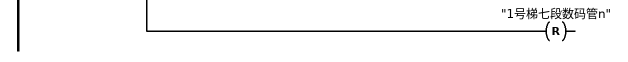
   RUNG wire#powerrail
      { S7_Templates := "SrcType := Int" } EQ_Contact(in1 := "1号梯当前楼层数", in2 := 1)
      wire#w1
      R_Coil( "1号梯七段数码管a" )
   END_RUNG
   RUNG wire#w1
      S_Coil( "1号梯七段数码管b" )
   END_RUNG
   RUNG wire#w1
      S_Coil( "1号梯七段数码管c" )
   END_RUNG
   RUNG wire#w1
      R_Coil( "1号梯七段数码管d" )
   END_RUNG
   RUNG wire#w1
      R_Coil( "1号梯七段数码管e" )
   END_RUNG
   RUNG wire#w1
      R_Coil( "1号梯七段数码管f" )
   END_RUNG
   RUNG wire#w1
      R_Coil( "1号梯七段数码管g" )
   END_RUNG
   RUNG wire#w1
      R_Coil( "1号梯七段数码管h" )
   END_RUNG
   RUNG wire#w1
      R_Coil( "1号梯七段数码管i" )
   END_RUNG
   RUNG wire#w1
      R_Coil( "1号梯七段数码管j" )
   END_RUNG
   RUNG wire#w1
      R_Coil( "1号梯七段数码管k" )
   END_RUNG
   RUNG wire#w1
      R_Coil( "1号梯七段数码管l" )
   END_RUNG
   RUNG wire#w1
      R_Coil( "1号梯七段数码管m" )
   END_RUNG
   RUNG wire#w1
      R_Coil( "1号梯七段数码管n" )
   END_RUNG
   RUNG wire#powerrail
      { S7_Templates := "SrcType := Int" } EQ_Contact(in1 := "1号梯当前楼层数", in2 := 2)
      wire#w2
      S_Coil( "1号梯七段数码管a" )
   END_RUNG
   RUNG wire#w2
      S_Coil( "1号梯七段数码管b" )
   END_RUNG
   RUNG wire#w2
      R_Coil( "1号梯七段数码管c" )
   END_RUNG
   RUNG wire#w2
      S_Coil( "1号梯七段数码管d" )
   END_RUNG
   RUNG wire#w2
      S_Coil( "1号梯七段数码管e" )
   END_RUNG
   RUNG wire#w2
      R_Coil( "1号梯七段数码管f" )
   END_RUNG
   RUNG wire#w2
      S_Coil( "1号梯七段数码管g" )
   END_RUNG
   RUNG wire#w2
      R_Coil( "1号梯七段数码管h" )
   END_RUNG
   RUNG wire#w2
      R_Coil( "1号梯七段数码管i" )
   END_RUNG
   RUNG wire#w2
      R_Coil( "1号梯七段数码管j" )
   END_RUNG
   RUNG wire#w2
      R_Coil( "1号梯七段数码管k" )
   END_RUNG
   RUNG wire#w2
      R_Coil( "1号梯七段数码管l" )
   END_RUNG
   RUNG wire#w2
      R_Coil( "1号梯七段数码管m" )
   END_RUNG
   RUNG wire#w2
      R_Coil( "1号梯七段数码管n" )
   END_RUNG
   RUNG wire#powerrail
      { S7_Templates := "SrcType := Int" } EQ_Contact(in1 := "1号梯当前楼层数", in2 := 3)
      wire#w3
      S_Coil( "1号梯七段数码管a" )
   END_RUNG
   RUNG wire#w3
      S_Coil( "1号梯七段数码管b" )
   END_RUNG
   RUNG wire#w3
      S_Coil( "1号梯七段数码管c" )
   END_RUNG
   RUNG wire#w3
      S_Coil( "1号梯七段数码管d" )
   END_RUNG
   RUNG wire#w3
      R_Coil( "1号梯七段数码管e" )
   END_RUNG
   RUNG wire#w3
      R_Coil( "1号梯七段数码管f" )
   END_RUNG
   RUNG wire#w3
      S_Coil( "1号梯七段数码管g" )
   END_RUNG
   RUNG wire#w3
      R_Coil( "1号梯七段数码管h" )
   END_RUNG
   RUNG wire#w3
      R_Coil( "1号梯七段数码管i" )
   END_RUNG
   RUNG wire#w3
      R_Coil( "1号梯七段数码管j" )
   END_RUNG
   RUNG wire#w3
      R_Coil( "1号梯七段数码管k" )
   END_RUNG
   RUNG wire#w3
      R_Coil( "1号梯七段数码管l" )
   END_RUNG
   RUNG wire#w3
      R_Coil( "1号梯七段数码管m" )
   END_RUNG
   RUNG wire#w3
      R_Coil( "1号梯七段数码管n" )
   END_RUNG
   RUNG wire#powerrail
      { S7_Templates := "SrcType := Int" } EQ_Contact(in1 := "1号梯当前楼层数", in2 := 4)
      wire#w4
      R_Coil( "1号梯七段数码管a" )
   END_RUNG
   RUNG wire#w4
      S_Coil( "1号梯七段数码管b" )
   END_RUNG
   RUNG wire#w4
      S_Coil( "1号梯七段数码管c" )
   END_RUNG
   RUNG wire#w4
      R_Coil( "1号梯七段数码管d" )
   END_RUNG
   RUNG wire#w4
      R_Coil( "1号梯七段数码管e" )
   END_RUNG
   RUNG wire#w4
      S_Coil( "1号梯七段数码管f" )
   END_RUNG
   RUNG wire#w4
      S_Coil( "1号梯七段数码管g" )
   END_RUNG
   RUNG wire#w4
      R_Coil( "1号梯七段数码管h" )
   END_RUNG
   RUNG wire#w4
      R_Coil( "1号梯七段数码管i" )
   END_RUNG
   RUNG wire#w4
      R_Coil( "1号梯七段数码管j" )
   END_RUNG
   RUNG wire#w4
      R_Coil( "1号梯七段数码管k" )
   END_RUNG
   RUNG wire#w4
      R_Coil( "1号梯七段数码管l" )
   END_RUNG
   RUNG wire#w4
      R_Coil( "1号梯七段数码管m" )
   END_RUNG
   RUNG wire#w4
      R_Coil( "1号梯七段数码管n" )
   END_RUNG
   RUNG wire#powerrail
      { S7_Templates := "SrcType := Int" } EQ_Contact(in1 := "1号梯当前楼层数", in2 := 5)
      wire#w5
      S_Coil( "1号梯七段数码管a" )
   END_RUNG
   RUNG wire#w5
      R_Coil( "1号梯七段数码管b" )
   END_RUNG
   RUNG wire#w5
      S_Coil( "1号梯七段数码管c" )
   END_RUNG
   RUNG wire#w5
      S_Coil( "1号梯七段数码管d" )
   END_RUNG
   RUNG wire#w5
      R_Coil( "1号梯七段数码管e" )
   END_RUNG
   RUNG wire#w5
      S_Coil( "1号梯七段数码管f" )
   END_RUNG
   RUNG wire#w5
      S_Coil( "1号梯七段数码管g" )
   END_RUNG
   RUNG wire#w5
      R_Coil( "1号梯七段数码管h" )
   END_RUNG
   RUNG wire#w5
      R_Coil( "1号梯七段数码管i" )
   END_RUNG
   RUNG wire#w5
      R_Coil( "1号梯七段数码管j" )
   END_RUNG
   RUNG wire#w5
      R_Coil( "1号梯七段数码管k" )
   END_RUNG
   RUNG wire#w5
      R_Coil( "1号梯七段数码管l" )
   END_RUNG
   RUNG wire#w5
      R_Coil( "1号梯七段数码管m" )
   END_RUNG
   RUNG wire#w5
      R_Coil( "1号梯七段数码管n" )
   END_RUNG
   RUNG wire#powerrail
      { S7_Templates := "SrcType := Int" } EQ_Contact(in1 := "1号梯当前楼层数", in2 := 6)
      wire#w6
      S_Coil( "1号梯七段数码管a" )
   END_RUNG
   RUNG wire#w6
      R_Coil( "1号梯七段数码管b" )
   END_RUNG
   RUNG wire#w6
      S_Coil( "1号梯七段数码管c" )
   END_RUNG
   RUNG wire#w6
      S_Coil( "1号梯七段数码管d" )
   END_RUNG
   RUNG wire#w6
      S_Coil( "1号梯七段数码管e" )
   END_RUNG
   RUNG wire#w6
      S_Coil( "1号梯七段数码管f" )
   END_RUNG
   RUNG wire#w6
      S_Coil( "1号梯七段数码管g" )
   END_RUNG
   RUNG wire#w6
      R_Coil( "1号梯七段数码管h" )
   END_RUNG
   RUNG wire#w6
      R_Coil( "1号梯七段数码管i" )
   END_RUNG
   RUNG wire#w6
      R_Coil( "1号梯七段数码管j" )
   END_RUNG
   RUNG wire#w6
      R_Coil( "1号梯七段数码管k" )
   END_RUNG
   RUNG wire#w6
      R_Coil( "1号梯七段数码管l" )
   END_RUNG
   RUNG wire#w6
      R_Coil( "1号梯七段数码管m" )
   END_RUNG
   RUNG wire#w6
      R_Coil( "1号梯七段数码管n" )
   END_RUNG
   RUNG wire#powerrail
      { S7_Templates := "SrcType := Int" } EQ_Contact(in1 := "1号梯当前楼层数", in2 := 7)
      wire#w7
      S_Coil( "1号梯七段数码管a" )
   END_RUNG
   RUNG wire#w7
      S_Coil( "1号梯七段数码管b" )
   END_RUNG
   RUNG wire#w7
      S_Coil( "1号梯七段数码管c" )
   END_RUNG
   RUNG wire#w7
      R_Coil( "1号梯七段数码管d" )
   END_RUNG
   RUNG wire#w7
      R_Coil( "1号梯七段数码管e" )
   END_RUNG
   RUNG wire#w7
      R_Coil( "1号梯七段数码管f" )
   END_RUNG
   RUNG wire#w7
      R_Coil( "1号梯七段数码管g" )
   END_RUNG
   RUNG wire#w7
      R_Coil( "1号梯七段数码管h" )
   END_RUNG
   RUNG wire#w7
      R_Coil( "1号梯七段数码管i" )
   END_RUNG
   RUNG wire#w7
      R_Coil( "1号梯七段数码管j" )
   END_RUNG
   RUNG wire#w7
      R_Coil( "1号梯七段数码管k" )
   END_RUNG
   RUNG wire#w7
      R_Coil( "1号梯七段数码管l" )
   END_RUNG
   RUNG wire#w7
      R_Coil( "1号梯七段数码管m" )
   END_RUNG
   RUNG wire#w7
      R_Coil( "1号梯七段数码管n" )
   END_RUNG
   RUNG wire#powerrail
      { S7_Templates := "SrcType := Int" } EQ_Contact(in1 := "1号梯当前楼层数", in2 := 8)
      wire#w8
      S_Coil( "1号梯七段数码管a" )
   END_RUNG
   RUNG wire#w8
      S_Coil( "1号梯七段数码管b" )
   END_RUNG
   RUNG wire#w8
      S_Coil( "1号梯七段数码管c" )
   END_RUNG
   RUNG wire#w8
      S_Coil( "1号梯七段数码管d" )
   END_RUNG
   RUNG wire#w8
      S_Coil( "1号梯七段数码管e" )
   END_RUNG
   RUNG wire#w8
      S_Coil( "1号梯七段数码管f" )
   END_RUNG
   RUNG wire#w8
      S_Coil( "1号梯七段数码管g" )
   END_RUNG
   RUNG wire#w8
      R_Coil( "1号梯七段数码管h" )
   END_RUNG
   RUNG wire#w8
      R_Coil( "1号梯七段数码管i" )
   END_RUNG
   RUNG wire#w8
      R_Coil( "1号梯七段数码管j" )
   END_RUNG
   RUNG wire#w8
      R_Coil( "1号梯七段数码管k" )
   END_RUNG
   RUNG wire#w8
      R_Coil( "1号梯七段数码管l" )
   END_RUNG
   RUNG wire#w8
      R_Coil( "1号梯七段数码管m" )
   END_RUNG
   RUNG wire#w8
      R_Coil( "1号梯七段数码管n" )
   END_RUNG
   RUNG wire#powerrail
      { S7_Templates := "SrcType := Int" } EQ_Contact(in1 := "1号梯当前楼层数", in2 := 9)
      wire#w9
      S_Coil( "1号梯七段数码管a" )
   END_RUNG
   RUNG wire#w9
      S_Coil( "1号梯七段数码管b" )
   END_RUNG
   RUNG wire#w9
      S_Coil( "1号梯七段数码管c" )
   END_RUNG
   RUNG wire#w9
      S_Coil( "1号梯七段数码管d" )
   END_RUNG
   RUNG wire#w9
      R_Coil( "1号梯七段数码管e" )
   END_RUNG
   RUNG wire#w9
      S_Coil( "1号梯七段数码管f" )
   END_RUNG
   RUNG wire#w9
      S_Coil( "1号梯七段数码管g" )
   END_RUNG
   RUNG wire#w9
      R_Coil( "1号梯七段数码管h" )
   END_RUNG
   RUNG wire#w9
      R_Coil( "1号梯七段数码管i" )
   END_RUNG
   RUNG wire#w9
      R_Coil( "1号梯七段数码管j" )
   END_RUNG
   RUNG wire#w9
      R_Coil( "1号梯七段数码管k" )
   END_RUNG
   RUNG wire#w9
      R_Coil( "1号梯七段数码管l" )
   END_RUNG
   RUNG wire#w9
      R_Coil( "1号梯七段数码管m" )
   END_RUNG
   RUNG wire#w9
      R_Coil( "1号梯七段数码管n" )
   END_RUNG
   RUNG wire#powerrail
      { S7_Templates := "SrcType := Int" } EQ_Contact(in1 := "1号梯当前楼层数", in2 := 10)
      wire#w10
      S_Coil( "1号梯七段数码管a" )
   END_RUNG
   RUNG wire#w10
      S_Coil( "1号梯七段数码管b" )
   END_RUNG
   RUNG wire#w10
      S_Coil( "1号梯七段数码管c" )
   END_RUNG
   RUNG wire#w10
      S_Coil( "1号梯七段数码管d" )
   END_RUNG
   RUNG wire#w10
      S_Coil( "1号梯七段数码管e" )
   END_RUNG
   RUNG wire#w10
      S_Coil( "1号梯七段数码管f" )
   END_RUNG
   RUNG wire#w10
      R_Coil( "1号梯七段数码管g" )
   END_RUNG
   RUNG wire#w10
      R_Coil( "1号梯七段数码管h" )
   END_RUNG
   RUNG wire#w10
      S_Coil( "1号梯七段数码管i" )
   END_RUNG
   RUNG wire#w10
      S_Coil( "1号梯七段数码管j" )
   END_RUNG
   RUNG wire#w10
      R_Coil( "1号梯七段数码管k" )
   END_RUNG
   RUNG wire#w10
      R_Coil( "1号梯七段数码管l" )
   END_RUNG
   RUNG wire#w10
      R_Coil( "1号梯七段数码管m" )
   END_RUNG
   RUNG wire#w10
      R_Coil( "1号梯七段数码管n" )
   END_RUNG
   // the same network as SCL:
   IF "1号梯当前楼层数" = 1 THEN
       "1号梯七段数码管a" := FALSE;
       "1号梯七段数码管b" := TRUE;
       "1号梯七段数码管c" := TRUE;
       "1号梯七段数码管d" := FALSE;
       "1号梯七段数码管e" := FALSE;
       "1号梯七段数码管f" := FALSE;
       "1号梯七段数码管g" := FALSE;
       "1号梯七段数码管h" := FALSE;
       "1号梯七段数码管i" := FALSE;
       "1号梯七段数码管j" := FALSE;
       "1号梯七段数码管k" := FALSE;
       "1号梯七段数码管l" := FALSE;
       "1号梯七段数码管m" := FALSE;
       "1号梯七段数码管n" := FALSE;
   END_IF;
   IF "1号梯当前楼层数" = 2 THEN
       "1号梯七段数码管a" := TRUE;
       "1号梯七段数码管b" := TRUE;
       "1号梯七段数码管c" := FALSE;
       "1号梯七段数码管d" := TRUE;
       "1号梯七段数码管e" := TRUE;
       "1号梯七段数码管f" := FALSE;
       "1号梯七段数码管g" := TRUE;
       "1号梯七段数码管h" := FALSE;
       "1号梯七段数码管i" := FALSE;
       "1号梯七段数码管j" := FALSE;
       "1号梯七段数码管k" := FALSE;
       "1号梯七段数码管l" := FALSE;
       "1号梯七段数码管m" := FALSE;
       "1号梯七段数码管n" := FALSE;
   END_IF;
   IF "1号梯当前楼层数" = 3 THEN
       "1号梯七段数码管a" := TRUE;
       "1号梯七段数码管b" := TRUE;
       "1号梯七段数码管c" := TRUE;
       "1号梯七段数码管d" := TRUE;
       "1号梯七段数码管e" := FALSE;
       "1号梯七段数码管f" := FALSE;
       "1号梯七段数码管g" := TRUE;
       "1号梯七段数码管h" := FALSE;
       "1号梯七段数码管i" := FALSE;
       "1号梯七段数码管j" := FALSE;
       "1号梯七段数码管k" := FALSE;
       "1号梯七段数码管l" := FALSE;
       "1号梯七段数码管m" := FALSE;
       "1号梯七段数码管n" := FALSE;
   END_IF;
   IF "1号梯当前楼层数" = 4 THEN
       "1号梯七段数码管a" := FALSE;
       "1号梯七段数码管b" := TRUE;
       "1号梯七段数码管c" := TRUE;
       "1号梯七段数码管d" := FALSE;
       "1号梯七段数码管e" := FALSE;
       "1号梯七段数码管f" := TRUE;
       "1号梯七段数码管g" := TRUE;
       "1号梯七段数码管h" := FALSE;
       "1号梯七段数码管i" := FALSE;
       "1号梯七段数码管j" := FALSE;
       "1号梯七段数码管k" := FALSE;
       "1号梯七段数码管l" := FALSE;
       "1号梯七段数码管m" := FALSE;
       "1号梯七段数码管n" := FALSE;
   END_IF;
   IF "1号梯当前楼层数" = 5 THEN
       "1号梯七段数码管a" := TRUE;
       "1号梯七段数码管b" := FALSE;
       "1号梯七段数码管c" := TRUE;
       "1号梯七段数码管d" := TRUE;
       "1号梯七段数码管e" := FALSE;
       "1号梯七段数码管f" := TRUE;
       "1号梯七段数码管g" := TRUE;
       "1号梯七段数码管h" := FALSE;
       "1号梯七段数码管i" := FALSE;
       "1号梯七段数码管j" := FALSE;
       "1号梯七段数码管k" := FALSE;
       "1号梯七段数码管l" := FALSE;
       "1号梯七段数码管m" := FALSE;
       "1号梯七段数码管n" := FALSE;
   END_IF;
   IF "1号梯当前楼层数" = 6 THEN
       "1号梯七段数码管a" := TRUE;
       "1号梯七段数码管b" := FALSE;
       "1号梯七段数码管c" := TRUE;
       "1号梯七段数码管d" := TRUE;
       "1号梯七段数码管e" := TRUE;
       "1号梯七段数码管f" := TRUE;
       "1号梯七段数码管g" := TRUE;
       "1号梯七段数码管h" := FALSE;
       "1号梯七段数码管i" := FALSE;
       "1号梯七段数码管j" := FALSE;
       "1号梯七段数码管k" := FALSE;
       "1号梯七段数码管l" := FALSE;
       "1号梯七段数码管m" := FALSE;
       "1号梯七段数码管n" := FALSE;
   END_IF;
   IF "1号梯当前楼层数" = 7 THEN
       "1号梯七段数码管a" := TRUE;
       "1号梯七段数码管b" := TRUE;
       "1号梯七段数码管c" := TRUE;
       "1号梯七段数码管d" := FALSE;
       "1号梯七段数码管e" := FALSE;
       "1号梯七段数码管f" := FALSE;
       "1号梯七段数码管g" := FALSE;
       "1号梯七段数码管h" := FALSE;
       "1号梯七段数码管i" := FALSE;
       "1号梯七段数码管j" := FALSE;
       "1号梯七段数码管k" := FALSE;
       "1号梯七段数码管l" := FALSE;
       "1号梯七段数码管m" := FALSE;
       "1号梯七段数码管n" := FALSE;
   END_IF;
   IF "1号梯当前楼层数" = 8 THEN
       "1号梯七段数码管a" := TRUE;
       "1号梯七段数码管b" := TRUE;
       "1号梯七段数码管c" := TRUE;
       "1号梯七段数码管d" := TRUE;
       "1号梯七段数码管e" := TRUE;
       "1号梯七段数码管f" := TRUE;
       "1号梯七段数码管g" := TRUE;
       "1号梯七段数码管h" := FALSE;
       "1号梯七段数码管i" := FALSE;
       "1号梯七段数码管j" := FALSE;
       "1号梯七段数码管k" := FALSE;
       "1号梯七段数码管l" := FALSE;
       "1号梯七段数码管m" := FALSE;
       "1号梯七段数码管n" := FALSE;
   END_IF;
   IF "1号梯当前楼层数" = 9 THEN
       "1号梯七段数码管a" := TRUE;
       "1号梯七段数码管b" := TRUE;
       "1号梯七段数码管c" := TRUE;
       "1号梯七段数码管d" := TRUE;
       "1号梯七段数码管e" := FALSE;
       "1号梯七段数码管f" := TRUE;
       "1号梯七段数码管g" := TRUE;
       "1号梯七段数码管h" := FALSE;
       "1号梯七段数码管i" := FALSE;
       "1号梯七段数码管j" := FALSE;
       "1号梯七段数码管k" := FALSE;
       "1号梯七段数码管l" := FALSE;
       "1号梯七段数码管m" := FALSE;
       "1号梯七段数码管n" := FALSE;
   END_IF;
   IF "1号梯当前楼层数" = 10 THEN
       "1号梯七段数码管a" := TRUE;
       "1号梯七段数码管b" := TRUE;
       "1号梯七段数码管c" := TRUE;
       "1号梯七段数码管d" := TRUE;
       "1号梯七段数码管e" := TRUE;
       "1号梯七段数码管f" := TRUE;
       "1号梯七段数码管g" := FALSE;
       "1号梯七段数码管h" := FALSE;
       "1号梯七段数码管i" := TRUE;
       "1号梯七段数码管j" := TRUE;
       "1号梯七段数码管k" := FALSE;
       "1号梯七段数码管l" := FALSE;
       "1号梯七段数码管m" := FALSE;
       "1号梯七段数码管n" := FALSE;
   END_IF;
END_REGION

REGION Network 2: 上下行指示灯
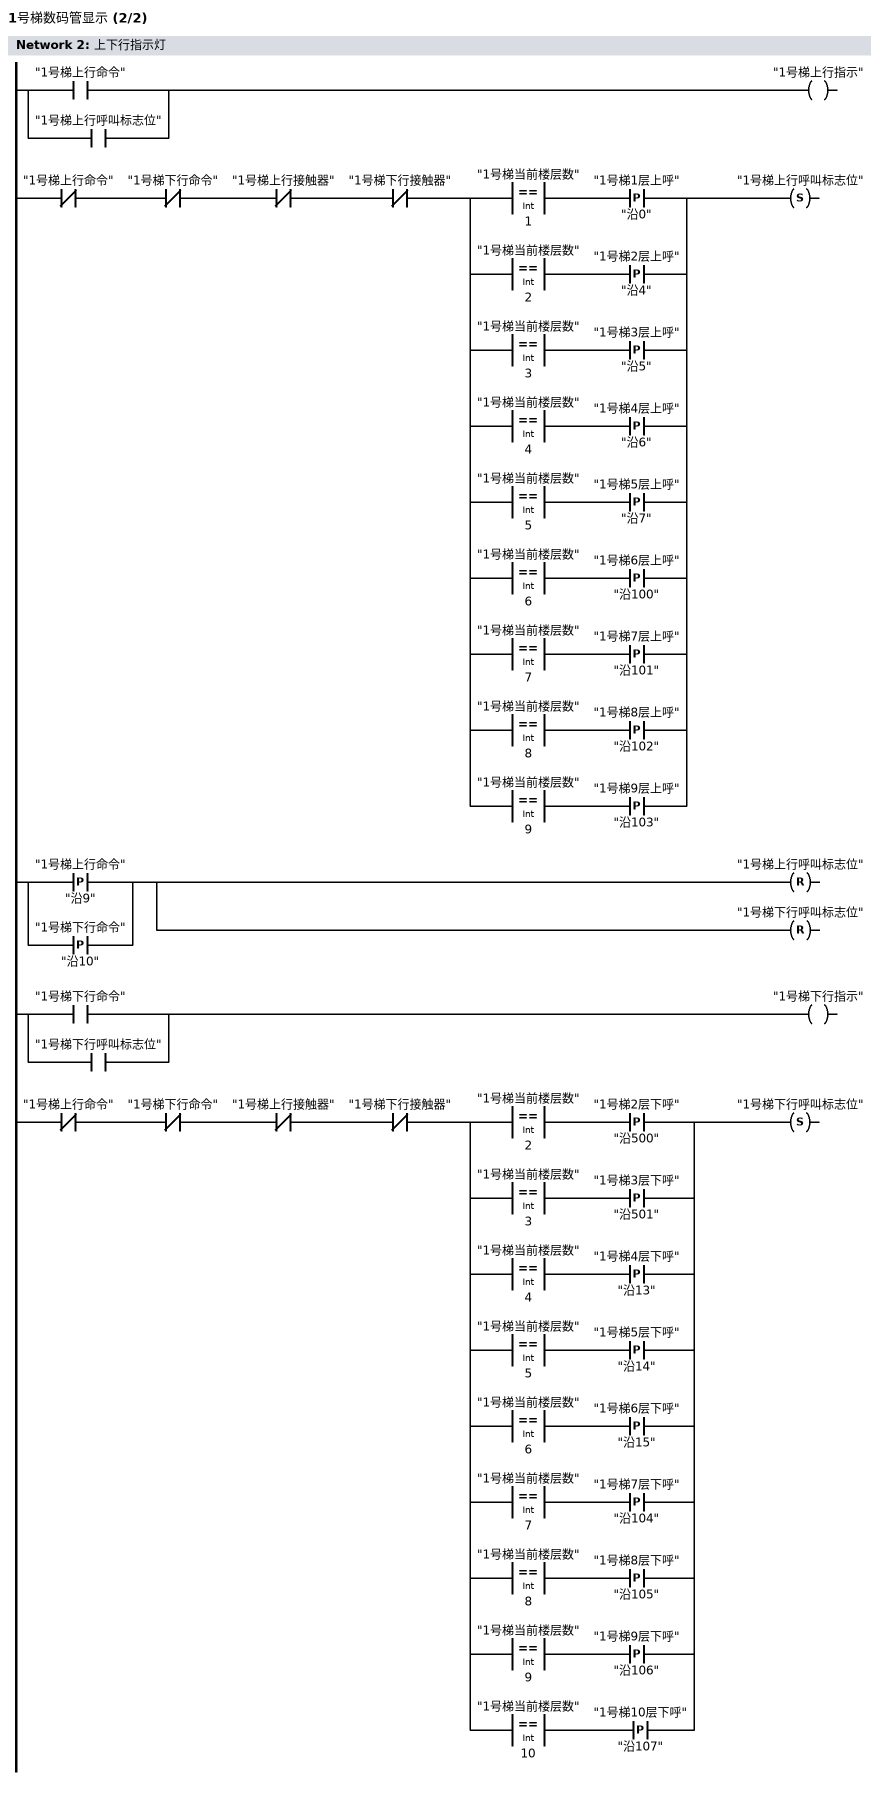
   RUNG wire#powerrail
      Contact( "1号梯上行命令" )
      wire#w1
      Coil( "1号梯上行指示" )
   END_RUNG
   RUNG wire#powerrail
      Contact( "1号梯上行呼叫标志位" )
   END_RUNG wire#w1
   RUNG wire#powerrail
      I_Contact( "1号梯上行命令" )
      I_Contact( "1号梯下行命令" )
      I_Contact( "1号梯上行接触器" )
      I_Contact( "1号梯下行接触器" )
      wire#w2
      { S7_Templates := "SrcType := Int" } EQ_Contact(in1 := "1号梯当前楼层数", in2 := 1)
      P_Contact(operand := "1号梯1层上呼", bit := "沿0")
      wire#w3
      S_Coil( "1号梯上行呼叫标志位" )
   END_RUNG
   RUNG wire#w2
      { S7_Templates := "SrcType := Int" } EQ_Contact(in1 := "1号梯当前楼层数", in2 := 2)
      P_Contact(operand := "1号梯2层上呼", bit := "沿4")
   END_RUNG wire#w3
   RUNG wire#w2
      { S7_Templates := "SrcType := Int" } EQ_Contact(in1 := "1号梯当前楼层数", in2 := 3)
      P_Contact(operand := "1号梯3层上呼", bit := "沿5")
   END_RUNG wire#w3
   RUNG wire#w2
      { S7_Templates := "SrcType := Int" } EQ_Contact(in1 := "1号梯当前楼层数", in2 := 4)
      P_Contact(operand := "1号梯4层上呼", bit := "沿6")
   END_RUNG wire#w3
   RUNG wire#w2
      { S7_Templates := "SrcType := Int" } EQ_Contact(in1 := "1号梯当前楼层数", in2 := 5)
      P_Contact(operand := "1号梯5层上呼", bit := "沿7")
   END_RUNG wire#w3
   RUNG wire#w2
      { S7_Templates := "SrcType := Int" } EQ_Contact(in1 := "1号梯当前楼层数", in2 := 6)
      P_Contact(operand := "1号梯6层上呼", bit := "沿100")
   END_RUNG wire#w3
   RUNG wire#w2
      { S7_Templates := "SrcType := Int" } EQ_Contact(in1 := "1号梯当前楼层数", in2 := 7)
      P_Contact(operand := "1号梯7层上呼", bit := "沿101")
   END_RUNG wire#w3
   RUNG wire#w2
      { S7_Templates := "SrcType := Int" } EQ_Contact(in1 := "1号梯当前楼层数", in2 := 8)
      P_Contact(operand := "1号梯8层上呼", bit := "沿102")
   END_RUNG wire#w3
   RUNG wire#w2
      { S7_Templates := "SrcType := Int" } EQ_Contact(in1 := "1号梯当前楼层数", in2 := 9)
      P_Contact(operand := "1号梯9层上呼", bit := "沿103")
   END_RUNG wire#w3
   RUNG wire#powerrail
      P_Contact(operand := "1号梯上行命令", bit := "沿9")
      wire#w4
      R_Coil( "1号梯上行呼叫标志位" )
   END_RUNG
   RUNG wire#powerrail
      P_Contact(operand := "1号梯下行命令", bit := "沿10")
   END_RUNG wire#w4
   RUNG wire#w4
      R_Coil( "1号梯下行呼叫标志位" )
   END_RUNG
   RUNG wire#powerrail
      Contact( "1号梯下行命令" )
      wire#w5
      Coil( "1号梯下行指示" )
   END_RUNG
   RUNG wire#powerrail
      Contact( "1号梯下行呼叫标志位" )
   END_RUNG wire#w5
   RUNG wire#powerrail
      I_Contact( "1号梯上行命令" )
      I_Contact( "1号梯下行命令" )
      I_Contact( "1号梯上行接触器" )
      I_Contact( "1号梯下行接触器" )
      wire#w6
      { S7_Templates := "SrcType := Int" } EQ_Contact(in1 := "1号梯当前楼层数", in2 := 2)
      P_Contact(operand := "1号梯2层下呼", bit := "沿500")
      wire#w7
      S_Coil( "1号梯下行呼叫标志位" )
   END_RUNG
   RUNG wire#w6
      { S7_Templates := "SrcType := Int" } EQ_Contact(in1 := "1号梯当前楼层数", in2 := 3)
      P_Contact(operand := "1号梯3层下呼", bit := "沿501")
   END_RUNG wire#w7
   RUNG wire#w6
      { S7_Templates := "SrcType := Int" } EQ_Contact(in1 := "1号梯当前楼层数", in2 := 4)
      P_Contact(operand := "1号梯4层下呼", bit := "沿13")
   END_RUNG wire#w7
   RUNG wire#w6
      { S7_Templates := "SrcType := Int" } EQ_Contact(in1 := "1号梯当前楼层数", in2 := 5)
      P_Contact(operand := "1号梯5层下呼", bit := "沿14")
   END_RUNG wire#w7
   RUNG wire#w6
      { S7_Templates := "SrcType := Int" } EQ_Contact(in1 := "1号梯当前楼层数", in2 := 6)
      P_Contact(operand := "1号梯6层下呼", bit := "沿15")
   END_RUNG wire#w7
   RUNG wire#w6
      { S7_Templates := "SrcType := Int" } EQ_Contact(in1 := "1号梯当前楼层数", in2 := 7)
      P_Contact(operand := "1号梯7层下呼", bit := "沿104")
   END_RUNG wire#w7
   RUNG wire#w6
      { S7_Templates := "SrcType := Int" } EQ_Contact(in1 := "1号梯当前楼层数", in2 := 8)
      P_Contact(operand := "1号梯8层下呼", bit := "沿105")
   END_RUNG wire#w7
   RUNG wire#w6
      { S7_Templates := "SrcType := Int" } EQ_Contact(in1 := "1号梯当前楼层数", in2 := 9)
      P_Contact(operand := "1号梯9层下呼", bit := "沿106")
   END_RUNG wire#w7
   RUNG wire#w6
      { S7_Templates := "SrcType := Int" } EQ_Contact(in1 := "1号梯当前楼层数", in2 := 10)
      P_Contact(operand := "1号梯10层下呼", bit := "沿107")
   END_RUNG wire#w7
   // the same network as SCL:
   "1号梯上行指示" := "1号梯上行命令" OR "1号梯上行呼叫标志位";
   #_w1 := NOT "1号梯上行命令" AND NOT "1号梯下行命令" AND NOT "1号梯上行接触器" AND NOT "1号梯下行接触器" AND ("1号梯当前楼层数" = 1) AND "1号梯1层上呼" AND NOT "沿0";   // rising edge of "1号梯1层上呼"
   "沿0" := "1号梯1层上呼";
   #_w2 := NOT "1号梯上行命令" AND NOT "1号梯下行命令" AND NOT "1号梯上行接触器" AND NOT "1号梯下行接触器" AND ("1号梯当前楼层数" = 2) AND "1号梯2层上呼" AND NOT "沿4";   // rising edge of "1号梯2层上呼"
   "沿4" := "1号梯2层上呼";
   #_w3 := NOT "1号梯上行命令" AND NOT "1号梯下行命令" AND NOT "1号梯上行接触器" AND NOT "1号梯下行接触器" AND ("1号梯当前楼层数" = 3) AND "1号梯3层上呼" AND NOT "沿5";   // rising edge of "1号梯3层上呼"
   "沿5" := "1号梯3层上呼";
   #_w4 := NOT "1号梯上行命令" AND NOT "1号梯下行命令" AND NOT "1号梯上行接触器" AND NOT "1号梯下行接触器" AND ("1号梯当前楼层数" = 4) AND "1号梯4层上呼" AND NOT "沿6";   // rising edge of "1号梯4层上呼"
   "沿6" := "1号梯4层上呼";
   #_w5 := NOT "1号梯上行命令" AND NOT "1号梯下行命令" AND NOT "1号梯上行接触器" AND NOT "1号梯下行接触器" AND ("1号梯当前楼层数" = 5) AND "1号梯5层上呼" AND NOT "沿7";   // rising edge of "1号梯5层上呼"
   "沿7" := "1号梯5层上呼";
   #_w6 := NOT "1号梯上行命令" AND NOT "1号梯下行命令" AND NOT "1号梯上行接触器" AND NOT "1号梯下行接触器" AND ("1号梯当前楼层数" = 6) AND "1号梯6层上呼" AND NOT "沿100";   // rising edge of "1号梯6层上呼"
   "沿100" := "1号梯6层上呼";
   #_w7 := NOT "1号梯上行命令" AND NOT "1号梯下行命令" AND NOT "1号梯上行接触器" AND NOT "1号梯下行接触器" AND ("1号梯当前楼层数" = 7) AND "1号梯7层上呼" AND NOT "沿101";   // rising edge of "1号梯7层上呼"
   "沿101" := "1号梯7层上呼";
   #_w8 := NOT "1号梯上行命令" AND NOT "1号梯下行命令" AND NOT "1号梯上行接触器" AND NOT "1号梯下行接触器" AND ("1号梯当前楼层数" = 8) AND "1号梯8层上呼" AND NOT "沿102";   // rising edge of "1号梯8层上呼"
   "沿102" := "1号梯8层上呼";
   #_w9 := NOT "1号梯上行命令" AND NOT "1号梯下行命令" AND NOT "1号梯上行接触器" AND NOT "1号梯下行接触器" AND ("1号梯当前楼层数" = 9) AND "1号梯9层上呼" AND NOT "沿103";   // rising edge of "1号梯9层上呼"
   "沿103" := "1号梯9层上呼";
   IF #_w1 OR #_w2 OR #_w3 OR #_w4 OR #_w5 OR #_w6 OR #_w7 OR #_w8 OR #_w9 THEN "1号梯上行呼叫标志位" := TRUE; END_IF;
   #_w10 := "1号梯上行命令" AND NOT "沿9";   // rising edge of "1号梯上行命令"
   "沿9" := "1号梯上行命令";
   #_w11 := "1号梯下行命令" AND NOT "沿10";   // rising edge of "1号梯下行命令"
   "沿10" := "1号梯下行命令";
   IF #_w10 OR #_w11 THEN
       "1号梯上行呼叫标志位" := FALSE;
       "1号梯下行呼叫标志位" := FALSE;
   END_IF;
   "1号梯下行指示" := "1号梯下行命令" OR "1号梯下行呼叫标志位";
   #_w12 := NOT "1号梯上行命令" AND NOT "1号梯下行命令" AND NOT "1号梯上行接触器" AND NOT "1号梯下行接触器" AND ("1号梯当前楼层数" = 2) AND "1号梯2层下呼" AND NOT "沿500";   // rising edge of "1号梯2层下呼"
   "沿500" := "1号梯2层下呼";
   #_w13 := NOT "1号梯上行命令" AND NOT "1号梯下行命令" AND NOT "1号梯上行接触器" AND NOT "1号梯下行接触器" AND ("1号梯当前楼层数" = 3) AND "1号梯3层下呼" AND NOT "沿501";   // rising edge of "1号梯3层下呼"
   "沿501" := "1号梯3层下呼";
   #_w14 := NOT "1号梯上行命令" AND NOT "1号梯下行命令" AND NOT "1号梯上行接触器" AND NOT "1号梯下行接触器" AND ("1号梯当前楼层数" = 4) AND "1号梯4层下呼" AND NOT "沿13";   // rising edge of "1号梯4层下呼"
   "沿13" := "1号梯4层下呼";
   #_w15 := NOT "1号梯上行命令" AND NOT "1号梯下行命令" AND NOT "1号梯上行接触器" AND NOT "1号梯下行接触器" AND ("1号梯当前楼层数" = 5) AND "1号梯5层下呼" AND NOT "沿14";   // rising edge of "1号梯5层下呼"
   "沿14" := "1号梯5层下呼";
   #_w16 := NOT "1号梯上行命令" AND NOT "1号梯下行命令" AND NOT "1号梯上行接触器" AND NOT "1号梯下行接触器" AND ("1号梯当前楼层数" = 6) AND "1号梯6层下呼" AND NOT "沿15";   // rising edge of "1号梯6层下呼"
   "沿15" := "1号梯6层下呼";
   #_w17 := NOT "1号梯上行命令" AND NOT "1号梯下行命令" AND NOT "1号梯上行接触器" AND NOT "1号梯下行接触器" AND ("1号梯当前楼层数" = 7) AND "1号梯7层下呼" AND NOT "沿104";   // rising edge of "1号梯7层下呼"
   "沿104" := "1号梯7层下呼";
   #_w18 := NOT "1号梯上行命令" AND NOT "1号梯下行命令" AND NOT "1号梯上行接触器" AND NOT "1号梯下行接触器" AND ("1号梯当前楼层数" = 8) AND "1号梯8层下呼" AND NOT "沿105";   // rising edge of "1号梯8层下呼"
   "沿105" := "1号梯8层下呼";
   #_w19 := NOT "1号梯上行命令" AND NOT "1号梯下行命令" AND NOT "1号梯上行接触器" AND NOT "1号梯下行接触器" AND ("1号梯当前楼层数" = 9) AND "1号梯9层下呼" AND NOT "沿106";   // rising edge of "1号梯9层下呼"
   "沿106" := "1号梯9层下呼";
   #_w20 := NOT "1号梯上行命令" AND NOT "1号梯下行命令" AND NOT "1号梯上行接触器" AND NOT "1号梯下行接触器" AND ("1号梯当前楼层数" = 10) AND "1号梯10层下呼" AND NOT "沿107";   // rising edge of "1号梯10层下呼"
   "沿107" := "1号梯10层下呼";
   IF #_w12 OR #_w13 OR #_w14 OR #_w15 OR #_w16 OR #_w17 OR #_w18 OR #_w19 OR #_w20 THEN
       "1号梯下行呼叫标志位" := TRUE;
   END_IF;
END_REGION
END_FUNCTION

FUNCTION "2号梯数码管显示" : Void   // FC10, LAD
{ S7_Optimized_Access := 'TRUE' }
VERSION : 0.1
   VAR_TEMP   // added for the SCL form of the ladder/FBD networks
      _w1 : Bool;
      _w2 : Bool;
      _w3 : Bool;
      _w4 : Bool;
      _w5 : Bool;
      _w6 : Bool;
      _w7 : Bool;
      _w8 : Bool;
      _w9 : Bool;
      _w10 : Bool;
      _w11 : Bool;
      _w12 : Bool;
      _w13 : Bool;
      _w14 : Bool;
      _w15 : Bool;
      _w16 : Bool;
      _w17 : Bool;
      _w18 : Bool;
      _w19 : Bool;
      _w20 : Bool;
   END_VAR
BEGIN

REGION Network 1: 根据楼层显示数码管
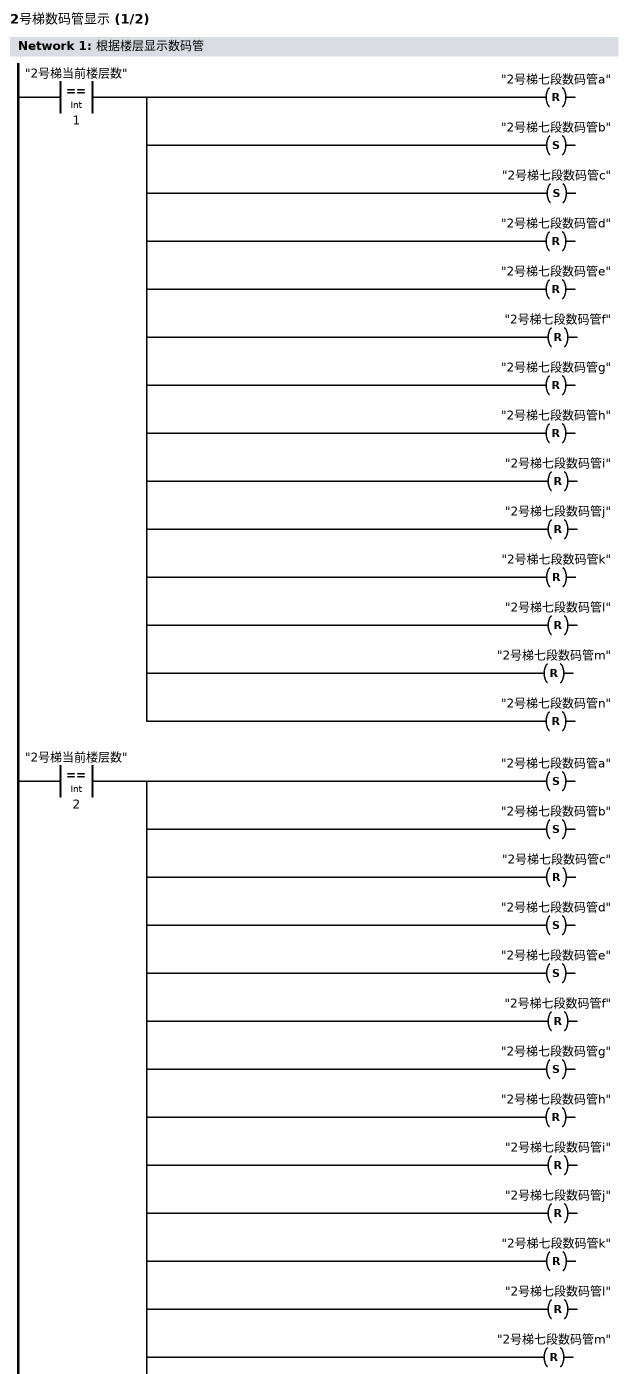
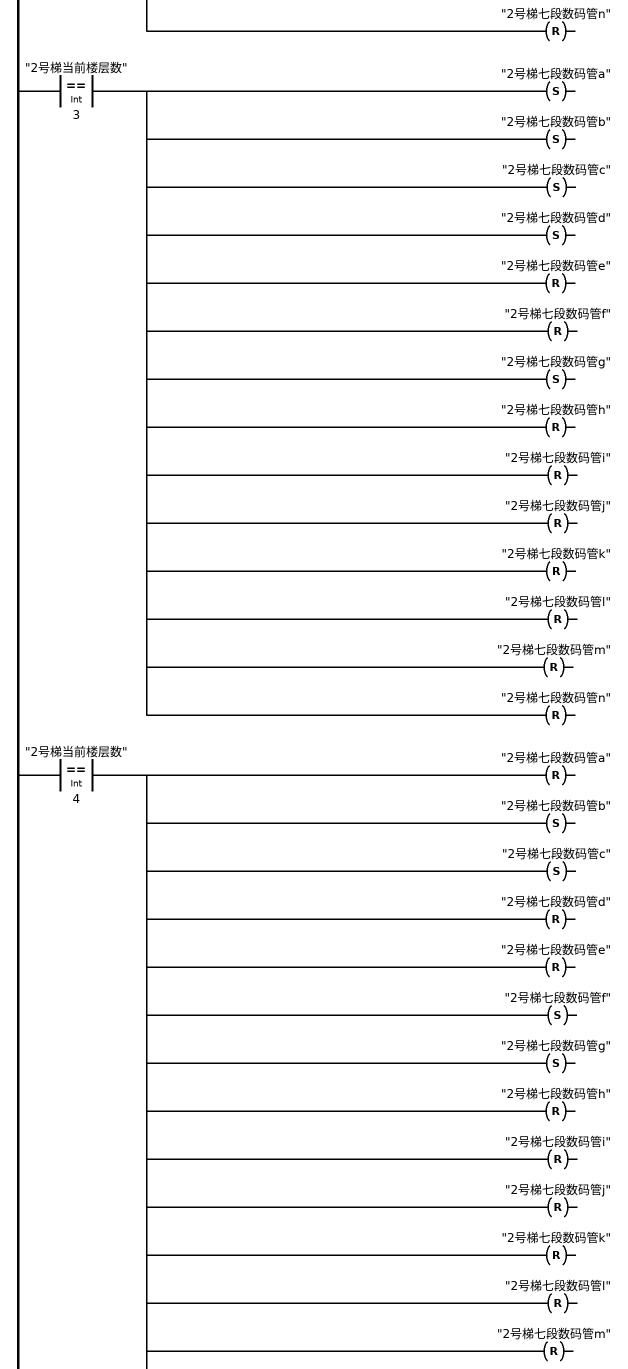
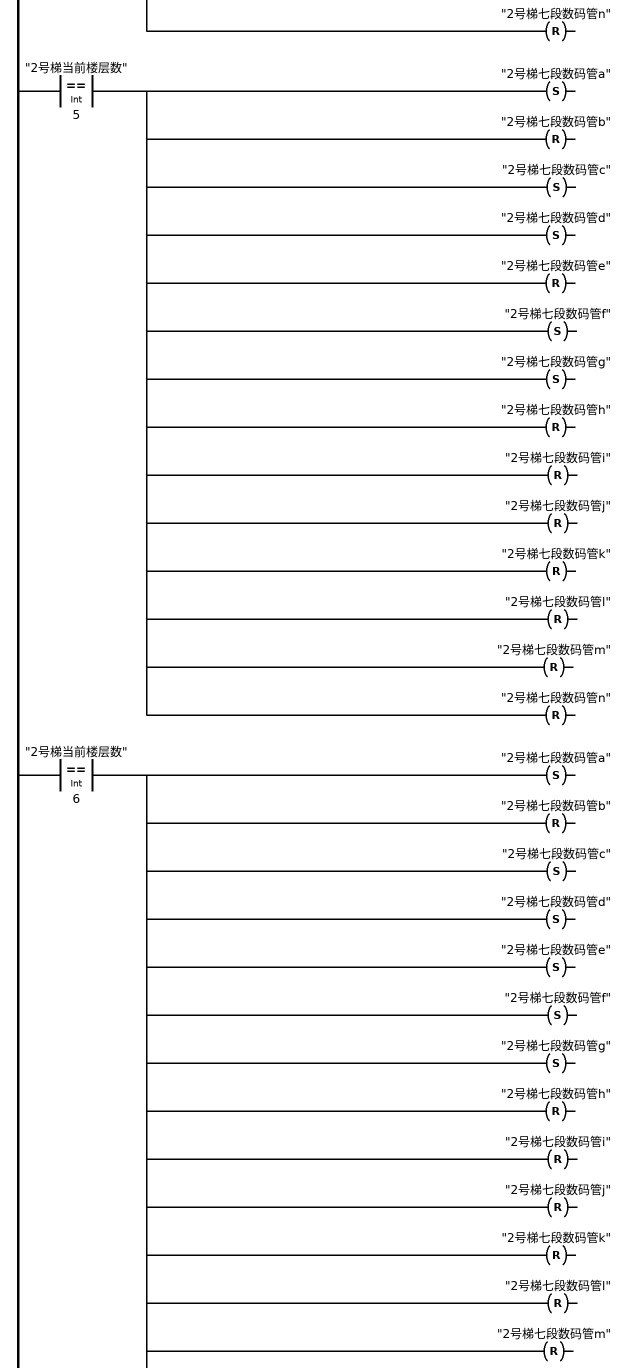
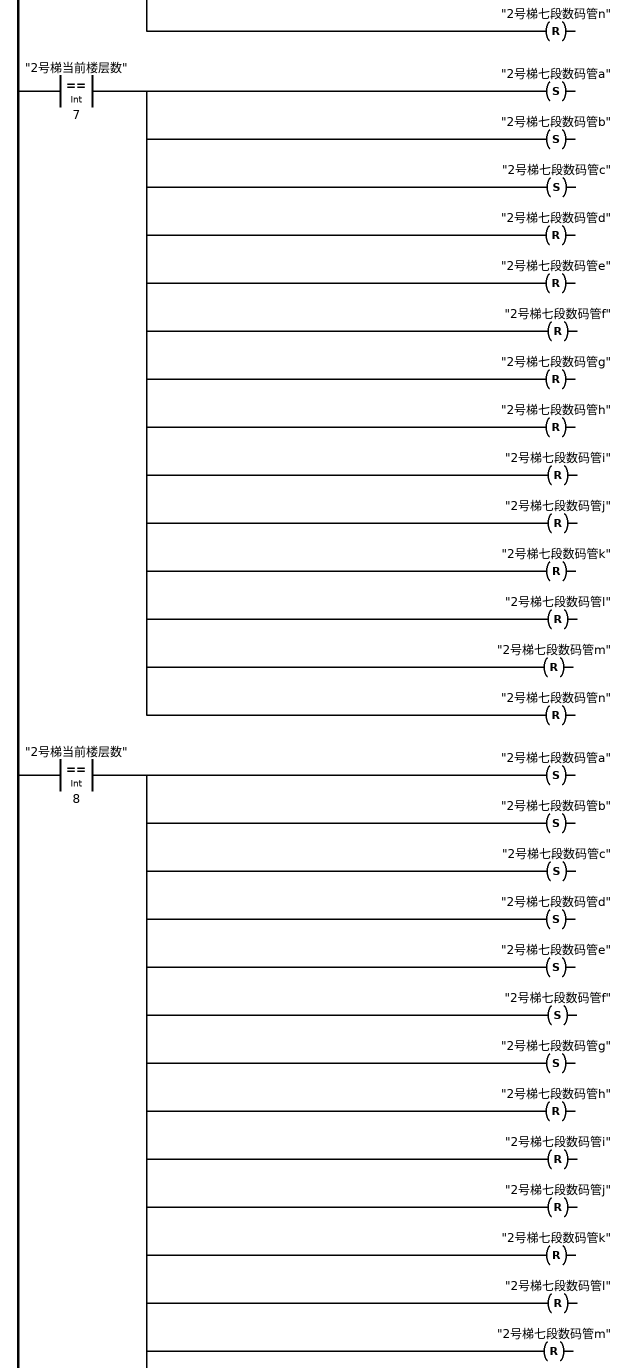
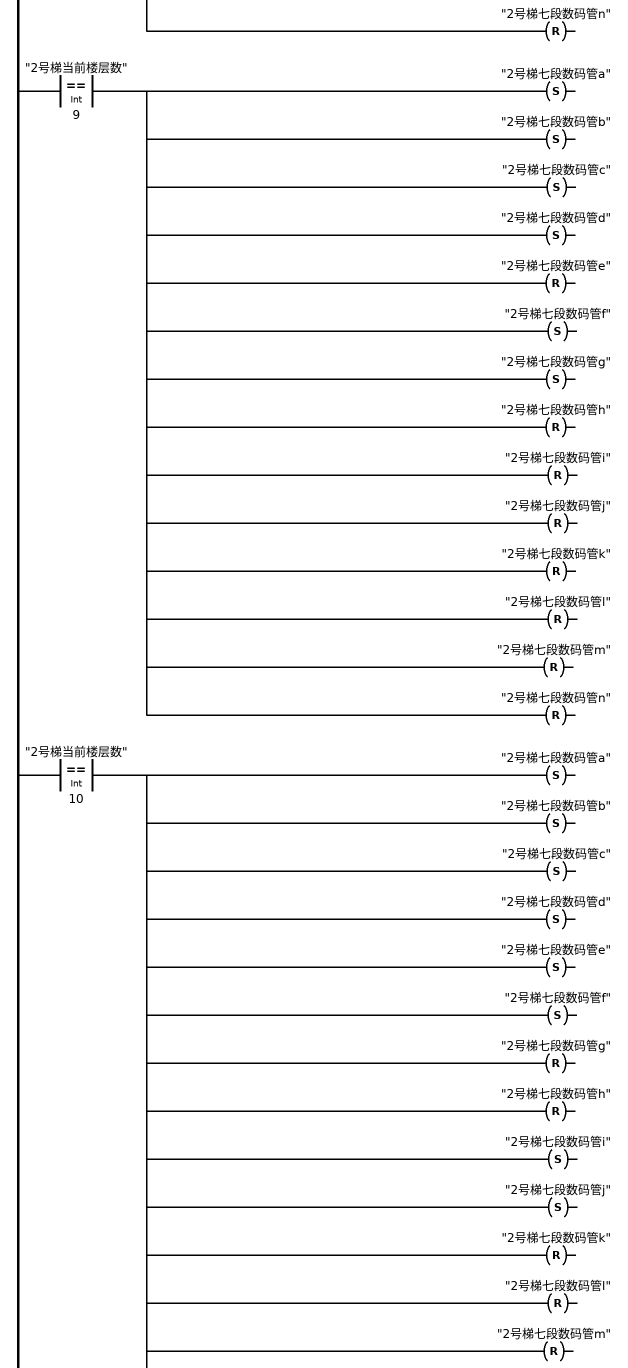
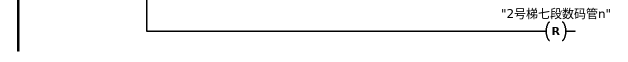
   RUNG wire#powerrail
      { S7_Templates := "SrcType := Int" } EQ_Contact(in1 := "2号梯当前楼层数", in2 := 1)
      wire#w1
      R_Coil( "2号梯七段数码管a" )
   END_RUNG
   RUNG wire#w1
      S_Coil( "2号梯七段数码管b" )
   END_RUNG
   RUNG wire#w1
      S_Coil( "2号梯七段数码管c" )
   END_RUNG
   RUNG wire#w1
      R_Coil( "2号梯七段数码管d" )
   END_RUNG
   RUNG wire#w1
      R_Coil( "2号梯七段数码管e" )
   END_RUNG
   RUNG wire#w1
      R_Coil( "2号梯七段数码管f" )
   END_RUNG
   RUNG wire#w1
      R_Coil( "2号梯七段数码管g" )
   END_RUNG
   RUNG wire#w1
      R_Coil( "2号梯七段数码管h" )
   END_RUNG
   RUNG wire#w1
      R_Coil( "2号梯七段数码管i" )
   END_RUNG
   RUNG wire#w1
      R_Coil( "2号梯七段数码管j" )
   END_RUNG
   RUNG wire#w1
      R_Coil( "2号梯七段数码管k" )
   END_RUNG
   RUNG wire#w1
      R_Coil( "2号梯七段数码管l" )
   END_RUNG
   RUNG wire#w1
      R_Coil( "2号梯七段数码管m" )
   END_RUNG
   RUNG wire#w1
      R_Coil( "2号梯七段数码管n" )
   END_RUNG
   RUNG wire#powerrail
      { S7_Templates := "SrcType := Int" } EQ_Contact(in1 := "2号梯当前楼层数", in2 := 2)
      wire#w2
      S_Coil( "2号梯七段数码管a" )
   END_RUNG
   RUNG wire#w2
      S_Coil( "2号梯七段数码管b" )
   END_RUNG
   RUNG wire#w2
      R_Coil( "2号梯七段数码管c" )
   END_RUNG
   RUNG wire#w2
      S_Coil( "2号梯七段数码管d" )
   END_RUNG
   RUNG wire#w2
      S_Coil( "2号梯七段数码管e" )
   END_RUNG
   RUNG wire#w2
      R_Coil( "2号梯七段数码管f" )
   END_RUNG
   RUNG wire#w2
      S_Coil( "2号梯七段数码管g" )
   END_RUNG
   RUNG wire#w2
      R_Coil( "2号梯七段数码管h" )
   END_RUNG
   RUNG wire#w2
      R_Coil( "2号梯七段数码管i" )
   END_RUNG
   RUNG wire#w2
      R_Coil( "2号梯七段数码管j" )
   END_RUNG
   RUNG wire#w2
      R_Coil( "2号梯七段数码管k" )
   END_RUNG
   RUNG wire#w2
      R_Coil( "2号梯七段数码管l" )
   END_RUNG
   RUNG wire#w2
      R_Coil( "2号梯七段数码管m" )
   END_RUNG
   RUNG wire#w2
      R_Coil( "2号梯七段数码管n" )
   END_RUNG
   RUNG wire#powerrail
      { S7_Templates := "SrcType := Int" } EQ_Contact(in1 := "2号梯当前楼层数", in2 := 3)
      wire#w3
      S_Coil( "2号梯七段数码管a" )
   END_RUNG
   RUNG wire#w3
      S_Coil( "2号梯七段数码管b" )
   END_RUNG
   RUNG wire#w3
      S_Coil( "2号梯七段数码管c" )
   END_RUNG
   RUNG wire#w3
      S_Coil( "2号梯七段数码管d" )
   END_RUNG
   RUNG wire#w3
      R_Coil( "2号梯七段数码管e" )
   END_RUNG
   RUNG wire#w3
      R_Coil( "2号梯七段数码管f" )
   END_RUNG
   RUNG wire#w3
      S_Coil( "2号梯七段数码管g" )
   END_RUNG
   RUNG wire#w3
      R_Coil( "2号梯七段数码管h" )
   END_RUNG
   RUNG wire#w3
      R_Coil( "2号梯七段数码管i" )
   END_RUNG
   RUNG wire#w3
      R_Coil( "2号梯七段数码管j" )
   END_RUNG
   RUNG wire#w3
      R_Coil( "2号梯七段数码管k" )
   END_RUNG
   RUNG wire#w3
      R_Coil( "2号梯七段数码管l" )
   END_RUNG
   RUNG wire#w3
      R_Coil( "2号梯七段数码管m" )
   END_RUNG
   RUNG wire#w3
      R_Coil( "2号梯七段数码管n" )
   END_RUNG
   RUNG wire#powerrail
      { S7_Templates := "SrcType := Int" } EQ_Contact(in1 := "2号梯当前楼层数", in2 := 4)
      wire#w4
      R_Coil( "2号梯七段数码管a" )
   END_RUNG
   RUNG wire#w4
      S_Coil( "2号梯七段数码管b" )
   END_RUNG
   RUNG wire#w4
      S_Coil( "2号梯七段数码管c" )
   END_RUNG
   RUNG wire#w4
      R_Coil( "2号梯七段数码管d" )
   END_RUNG
   RUNG wire#w4
      R_Coil( "2号梯七段数码管e" )
   END_RUNG
   RUNG wire#w4
      S_Coil( "2号梯七段数码管f" )
   END_RUNG
   RUNG wire#w4
      S_Coil( "2号梯七段数码管g" )
   END_RUNG
   RUNG wire#w4
      R_Coil( "2号梯七段数码管h" )
   END_RUNG
   RUNG wire#w4
      R_Coil( "2号梯七段数码管i" )
   END_RUNG
   RUNG wire#w4
      R_Coil( "2号梯七段数码管j" )
   END_RUNG
   RUNG wire#w4
      R_Coil( "2号梯七段数码管k" )
   END_RUNG
   RUNG wire#w4
      R_Coil( "2号梯七段数码管l" )
   END_RUNG
   RUNG wire#w4
      R_Coil( "2号梯七段数码管m" )
   END_RUNG
   RUNG wire#w4
      R_Coil( "2号梯七段数码管n" )
   END_RUNG
   RUNG wire#powerrail
      { S7_Templates := "SrcType := Int" } EQ_Contact(in1 := "2号梯当前楼层数", in2 := 5)
      wire#w5
      S_Coil( "2号梯七段数码管a" )
   END_RUNG
   RUNG wire#w5
      R_Coil( "2号梯七段数码管b" )
   END_RUNG
   RUNG wire#w5
      S_Coil( "2号梯七段数码管c" )
   END_RUNG
   RUNG wire#w5
      S_Coil( "2号梯七段数码管d" )
   END_RUNG
   RUNG wire#w5
      R_Coil( "2号梯七段数码管e" )
   END_RUNG
   RUNG wire#w5
      S_Coil( "2号梯七段数码管f" )
   END_RUNG
   RUNG wire#w5
      S_Coil( "2号梯七段数码管g" )
   END_RUNG
   RUNG wire#w5
      R_Coil( "2号梯七段数码管h" )
   END_RUNG
   RUNG wire#w5
      R_Coil( "2号梯七段数码管i" )
   END_RUNG
   RUNG wire#w5
      R_Coil( "2号梯七段数码管j" )
   END_RUNG
   RUNG wire#w5
      R_Coil( "2号梯七段数码管k" )
   END_RUNG
   RUNG wire#w5
      R_Coil( "2号梯七段数码管l" )
   END_RUNG
   RUNG wire#w5
      R_Coil( "2号梯七段数码管m" )
   END_RUNG
   RUNG wire#w5
      R_Coil( "2号梯七段数码管n" )
   END_RUNG
   RUNG wire#powerrail
      { S7_Templates := "SrcType := Int" } EQ_Contact(in1 := "2号梯当前楼层数", in2 := 6)
      wire#w6
      S_Coil( "2号梯七段数码管a" )
   END_RUNG
   RUNG wire#w6
      R_Coil( "2号梯七段数码管b" )
   END_RUNG
   RUNG wire#w6
      S_Coil( "2号梯七段数码管c" )
   END_RUNG
   RUNG wire#w6
      S_Coil( "2号梯七段数码管d" )
   END_RUNG
   RUNG wire#w6
      S_Coil( "2号梯七段数码管e" )
   END_RUNG
   RUNG wire#w6
      S_Coil( "2号梯七段数码管f" )
   END_RUNG
   RUNG wire#w6
      S_Coil( "2号梯七段数码管g" )
   END_RUNG
   RUNG wire#w6
      R_Coil( "2号梯七段数码管h" )
   END_RUNG
   RUNG wire#w6
      R_Coil( "2号梯七段数码管i" )
   END_RUNG
   RUNG wire#w6
      R_Coil( "2号梯七段数码管j" )
   END_RUNG
   RUNG wire#w6
      R_Coil( "2号梯七段数码管k" )
   END_RUNG
   RUNG wire#w6
      R_Coil( "2号梯七段数码管l" )
   END_RUNG
   RUNG wire#w6
      R_Coil( "2号梯七段数码管m" )
   END_RUNG
   RUNG wire#w6
      R_Coil( "2号梯七段数码管n" )
   END_RUNG
   RUNG wire#powerrail
      { S7_Templates := "SrcType := Int" } EQ_Contact(in1 := "2号梯当前楼层数", in2 := 7)
      wire#w7
      S_Coil( "2号梯七段数码管a" )
   END_RUNG
   RUNG wire#w7
      S_Coil( "2号梯七段数码管b" )
   END_RUNG
   RUNG wire#w7
      S_Coil( "2号梯七段数码管c" )
   END_RUNG
   RUNG wire#w7
      R_Coil( "2号梯七段数码管d" )
   END_RUNG
   RUNG wire#w7
      R_Coil( "2号梯七段数码管e" )
   END_RUNG
   RUNG wire#w7
      R_Coil( "2号梯七段数码管f" )
   END_RUNG
   RUNG wire#w7
      R_Coil( "2号梯七段数码管g" )
   END_RUNG
   RUNG wire#w7
      R_Coil( "2号梯七段数码管h" )
   END_RUNG
   RUNG wire#w7
      R_Coil( "2号梯七段数码管i" )
   END_RUNG
   RUNG wire#w7
      R_Coil( "2号梯七段数码管j" )
   END_RUNG
   RUNG wire#w7
      R_Coil( "2号梯七段数码管k" )
   END_RUNG
   RUNG wire#w7
      R_Coil( "2号梯七段数码管l" )
   END_RUNG
   RUNG wire#w7
      R_Coil( "2号梯七段数码管m" )
   END_RUNG
   RUNG wire#w7
      R_Coil( "2号梯七段数码管n" )
   END_RUNG
   RUNG wire#powerrail
      { S7_Templates := "SrcType := Int" } EQ_Contact(in1 := "2号梯当前楼层数", in2 := 8)
      wire#w8
      S_Coil( "2号梯七段数码管a" )
   END_RUNG
   RUNG wire#w8
      S_Coil( "2号梯七段数码管b" )
   END_RUNG
   RUNG wire#w8
      S_Coil( "2号梯七段数码管c" )
   END_RUNG
   RUNG wire#w8
      S_Coil( "2号梯七段数码管d" )
   END_RUNG
   RUNG wire#w8
      S_Coil( "2号梯七段数码管e" )
   END_RUNG
   RUNG wire#w8
      S_Coil( "2号梯七段数码管f" )
   END_RUNG
   RUNG wire#w8
      S_Coil( "2号梯七段数码管g" )
   END_RUNG
   RUNG wire#w8
      R_Coil( "2号梯七段数码管h" )
   END_RUNG
   RUNG wire#w8
      R_Coil( "2号梯七段数码管i" )
   END_RUNG
   RUNG wire#w8
      R_Coil( "2号梯七段数码管j" )
   END_RUNG
   RUNG wire#w8
      R_Coil( "2号梯七段数码管k" )
   END_RUNG
   RUNG wire#w8
      R_Coil( "2号梯七段数码管l" )
   END_RUNG
   RUNG wire#w8
      R_Coil( "2号梯七段数码管m" )
   END_RUNG
   RUNG wire#w8
      R_Coil( "2号梯七段数码管n" )
   END_RUNG
   RUNG wire#powerrail
      { S7_Templates := "SrcType := Int" } EQ_Contact(in1 := "2号梯当前楼层数", in2 := 9)
      wire#w9
      S_Coil( "2号梯七段数码管a" )
   END_RUNG
   RUNG wire#w9
      S_Coil( "2号梯七段数码管b" )
   END_RUNG
   RUNG wire#w9
      S_Coil( "2号梯七段数码管c" )
   END_RUNG
   RUNG wire#w9
      S_Coil( "2号梯七段数码管d" )
   END_RUNG
   RUNG wire#w9
      R_Coil( "2号梯七段数码管e" )
   END_RUNG
   RUNG wire#w9
      S_Coil( "2号梯七段数码管f" )
   END_RUNG
   RUNG wire#w9
      S_Coil( "2号梯七段数码管g" )
   END_RUNG
   RUNG wire#w9
      R_Coil( "2号梯七段数码管h" )
   END_RUNG
   RUNG wire#w9
      R_Coil( "2号梯七段数码管i" )
   END_RUNG
   RUNG wire#w9
      R_Coil( "2号梯七段数码管j" )
   END_RUNG
   RUNG wire#w9
      R_Coil( "2号梯七段数码管k" )
   END_RUNG
   RUNG wire#w9
      R_Coil( "2号梯七段数码管l" )
   END_RUNG
   RUNG wire#w9
      R_Coil( "2号梯七段数码管m" )
   END_RUNG
   RUNG wire#w9
      R_Coil( "2号梯七段数码管n" )
   END_RUNG
   RUNG wire#powerrail
      { S7_Templates := "SrcType := Int" } EQ_Contact(in1 := "2号梯当前楼层数", in2 := 10)
      wire#w10
      S_Coil( "2号梯七段数码管a" )
   END_RUNG
   RUNG wire#w10
      S_Coil( "2号梯七段数码管b" )
   END_RUNG
   RUNG wire#w10
      S_Coil( "2号梯七段数码管c" )
   END_RUNG
   RUNG wire#w10
      S_Coil( "2号梯七段数码管d" )
   END_RUNG
   RUNG wire#w10
      S_Coil( "2号梯七段数码管e" )
   END_RUNG
   RUNG wire#w10
      S_Coil( "2号梯七段数码管f" )
   END_RUNG
   RUNG wire#w10
      R_Coil( "2号梯七段数码管g" )
   END_RUNG
   RUNG wire#w10
      R_Coil( "2号梯七段数码管h" )
   END_RUNG
   RUNG wire#w10
      S_Coil( "2号梯七段数码管i" )
   END_RUNG
   RUNG wire#w10
      S_Coil( "2号梯七段数码管j" )
   END_RUNG
   RUNG wire#w10
      R_Coil( "2号梯七段数码管k" )
   END_RUNG
   RUNG wire#w10
      R_Coil( "2号梯七段数码管l" )
   END_RUNG
   RUNG wire#w10
      R_Coil( "2号梯七段数码管m" )
   END_RUNG
   RUNG wire#w10
      R_Coil( "2号梯七段数码管n" )
   END_RUNG
   // the same network as SCL:
   IF "2号梯当前楼层数" = 1 THEN
       "2号梯七段数码管a" := FALSE;
       "2号梯七段数码管b" := TRUE;
       "2号梯七段数码管c" := TRUE;
       "2号梯七段数码管d" := FALSE;
       "2号梯七段数码管e" := FALSE;
       "2号梯七段数码管f" := FALSE;
       "2号梯七段数码管g" := FALSE;
       "2号梯七段数码管h" := FALSE;
       "2号梯七段数码管i" := FALSE;
       "2号梯七段数码管j" := FALSE;
       "2号梯七段数码管k" := FALSE;
       "2号梯七段数码管l" := FALSE;
       "2号梯七段数码管m" := FALSE;
       "2号梯七段数码管n" := FALSE;
   END_IF;
   IF "2号梯当前楼层数" = 2 THEN
       "2号梯七段数码管a" := TRUE;
       "2号梯七段数码管b" := TRUE;
       "2号梯七段数码管c" := FALSE;
       "2号梯七段数码管d" := TRUE;
       "2号梯七段数码管e" := TRUE;
       "2号梯七段数码管f" := FALSE;
       "2号梯七段数码管g" := TRUE;
       "2号梯七段数码管h" := FALSE;
       "2号梯七段数码管i" := FALSE;
       "2号梯七段数码管j" := FALSE;
       "2号梯七段数码管k" := FALSE;
       "2号梯七段数码管l" := FALSE;
       "2号梯七段数码管m" := FALSE;
       "2号梯七段数码管n" := FALSE;
   END_IF;
   IF "2号梯当前楼层数" = 3 THEN
       "2号梯七段数码管a" := TRUE;
       "2号梯七段数码管b" := TRUE;
       "2号梯七段数码管c" := TRUE;
       "2号梯七段数码管d" := TRUE;
       "2号梯七段数码管e" := FALSE;
       "2号梯七段数码管f" := FALSE;
       "2号梯七段数码管g" := TRUE;
       "2号梯七段数码管h" := FALSE;
       "2号梯七段数码管i" := FALSE;
       "2号梯七段数码管j" := FALSE;
       "2号梯七段数码管k" := FALSE;
       "2号梯七段数码管l" := FALSE;
       "2号梯七段数码管m" := FALSE;
       "2号梯七段数码管n" := FALSE;
   END_IF;
   IF "2号梯当前楼层数" = 4 THEN
       "2号梯七段数码管a" := FALSE;
       "2号梯七段数码管b" := TRUE;
       "2号梯七段数码管c" := TRUE;
       "2号梯七段数码管d" := FALSE;
       "2号梯七段数码管e" := FALSE;
       "2号梯七段数码管f" := TRUE;
       "2号梯七段数码管g" := TRUE;
       "2号梯七段数码管h" := FALSE;
       "2号梯七段数码管i" := FALSE;
       "2号梯七段数码管j" := FALSE;
       "2号梯七段数码管k" := FALSE;
       "2号梯七段数码管l" := FALSE;
       "2号梯七段数码管m" := FALSE;
       "2号梯七段数码管n" := FALSE;
   END_IF;
   IF "2号梯当前楼层数" = 5 THEN
       "2号梯七段数码管a" := TRUE;
       "2号梯七段数码管b" := FALSE;
       "2号梯七段数码管c" := TRUE;
       "2号梯七段数码管d" := TRUE;
       "2号梯七段数码管e" := FALSE;
       "2号梯七段数码管f" := TRUE;
       "2号梯七段数码管g" := TRUE;
       "2号梯七段数码管h" := FALSE;
       "2号梯七段数码管i" := FALSE;
       "2号梯七段数码管j" := FALSE;
       "2号梯七段数码管k" := FALSE;
       "2号梯七段数码管l" := FALSE;
       "2号梯七段数码管m" := FALSE;
       "2号梯七段数码管n" := FALSE;
   END_IF;
   IF "2号梯当前楼层数" = 6 THEN
       "2号梯七段数码管a" := TRUE;
       "2号梯七段数码管b" := FALSE;
       "2号梯七段数码管c" := TRUE;
       "2号梯七段数码管d" := TRUE;
       "2号梯七段数码管e" := TRUE;
       "2号梯七段数码管f" := TRUE;
       "2号梯七段数码管g" := TRUE;
       "2号梯七段数码管h" := FALSE;
       "2号梯七段数码管i" := FALSE;
       "2号梯七段数码管j" := FALSE;
       "2号梯七段数码管k" := FALSE;
       "2号梯七段数码管l" := FALSE;
       "2号梯七段数码管m" := FALSE;
       "2号梯七段数码管n" := FALSE;
   END_IF;
   IF "2号梯当前楼层数" = 7 THEN
       "2号梯七段数码管a" := TRUE;
       "2号梯七段数码管b" := TRUE;
       "2号梯七段数码管c" := TRUE;
       "2号梯七段数码管d" := FALSE;
       "2号梯七段数码管e" := FALSE;
       "2号梯七段数码管f" := FALSE;
       "2号梯七段数码管g" := FALSE;
       "2号梯七段数码管h" := FALSE;
       "2号梯七段数码管i" := FALSE;
       "2号梯七段数码管j" := FALSE;
       "2号梯七段数码管k" := FALSE;
       "2号梯七段数码管l" := FALSE;
       "2号梯七段数码管m" := FALSE;
       "2号梯七段数码管n" := FALSE;
   END_IF;
   IF "2号梯当前楼层数" = 8 THEN
       "2号梯七段数码管a" := TRUE;
       "2号梯七段数码管b" := TRUE;
       "2号梯七段数码管c" := TRUE;
       "2号梯七段数码管d" := TRUE;
       "2号梯七段数码管e" := TRUE;
       "2号梯七段数码管f" := TRUE;
       "2号梯七段数码管g" := TRUE;
       "2号梯七段数码管h" := FALSE;
       "2号梯七段数码管i" := FALSE;
       "2号梯七段数码管j" := FALSE;
       "2号梯七段数码管k" := FALSE;
       "2号梯七段数码管l" := FALSE;
       "2号梯七段数码管m" := FALSE;
       "2号梯七段数码管n" := FALSE;
   END_IF;
   IF "2号梯当前楼层数" = 9 THEN
       "2号梯七段数码管a" := TRUE;
       "2号梯七段数码管b" := TRUE;
       "2号梯七段数码管c" := TRUE;
       "2号梯七段数码管d" := TRUE;
       "2号梯七段数码管e" := FALSE;
       "2号梯七段数码管f" := TRUE;
       "2号梯七段数码管g" := TRUE;
       "2号梯七段数码管h" := FALSE;
       "2号梯七段数码管i" := FALSE;
       "2号梯七段数码管j" := FALSE;
       "2号梯七段数码管k" := FALSE;
       "2号梯七段数码管l" := FALSE;
       "2号梯七段数码管m" := FALSE;
       "2号梯七段数码管n" := FALSE;
   END_IF;
   IF "2号梯当前楼层数" = 10 THEN
       "2号梯七段数码管a" := TRUE;
       "2号梯七段数码管b" := TRUE;
       "2号梯七段数码管c" := TRUE;
       "2号梯七段数码管d" := TRUE;
       "2号梯七段数码管e" := TRUE;
       "2号梯七段数码管f" := TRUE;
       "2号梯七段数码管g" := FALSE;
       "2号梯七段数码管h" := FALSE;
       "2号梯七段数码管i" := TRUE;
       "2号梯七段数码管j" := TRUE;
       "2号梯七段数码管k" := FALSE;
       "2号梯七段数码管l" := FALSE;
       "2号梯七段数码管m" := FALSE;
       "2号梯七段数码管n" := FALSE;
   END_IF;
END_REGION

REGION Network 2: 上下行指示灯
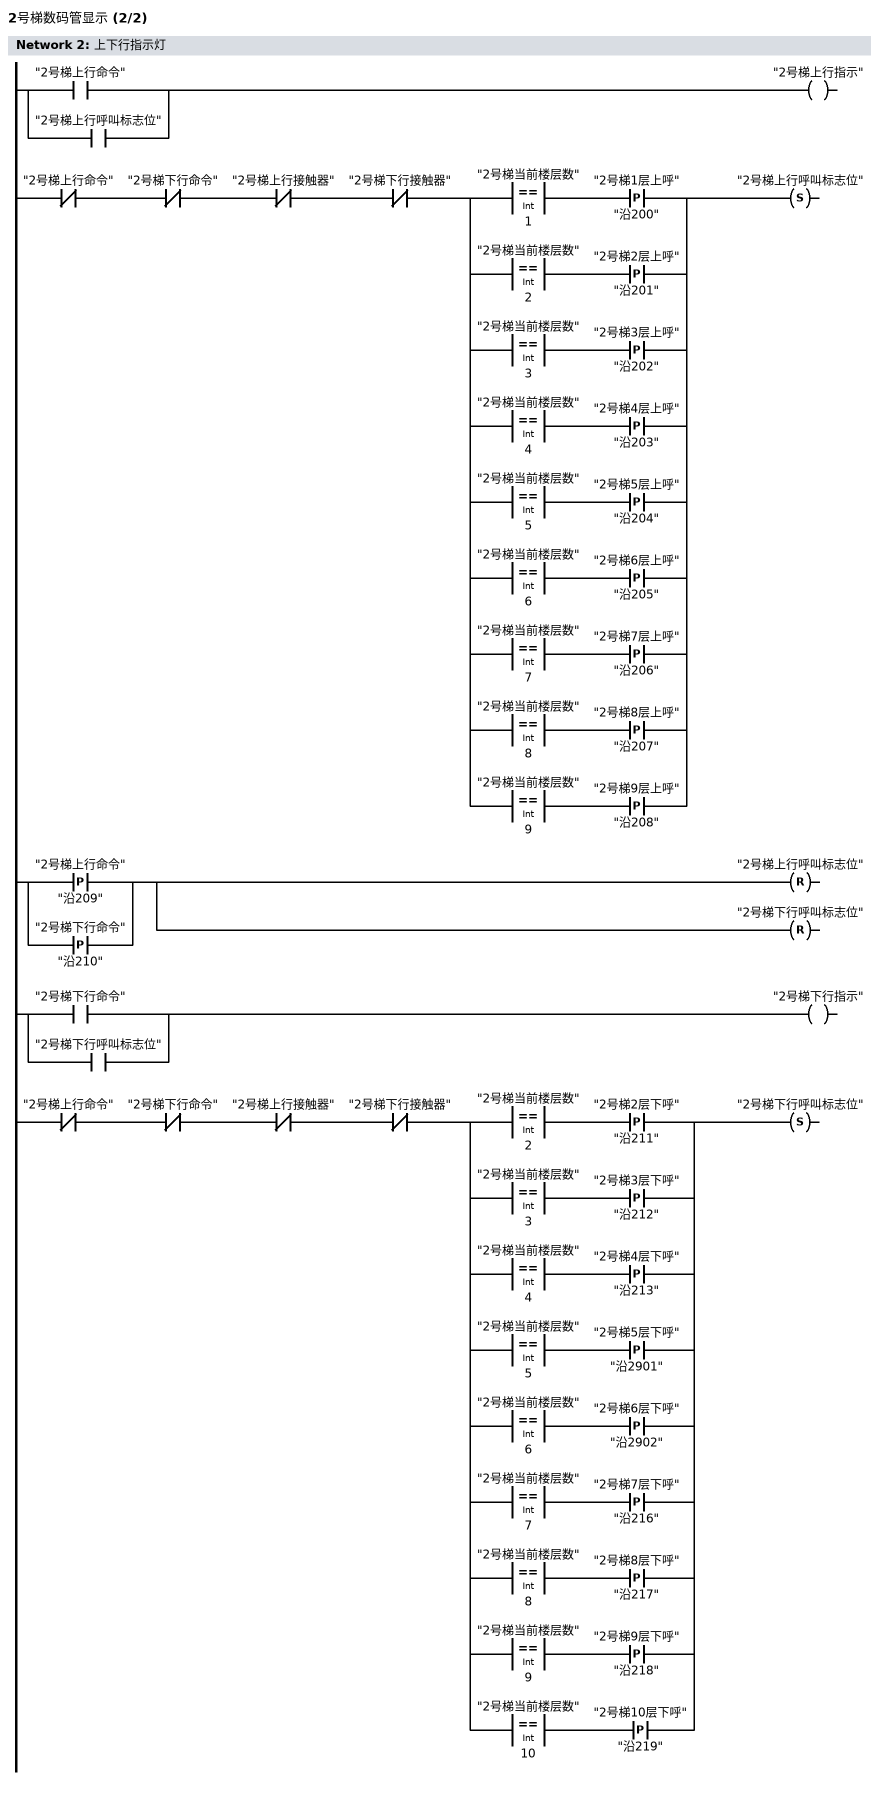
   RUNG wire#powerrail
      Contact( "2号梯上行命令" )
      wire#w1
      Coil( "2号梯上行指示" )
   END_RUNG
   RUNG wire#powerrail
      Contact( "2号梯上行呼叫标志位" )
   END_RUNG wire#w1
   RUNG wire#powerrail
      I_Contact( "2号梯上行命令" )
      I_Contact( "2号梯下行命令" )
      I_Contact( "2号梯上行接触器" )
      I_Contact( "2号梯下行接触器" )
      wire#w2
      { S7_Templates := "SrcType := Int" } EQ_Contact(in1 := "2号梯当前楼层数", in2 := 1)
      P_Contact(operand := "2号梯1层上呼", bit := "沿200")
      wire#w3
      S_Coil( "2号梯上行呼叫标志位" )
   END_RUNG
   RUNG wire#w2
      { S7_Templates := "SrcType := Int" } EQ_Contact(in1 := "2号梯当前楼层数", in2 := 2)
      P_Contact(operand := "2号梯2层上呼", bit := "沿201")
   END_RUNG wire#w3
   RUNG wire#w2
      { S7_Templates := "SrcType := Int" } EQ_Contact(in1 := "2号梯当前楼层数", in2 := 3)
      P_Contact(operand := "2号梯3层上呼", bit := "沿202")
   END_RUNG wire#w3
   RUNG wire#w2
      { S7_Templates := "SrcType := Int" } EQ_Contact(in1 := "2号梯当前楼层数", in2 := 4)
      P_Contact(operand := "2号梯4层上呼", bit := "沿203")
   END_RUNG wire#w3
   RUNG wire#w2
      { S7_Templates := "SrcType := Int" } EQ_Contact(in1 := "2号梯当前楼层数", in2 := 5)
      P_Contact(operand := "2号梯5层上呼", bit := "沿204")
   END_RUNG wire#w3
   RUNG wire#w2
      { S7_Templates := "SrcType := Int" } EQ_Contact(in1 := "2号梯当前楼层数", in2 := 6)
      P_Contact(operand := "2号梯6层上呼", bit := "沿205")
   END_RUNG wire#w3
   RUNG wire#w2
      { S7_Templates := "SrcType := Int" } EQ_Contact(in1 := "2号梯当前楼层数", in2 := 7)
      P_Contact(operand := "2号梯7层上呼", bit := "沿206")
   END_RUNG wire#w3
   RUNG wire#w2
      { S7_Templates := "SrcType := Int" } EQ_Contact(in1 := "2号梯当前楼层数", in2 := 8)
      P_Contact(operand := "2号梯8层上呼", bit := "沿207")
   END_RUNG wire#w3
   RUNG wire#w2
      { S7_Templates := "SrcType := Int" } EQ_Contact(in1 := "2号梯当前楼层数", in2 := 9)
      P_Contact(operand := "2号梯9层上呼", bit := "沿208")
   END_RUNG wire#w3
   RUNG wire#powerrail
      P_Contact(operand := "2号梯上行命令", bit := "沿209")
      wire#w4
      R_Coil( "2号梯上行呼叫标志位" )
   END_RUNG
   RUNG wire#powerrail
      P_Contact(operand := "2号梯下行命令", bit := "沿210")
   END_RUNG wire#w4
   RUNG wire#w4
      R_Coil( "2号梯下行呼叫标志位" )
   END_RUNG
   RUNG wire#powerrail
      Contact( "2号梯下行命令" )
      wire#w5
      Coil( "2号梯下行指示" )
   END_RUNG
   RUNG wire#powerrail
      Contact( "2号梯下行呼叫标志位" )
   END_RUNG wire#w5
   RUNG wire#powerrail
      I_Contact( "2号梯上行命令" )
      I_Contact( "2号梯下行命令" )
      I_Contact( "2号梯上行接触器" )
      I_Contact( "2号梯下行接触器" )
      wire#w6
      { S7_Templates := "SrcType := Int" } EQ_Contact(in1 := "2号梯当前楼层数", in2 := 2)
      P_Contact(operand := "2号梯2层下呼", bit := "沿211")
      wire#w7
      S_Coil( "2号梯下行呼叫标志位" )
   END_RUNG
   RUNG wire#w6
      { S7_Templates := "SrcType := Int" } EQ_Contact(in1 := "2号梯当前楼层数", in2 := 3)
      P_Contact(operand := "2号梯3层下呼", bit := "沿212")
   END_RUNG wire#w7
   RUNG wire#w6
      { S7_Templates := "SrcType := Int" } EQ_Contact(in1 := "2号梯当前楼层数", in2 := 4)
      P_Contact(operand := "2号梯4层下呼", bit := "沿213")
   END_RUNG wire#w7
   RUNG wire#w6
      { S7_Templates := "SrcType := Int" } EQ_Contact(in1 := "2号梯当前楼层数", in2 := 5)
      P_Contact(operand := "2号梯5层下呼", bit := "沿2901")
   END_RUNG wire#w7
   RUNG wire#w6
      { S7_Templates := "SrcType := Int" } EQ_Contact(in1 := "2号梯当前楼层数", in2 := 6)
      P_Contact(operand := "2号梯6层下呼", bit := "沿2902")
   END_RUNG wire#w7
   RUNG wire#w6
      { S7_Templates := "SrcType := Int" } EQ_Contact(in1 := "2号梯当前楼层数", in2 := 7)
      P_Contact(operand := "2号梯7层下呼", bit := "沿216")
   END_RUNG wire#w7
   RUNG wire#w6
      { S7_Templates := "SrcType := Int" } EQ_Contact(in1 := "2号梯当前楼层数", in2 := 8)
      P_Contact(operand := "2号梯8层下呼", bit := "沿217")
   END_RUNG wire#w7
   RUNG wire#w6
      { S7_Templates := "SrcType := Int" } EQ_Contact(in1 := "2号梯当前楼层数", in2 := 9)
      P_Contact(operand := "2号梯9层下呼", bit := "沿218")
   END_RUNG wire#w7
   RUNG wire#w6
      { S7_Templates := "SrcType := Int" } EQ_Contact(in1 := "2号梯当前楼层数", in2 := 10)
      P_Contact(operand := "2号梯10层下呼", bit := "沿219")
   END_RUNG wire#w7
   // the same network as SCL:
   "2号梯上行指示" := "2号梯上行命令" OR "2号梯上行呼叫标志位";
   #_w1 := NOT "2号梯上行命令" AND NOT "2号梯下行命令" AND NOT "2号梯上行接触器" AND NOT "2号梯下行接触器" AND ("2号梯当前楼层数" = 1) AND "2号梯1层上呼" AND NOT "沿200";   // rising edge of "2号梯1层上呼"
   "沿200" := "2号梯1层上呼";
   #_w2 := NOT "2号梯上行命令" AND NOT "2号梯下行命令" AND NOT "2号梯上行接触器" AND NOT "2号梯下行接触器" AND ("2号梯当前楼层数" = 2) AND "2号梯2层上呼" AND NOT "沿201";   // rising edge of "2号梯2层上呼"
   "沿201" := "2号梯2层上呼";
   #_w3 := NOT "2号梯上行命令" AND NOT "2号梯下行命令" AND NOT "2号梯上行接触器" AND NOT "2号梯下行接触器" AND ("2号梯当前楼层数" = 3) AND "2号梯3层上呼" AND NOT "沿202";   // rising edge of "2号梯3层上呼"
   "沿202" := "2号梯3层上呼";
   #_w4 := NOT "2号梯上行命令" AND NOT "2号梯下行命令" AND NOT "2号梯上行接触器" AND NOT "2号梯下行接触器" AND ("2号梯当前楼层数" = 4) AND "2号梯4层上呼" AND NOT "沿203";   // rising edge of "2号梯4层上呼"
   "沿203" := "2号梯4层上呼";
   #_w5 := NOT "2号梯上行命令" AND NOT "2号梯下行命令" AND NOT "2号梯上行接触器" AND NOT "2号梯下行接触器" AND ("2号梯当前楼层数" = 5) AND "2号梯5层上呼" AND NOT "沿204";   // rising edge of "2号梯5层上呼"
   "沿204" := "2号梯5层上呼";
   #_w6 := NOT "2号梯上行命令" AND NOT "2号梯下行命令" AND NOT "2号梯上行接触器" AND NOT "2号梯下行接触器" AND ("2号梯当前楼层数" = 6) AND "2号梯6层上呼" AND NOT "沿205";   // rising edge of "2号梯6层上呼"
   "沿205" := "2号梯6层上呼";
   #_w7 := NOT "2号梯上行命令" AND NOT "2号梯下行命令" AND NOT "2号梯上行接触器" AND NOT "2号梯下行接触器" AND ("2号梯当前楼层数" = 7) AND "2号梯7层上呼" AND NOT "沿206";   // rising edge of "2号梯7层上呼"
   "沿206" := "2号梯7层上呼";
   #_w8 := NOT "2号梯上行命令" AND NOT "2号梯下行命令" AND NOT "2号梯上行接触器" AND NOT "2号梯下行接触器" AND ("2号梯当前楼层数" = 8) AND "2号梯8层上呼" AND NOT "沿207";   // rising edge of "2号梯8层上呼"
   "沿207" := "2号梯8层上呼";
   #_w9 := NOT "2号梯上行命令" AND NOT "2号梯下行命令" AND NOT "2号梯上行接触器" AND NOT "2号梯下行接触器" AND ("2号梯当前楼层数" = 9) AND "2号梯9层上呼" AND NOT "沿208";   // rising edge of "2号梯9层上呼"
   "沿208" := "2号梯9层上呼";
   IF #_w1 OR #_w2 OR #_w3 OR #_w4 OR #_w5 OR #_w6 OR #_w7 OR #_w8 OR #_w9 THEN "2号梯上行呼叫标志位" := TRUE; END_IF;
   #_w10 := "2号梯上行命令" AND NOT "沿209";   // rising edge of "2号梯上行命令"
   "沿209" := "2号梯上行命令";
   #_w11 := "2号梯下行命令" AND NOT "沿210";   // rising edge of "2号梯下行命令"
   "沿210" := "2号梯下行命令";
   IF #_w10 OR #_w11 THEN
       "2号梯上行呼叫标志位" := FALSE;
       "2号梯下行呼叫标志位" := FALSE;
   END_IF;
   "2号梯下行指示" := "2号梯下行命令" OR "2号梯下行呼叫标志位";
   #_w12 := NOT "2号梯上行命令" AND NOT "2号梯下行命令" AND NOT "2号梯上行接触器" AND NOT "2号梯下行接触器" AND ("2号梯当前楼层数" = 2) AND "2号梯2层下呼" AND NOT "沿211";   // rising edge of "2号梯2层下呼"
   "沿211" := "2号梯2层下呼";
   #_w13 := NOT "2号梯上行命令" AND NOT "2号梯下行命令" AND NOT "2号梯上行接触器" AND NOT "2号梯下行接触器" AND ("2号梯当前楼层数" = 3) AND "2号梯3层下呼" AND NOT "沿212";   // rising edge of "2号梯3层下呼"
   "沿212" := "2号梯3层下呼";
   #_w14 := NOT "2号梯上行命令" AND NOT "2号梯下行命令" AND NOT "2号梯上行接触器" AND NOT "2号梯下行接触器" AND ("2号梯当前楼层数" = 4) AND "2号梯4层下呼" AND NOT "沿213";   // rising edge of "2号梯4层下呼"
   "沿213" := "2号梯4层下呼";
   #_w15 := NOT "2号梯上行命令" AND NOT "2号梯下行命令" AND NOT "2号梯上行接触器" AND NOT "2号梯下行接触器" AND ("2号梯当前楼层数" = 5) AND "2号梯5层下呼" AND NOT "沿2901";   // rising edge of "2号梯5层下呼"
   "沿2901" := "2号梯5层下呼";
   #_w16 := NOT "2号梯上行命令" AND NOT "2号梯下行命令" AND NOT "2号梯上行接触器" AND NOT "2号梯下行接触器" AND ("2号梯当前楼层数" = 6) AND "2号梯6层下呼" AND NOT "沿2902";   // rising edge of "2号梯6层下呼"
   "沿2902" := "2号梯6层下呼";
   #_w17 := NOT "2号梯上行命令" AND NOT "2号梯下行命令" AND NOT "2号梯上行接触器" AND NOT "2号梯下行接触器" AND ("2号梯当前楼层数" = 7) AND "2号梯7层下呼" AND NOT "沿216";   // rising edge of "2号梯7层下呼"
   "沿216" := "2号梯7层下呼";
   #_w18 := NOT "2号梯上行命令" AND NOT "2号梯下行命令" AND NOT "2号梯上行接触器" AND NOT "2号梯下行接触器" AND ("2号梯当前楼层数" = 8) AND "2号梯8层下呼" AND NOT "沿217";   // rising edge of "2号梯8层下呼"
   "沿217" := "2号梯8层下呼";
   #_w19 := NOT "2号梯上行命令" AND NOT "2号梯下行命令" AND NOT "2号梯上行接触器" AND NOT "2号梯下行接触器" AND ("2号梯当前楼层数" = 9) AND "2号梯9层下呼" AND NOT "沿218";   // rising edge of "2号梯9层下呼"
   "沿218" := "2号梯9层下呼";
   #_w20 := NOT "2号梯上行命令" AND NOT "2号梯下行命令" AND NOT "2号梯上行接触器" AND NOT "2号梯下行接触器" AND ("2号梯当前楼层数" = 10) AND "2号梯10层下呼" AND NOT "沿219";   // rising edge of "2号梯10层下呼"
   "沿219" := "2号梯10层下呼";
   IF #_w12 OR #_w13 OR #_w14 OR #_w15 OR #_w16 OR #_w17 OR #_w18 OR #_w19 OR #_w20 THEN
       "2号梯下行呼叫标志位" := TRUE;
   END_IF;
END_REGION
END_FUNCTION

FUNCTION "1号梯开门信号" : Void   // FC11, LAD
{ S7_Optimized_Access := 'TRUE' }
VERSION : 0.1
BEGIN

REGION Network 1: 本层开门
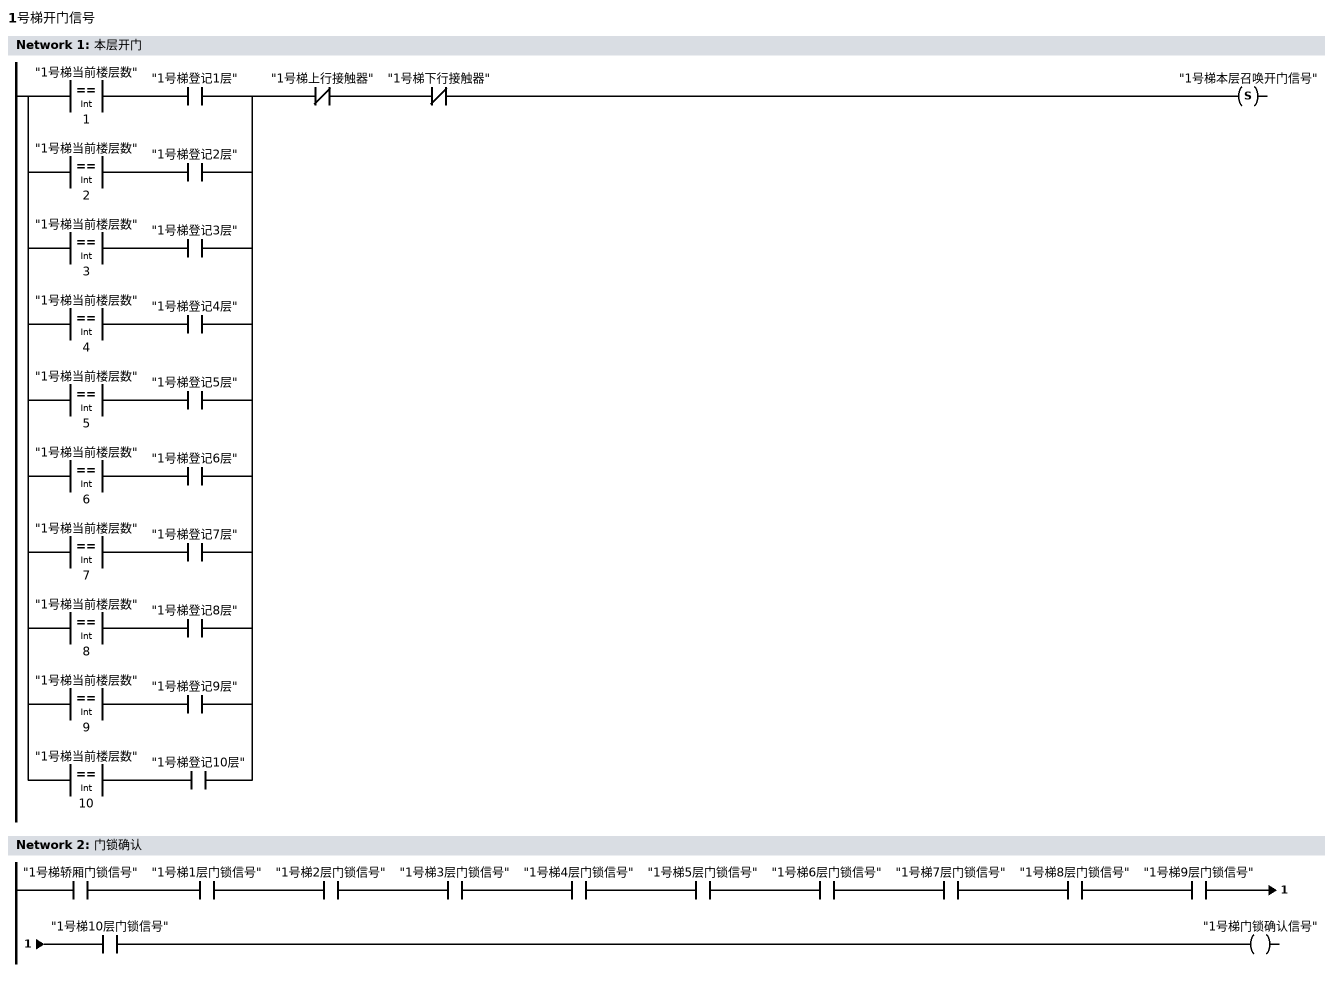
   RUNG wire#powerrail
      { S7_Templates := "SrcType := Int" } EQ_Contact(in1 := "1号梯当前楼层数", in2 := 1)
      Contact( "1号梯登记1层" )
      wire#w1
      I_Contact( "1号梯上行接触器" )
      I_Contact( "1号梯下行接触器" )
      S_Coil( "1号梯本层召唤开门信号" )
   END_RUNG
   RUNG wire#powerrail
      { S7_Templates := "SrcType := Int" } EQ_Contact(in1 := "1号梯当前楼层数", in2 := 2)
      Contact( "1号梯登记2层" )
   END_RUNG wire#w1
   RUNG wire#powerrail
      { S7_Templates := "SrcType := Int" } EQ_Contact(in1 := "1号梯当前楼层数", in2 := 3)
      Contact( "1号梯登记3层" )
   END_RUNG wire#w1
   RUNG wire#powerrail
      { S7_Templates := "SrcType := Int" } EQ_Contact(in1 := "1号梯当前楼层数", in2 := 4)
      Contact( "1号梯登记4层" )
   END_RUNG wire#w1
   RUNG wire#powerrail
      { S7_Templates := "SrcType := Int" } EQ_Contact(in1 := "1号梯当前楼层数", in2 := 5)
      Contact( "1号梯登记5层" )
   END_RUNG wire#w1
   RUNG wire#powerrail
      { S7_Templates := "SrcType := Int" } EQ_Contact(in1 := "1号梯当前楼层数", in2 := 6)
      Contact( "1号梯登记6层" )
   END_RUNG wire#w1
   RUNG wire#powerrail
      { S7_Templates := "SrcType := Int" } EQ_Contact(in1 := "1号梯当前楼层数", in2 := 7)
      Contact( "1号梯登记7层" )
   END_RUNG wire#w1
   RUNG wire#powerrail
      { S7_Templates := "SrcType := Int" } EQ_Contact(in1 := "1号梯当前楼层数", in2 := 8)
      Contact( "1号梯登记8层" )
   END_RUNG wire#w1
   RUNG wire#powerrail
      { S7_Templates := "SrcType := Int" } EQ_Contact(in1 := "1号梯当前楼层数", in2 := 9)
      Contact( "1号梯登记9层" )
   END_RUNG wire#w1
   RUNG wire#powerrail
      { S7_Templates := "SrcType := Int" } EQ_Contact(in1 := "1号梯当前楼层数", in2 := 10)
      Contact( "1号梯登记10层" )
   END_RUNG wire#w1
   // the same network as SCL:
   IF ((("1号梯当前楼层数" = 1) AND "1号梯登记1层") OR (("1号梯当前楼层数" = 2) AND "1号梯登记2层") OR (("1号梯当前楼层数" = 3) AND "1号梯登记3层") OR (("1号梯当前楼层数" = 4) AND "1号梯登记4层") OR (("1号梯当前楼层数" = 5) AND "1号梯登记5层") OR (("1号梯当前楼层数" = 6) AND "1号梯登记6层") OR (("1号梯当前楼层数" = 7) AND "1号梯登记7层") OR (("1号梯当前楼层数" = 8) AND "1号梯登记8层") OR (("1号梯当前楼层数" = 9) AND "1号梯登记9层") OR (("1号梯当前楼层数" = 10) AND "1号梯登记10层")) AND NOT "1号梯上行接触器" AND NOT "1号梯下行接触器" THEN
       "1号梯本层召唤开门信号" := TRUE;
   END_IF;
END_REGION

REGION Network 2: 门锁确认
   RUNG wire#powerrail
      Contact( "1号梯轿厢门锁信号" )
      Contact( "1号梯1层门锁信号" )
      Contact( "1号梯2层门锁信号" )
      Contact( "1号梯3层门锁信号" )
      Contact( "1号梯4层门锁信号" )
      Contact( "1号梯5层门锁信号" )
      Contact( "1号梯6层门锁信号" )
      Contact( "1号梯7层门锁信号" )
      Contact( "1号梯8层门锁信号" )
      Contact( "1号梯9层门锁信号" )
      Contact( "1号梯10层门锁信号" )
      Coil( "1号梯门锁确认信号" )
   END_RUNG
   // the same network as SCL:
   "1号梯门锁确认信号" := "1号梯轿厢门锁信号" AND "1号梯1层门锁信号" AND "1号梯2层门锁信号" AND "1号梯3层门锁信号" AND "1号梯4层门锁信号" AND "1号梯5层门锁信号" AND "1号梯6层门锁信号" AND "1号梯7层门锁信号" AND "1号梯8层门锁信号" AND "1号梯9层门锁信号" AND "1号梯10层门锁信号";
END_REGION
END_FUNCTION

FUNCTION "楼层计数" : Void   // FC12, LAD
{ S7_Optimized_Access := 'TRUE' }
VERSION : 0.1
   VAR_TEMP   // added for the SCL form of the ladder/FBD networks
      _w1 : Bool;
      _w2 : Bool;
      _w3 : Bool;
   END_VAR
BEGIN

REGION Network 1: 上行楼层计数
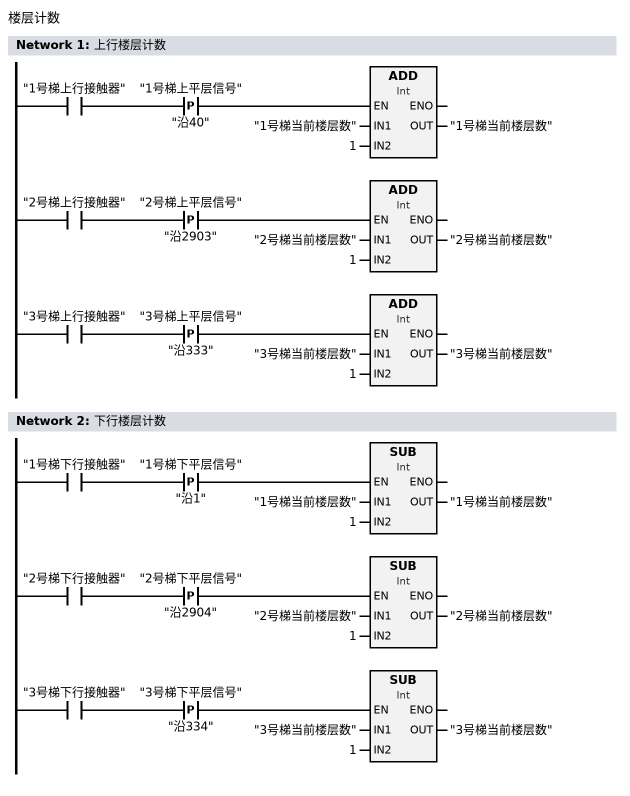
   RUNG wire#powerrail
      Contact( "1号梯上行接触器" )
      P_Contact(operand := "1号梯上平层信号", bit := "沿40")
      { S7_Templates := "SrcType := Int" } Add(in1 := "1号梯当前楼层数", in2 := 1, out => "1号梯当前楼层数")
   END_RUNG
   RUNG wire#powerrail
      Contact( "2号梯上行接触器" )
      P_Contact(operand := "2号梯上平层信号", bit := "沿2903")
      { S7_Templates := "SrcType := Int" } Add(in1 := "2号梯当前楼层数", in2 := 1, out => "2号梯当前楼层数")
   END_RUNG
   RUNG wire#powerrail
      Contact( "3号梯上行接触器" )
      P_Contact(operand := "3号梯上平层信号", bit := "沿333")
      { S7_Templates := "SrcType := Int" } Add(in1 := "3号梯当前楼层数", in2 := 1, out => "3号梯当前楼层数")
   END_RUNG
   // the same network as SCL:
   #_w1 := "1号梯上行接触器" AND "1号梯上平层信号" AND NOT "沿40";   // rising edge of "1号梯上平层信号"
   "沿40" := "1号梯上平层信号";
   IF #_w1 THEN "1号梯当前楼层数" := "1号梯当前楼层数" + 1; END_IF;
   #_w2 := "2号梯上行接触器" AND "2号梯上平层信号" AND NOT "沿2903";   // rising edge of "2号梯上平层信号"
   "沿2903" := "2号梯上平层信号";
   IF #_w2 THEN "2号梯当前楼层数" := "2号梯当前楼层数" + 1; END_IF;
   #_w3 := "3号梯上行接触器" AND "3号梯上平层信号" AND NOT "沿333";   // rising edge of "3号梯上平层信号"
   "沿333" := "3号梯上平层信号";
   IF #_w3 THEN "3号梯当前楼层数" := "3号梯当前楼层数" + 1; END_IF;
END_REGION

REGION Network 2: 下行楼层计数
   RUNG wire#powerrail
      Contact( "1号梯下行接触器" )
      P_Contact(operand := "1号梯下平层信号", bit := "沿1")
      { S7_Templates := "SrcType := Int" } Sub(in1 := "1号梯当前楼层数", in2 := 1, out => "1号梯当前楼层数")
   END_RUNG
   RUNG wire#powerrail
      Contact( "2号梯下行接触器" )
      P_Contact(operand := "2号梯下平层信号", bit := "沿2904")
      { S7_Templates := "SrcType := Int" } Sub(in1 := "2号梯当前楼层数", in2 := 1, out => "2号梯当前楼层数")
   END_RUNG
   RUNG wire#powerrail
      Contact( "3号梯下行接触器" )
      P_Contact(operand := "3号梯下平层信号", bit := "沿334")
      { S7_Templates := "SrcType := Int" } Sub(in1 := "3号梯当前楼层数", in2 := 1, out => "3号梯当前楼层数")
   END_RUNG
   // the same network as SCL:
   #_w1 := "1号梯下行接触器" AND "1号梯下平层信号" AND NOT "沿1";   // rising edge of "1号梯下平层信号"
   "沿1" := "1号梯下平层信号";
   IF #_w1 THEN "1号梯当前楼层数" := "1号梯当前楼层数" - 1; END_IF;
   #_w2 := "2号梯下行接触器" AND "2号梯下平层信号" AND NOT "沿2904";   // rising edge of "2号梯下平层信号"
   "沿2904" := "2号梯下平层信号";
   IF #_w2 THEN "2号梯当前楼层数" := "2号梯当前楼层数" - 1; END_IF;
   #_w3 := "3号梯下行接触器" AND "3号梯下平层信号" AND NOT "沿334";   // rising edge of "3号梯下平层信号"
   "沿334" := "3号梯下平层信号";
   IF #_w3 THEN "3号梯当前楼层数" := "3号梯当前楼层数" - 1; END_IF;
END_REGION
END_FUNCTION

FUNCTION "1号梯指示灯控制" : Void   // FC13, LAD
{ S7_Optimized_Access := 'TRUE' }
VERSION : 0.1
   VAR_TEMP   // added for the SCL form of the ladder/FBD networks
      _w1 : Bool;
      _w2 : Bool;
      _w3 : Bool;
      _w4 : Bool;
      _w5 : Bool;
      _w6 : Bool;
      _w7 : Bool;
      _w8 : Bool;
      _w9 : Bool;
   END_VAR
BEGIN

REGION Network 1: 1号梯终止下呼
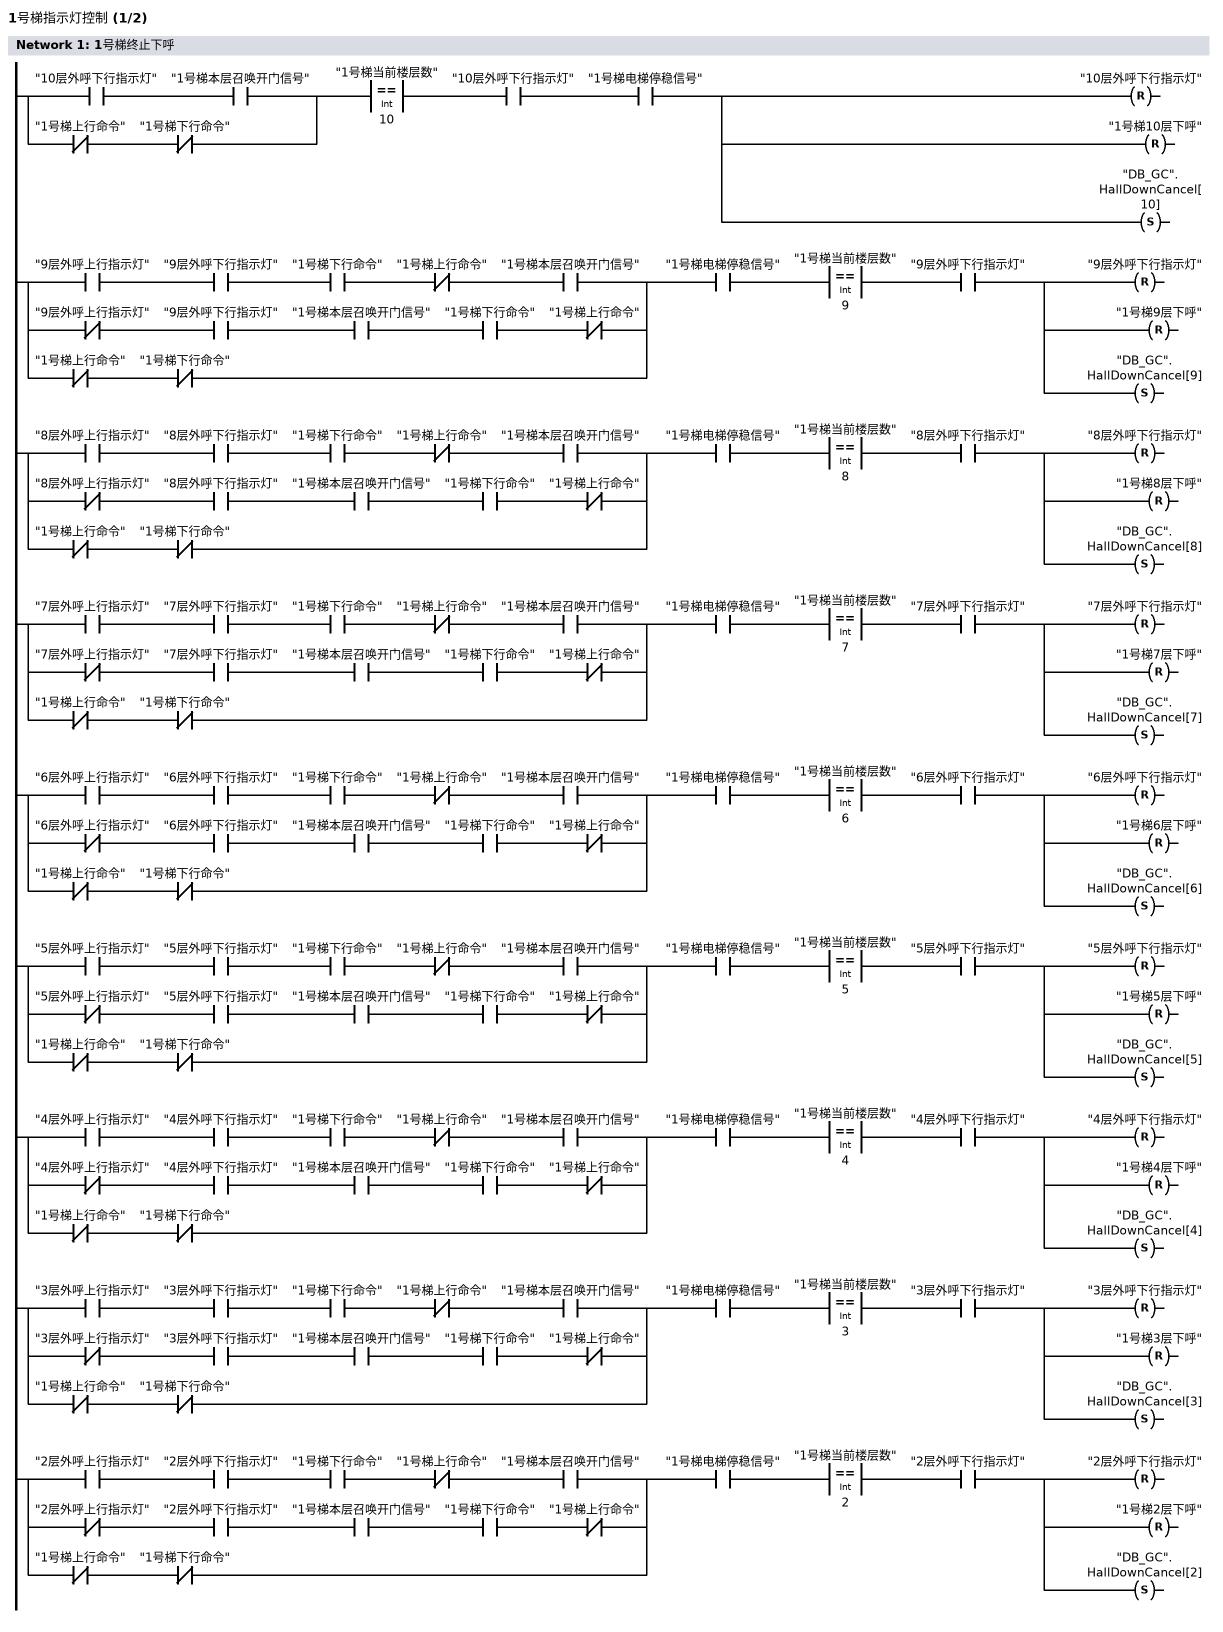
   RUNG wire#powerrail
      Contact( "10层外呼下行指示灯" )
      Contact( "1号梯本层召唤开门信号" )
      wire#w1
      { S7_Templates := "SrcType := Int" } EQ_Contact(in1 := "1号梯当前楼层数", in2 := 10)
      Contact( "10层外呼下行指示灯" )
      Contact( "1号梯电梯停稳信号" )
      wire#w2
      R_Coil( "10层外呼下行指示灯" )
   END_RUNG
   RUNG wire#powerrail
      I_Contact( "1号梯上行命令" )
      I_Contact( "1号梯下行命令" )
   END_RUNG wire#w1
   RUNG wire#w2
      R_Coil( "1号梯10层下呼" )
   END_RUNG
   RUNG wire#w2
      S_Coil( "DB_GC".HallDownCancel[10] )
   END_RUNG
   RUNG wire#powerrail
      Contact( "9层外呼上行指示灯" )
      Contact( "9层外呼下行指示灯" )
      Contact( "1号梯下行命令" )
      I_Contact( "1号梯上行命令" )
      Contact( "1号梯本层召唤开门信号" )
      wire#w3
      Contact( "1号梯电梯停稳信号" )
      { S7_Templates := "SrcType := Int" } EQ_Contact(in1 := "1号梯当前楼层数", in2 := 9)
      Contact( "9层外呼下行指示灯" )
      wire#w4
      R_Coil( "9层外呼下行指示灯" )
   END_RUNG
   RUNG wire#powerrail
      I_Contact( "9层外呼上行指示灯" )
      Contact( "9层外呼下行指示灯" )
      Contact( "1号梯本层召唤开门信号" )
      Contact( "1号梯下行命令" )
      I_Contact( "1号梯上行命令" )
   END_RUNG wire#w3
   RUNG wire#powerrail
      I_Contact( "1号梯上行命令" )
      I_Contact( "1号梯下行命令" )
   END_RUNG wire#w3
   RUNG wire#w4
      R_Coil( "1号梯9层下呼" )
   END_RUNG
   RUNG wire#w4
      S_Coil( "DB_GC".HallDownCancel[9] )
   END_RUNG
   RUNG wire#powerrail
      Contact( "8层外呼上行指示灯" )
      Contact( "8层外呼下行指示灯" )
      Contact( "1号梯下行命令" )
      I_Contact( "1号梯上行命令" )
      Contact( "1号梯本层召唤开门信号" )
      wire#w5
      Contact( "1号梯电梯停稳信号" )
      { S7_Templates := "SrcType := Int" } EQ_Contact(in1 := "1号梯当前楼层数", in2 := 8)
      Contact( "8层外呼下行指示灯" )
      wire#w6
      R_Coil( "8层外呼下行指示灯" )
   END_RUNG
   RUNG wire#powerrail
      I_Contact( "8层外呼上行指示灯" )
      Contact( "8层外呼下行指示灯" )
      Contact( "1号梯本层召唤开门信号" )
      Contact( "1号梯下行命令" )
      I_Contact( "1号梯上行命令" )
   END_RUNG wire#w5
   RUNG wire#powerrail
      I_Contact( "1号梯上行命令" )
      I_Contact( "1号梯下行命令" )
   END_RUNG wire#w5
   RUNG wire#w6
      R_Coil( "1号梯8层下呼" )
   END_RUNG
   RUNG wire#w6
      S_Coil( "DB_GC".HallDownCancel[8] )
   END_RUNG
   RUNG wire#powerrail
      Contact( "7层外呼上行指示灯" )
      Contact( "7层外呼下行指示灯" )
      Contact( "1号梯下行命令" )
      I_Contact( "1号梯上行命令" )
      Contact( "1号梯本层召唤开门信号" )
      wire#w7
      Contact( "1号梯电梯停稳信号" )
      { S7_Templates := "SrcType := Int" } EQ_Contact(in1 := "1号梯当前楼层数", in2 := 7)
      Contact( "7层外呼下行指示灯" )
      wire#w8
      R_Coil( "7层外呼下行指示灯" )
   END_RUNG
   RUNG wire#powerrail
      I_Contact( "7层外呼上行指示灯" )
      Contact( "7层外呼下行指示灯" )
      Contact( "1号梯本层召唤开门信号" )
      Contact( "1号梯下行命令" )
      I_Contact( "1号梯上行命令" )
   END_RUNG wire#w7
   RUNG wire#powerrail
      I_Contact( "1号梯上行命令" )
      I_Contact( "1号梯下行命令" )
   END_RUNG wire#w7
   RUNG wire#w8
      R_Coil( "1号梯7层下呼" )
   END_RUNG
   RUNG wire#w8
      S_Coil( "DB_GC".HallDownCancel[7] )
   END_RUNG
   RUNG wire#powerrail
      Contact( "6层外呼上行指示灯" )
      Contact( "6层外呼下行指示灯" )
      Contact( "1号梯下行命令" )
      I_Contact( "1号梯上行命令" )
      Contact( "1号梯本层召唤开门信号" )
      wire#w9
      Contact( "1号梯电梯停稳信号" )
      { S7_Templates := "SrcType := Int" } EQ_Contact(in1 := "1号梯当前楼层数", in2 := 6)
      Contact( "6层外呼下行指示灯" )
      wire#w10
      R_Coil( "6层外呼下行指示灯" )
   END_RUNG
   RUNG wire#powerrail
      I_Contact( "6层外呼上行指示灯" )
      Contact( "6层外呼下行指示灯" )
      Contact( "1号梯本层召唤开门信号" )
      Contact( "1号梯下行命令" )
      I_Contact( "1号梯上行命令" )
   END_RUNG wire#w9
   RUNG wire#powerrail
      I_Contact( "1号梯上行命令" )
      I_Contact( "1号梯下行命令" )
   END_RUNG wire#w9
   RUNG wire#w10
      R_Coil( "1号梯6层下呼" )
   END_RUNG
   RUNG wire#w10
      S_Coil( "DB_GC".HallDownCancel[6] )
   END_RUNG
   RUNG wire#powerrail
      Contact( "5层外呼上行指示灯" )
      Contact( "5层外呼下行指示灯" )
      Contact( "1号梯下行命令" )
      I_Contact( "1号梯上行命令" )
      Contact( "1号梯本层召唤开门信号" )
      wire#w11
      Contact( "1号梯电梯停稳信号" )
      { S7_Templates := "SrcType := Int" } EQ_Contact(in1 := "1号梯当前楼层数", in2 := 5)
      Contact( "5层外呼下行指示灯" )
      wire#w12
      R_Coil( "5层外呼下行指示灯" )
   END_RUNG
   RUNG wire#powerrail
      I_Contact( "5层外呼上行指示灯" )
      Contact( "5层外呼下行指示灯" )
      Contact( "1号梯本层召唤开门信号" )
      Contact( "1号梯下行命令" )
      I_Contact( "1号梯上行命令" )
   END_RUNG wire#w11
   RUNG wire#powerrail
      I_Contact( "1号梯上行命令" )
      I_Contact( "1号梯下行命令" )
   END_RUNG wire#w11
   RUNG wire#w12
      R_Coil( "1号梯5层下呼" )
   END_RUNG
   RUNG wire#w12
      S_Coil( "DB_GC".HallDownCancel[5] )
   END_RUNG
   RUNG wire#powerrail
      Contact( "4层外呼上行指示灯" )
      Contact( "4层外呼下行指示灯" )
      Contact( "1号梯下行命令" )
      I_Contact( "1号梯上行命令" )
      Contact( "1号梯本层召唤开门信号" )
      wire#w13
      Contact( "1号梯电梯停稳信号" )
      { S7_Templates := "SrcType := Int" } EQ_Contact(in1 := "1号梯当前楼层数", in2 := 4)
      Contact( "4层外呼下行指示灯" )
      wire#w14
      R_Coil( "4层外呼下行指示灯" )
   END_RUNG
   RUNG wire#powerrail
      I_Contact( "4层外呼上行指示灯" )
      Contact( "4层外呼下行指示灯" )
      Contact( "1号梯本层召唤开门信号" )
      Contact( "1号梯下行命令" )
      I_Contact( "1号梯上行命令" )
   END_RUNG wire#w13
   RUNG wire#powerrail
      I_Contact( "1号梯上行命令" )
      I_Contact( "1号梯下行命令" )
   END_RUNG wire#w13
   RUNG wire#w14
      R_Coil( "1号梯4层下呼" )
   END_RUNG
   RUNG wire#w14
      S_Coil( "DB_GC".HallDownCancel[4] )
   END_RUNG
   RUNG wire#powerrail
      Contact( "3层外呼上行指示灯" )
      Contact( "3层外呼下行指示灯" )
      Contact( "1号梯下行命令" )
      I_Contact( "1号梯上行命令" )
      Contact( "1号梯本层召唤开门信号" )
      wire#w15
      Contact( "1号梯电梯停稳信号" )
      { S7_Templates := "SrcType := Int" } EQ_Contact(in1 := "1号梯当前楼层数", in2 := 3)
      Contact( "3层外呼下行指示灯" )
      wire#w16
      R_Coil( "3层外呼下行指示灯" )
   END_RUNG
   RUNG wire#powerrail
      I_Contact( "3层外呼上行指示灯" )
      Contact( "3层外呼下行指示灯" )
      Contact( "1号梯本层召唤开门信号" )
      Contact( "1号梯下行命令" )
      I_Contact( "1号梯上行命令" )
   END_RUNG wire#w15
   RUNG wire#powerrail
      I_Contact( "1号梯上行命令" )
      I_Contact( "1号梯下行命令" )
   END_RUNG wire#w15
   RUNG wire#w16
      R_Coil( "1号梯3层下呼" )
   END_RUNG
   RUNG wire#w16
      S_Coil( "DB_GC".HallDownCancel[3] )
   END_RUNG
   RUNG wire#powerrail
      Contact( "2层外呼上行指示灯" )
      Contact( "2层外呼下行指示灯" )
      Contact( "1号梯下行命令" )
      I_Contact( "1号梯上行命令" )
      Contact( "1号梯本层召唤开门信号" )
      wire#w17
      Contact( "1号梯电梯停稳信号" )
      { S7_Templates := "SrcType := Int" } EQ_Contact(in1 := "1号梯当前楼层数", in2 := 2)
      Contact( "2层外呼下行指示灯" )
      wire#w18
      R_Coil( "2层外呼下行指示灯" )
   END_RUNG
   RUNG wire#powerrail
      I_Contact( "2层外呼上行指示灯" )
      Contact( "2层外呼下行指示灯" )
      Contact( "1号梯本层召唤开门信号" )
      Contact( "1号梯下行命令" )
      I_Contact( "1号梯上行命令" )
   END_RUNG wire#w17
   RUNG wire#powerrail
      I_Contact( "1号梯上行命令" )
      I_Contact( "1号梯下行命令" )
   END_RUNG wire#w17
   RUNG wire#w18
      R_Coil( "1号梯2层下呼" )
   END_RUNG
   RUNG wire#w18
      S_Coil( "DB_GC".HallDownCancel[2] )
   END_RUNG
   // the same network as SCL:
   #_w1 := (("10层外呼下行指示灯" AND "1号梯本层召唤开门信号") OR (NOT "1号梯上行命令" AND NOT "1号梯下行命令")) AND ("1号梯当前楼层数" = 10) AND "10层外呼下行指示灯" AND "1号梯电梯停稳信号";
   IF #_w1 THEN
       "10层外呼下行指示灯" := FALSE;
       "1号梯10层下呼" := FALSE;
       "DB_GC".HallDownCancel[10] := TRUE;
   END_IF;
   #_w2 := (("9层外呼上行指示灯" AND "9层外呼下行指示灯" AND "1号梯下行命令" AND NOT "1号梯上行命令" AND "1号梯本层召唤开门信号") OR (NOT "9层外呼上行指示灯" AND "9层外呼下行指示灯" AND "1号梯本层召唤开门信号" AND "1号梯下行命令" AND NOT "1号梯上行命令") OR (NOT "1号梯上行命令" AND NOT "1号梯下行命令")) AND "1号梯电梯停稳信号" AND ("1号梯当前楼层数" = 9) AND "9层外呼下行指示灯";
   IF #_w2 THEN
       "9层外呼下行指示灯" := FALSE;
       "1号梯9层下呼" := FALSE;
       "DB_GC".HallDownCancel[9] := TRUE;
   END_IF;
   #_w3 := (("8层外呼上行指示灯" AND "8层外呼下行指示灯" AND "1号梯下行命令" AND NOT "1号梯上行命令" AND "1号梯本层召唤开门信号") OR (NOT "8层外呼上行指示灯" AND "8层外呼下行指示灯" AND "1号梯本层召唤开门信号" AND "1号梯下行命令" AND NOT "1号梯上行命令") OR (NOT "1号梯上行命令" AND NOT "1号梯下行命令")) AND "1号梯电梯停稳信号" AND ("1号梯当前楼层数" = 8) AND "8层外呼下行指示灯";
   IF #_w3 THEN
       "8层外呼下行指示灯" := FALSE;
       "1号梯8层下呼" := FALSE;
       "DB_GC".HallDownCancel[8] := TRUE;
   END_IF;
   #_w4 := (("7层外呼上行指示灯" AND "7层外呼下行指示灯" AND "1号梯下行命令" AND NOT "1号梯上行命令" AND "1号梯本层召唤开门信号") OR (NOT "7层外呼上行指示灯" AND "7层外呼下行指示灯" AND "1号梯本层召唤开门信号" AND "1号梯下行命令" AND NOT "1号梯上行命令") OR (NOT "1号梯上行命令" AND NOT "1号梯下行命令")) AND "1号梯电梯停稳信号" AND ("1号梯当前楼层数" = 7) AND "7层外呼下行指示灯";
   IF #_w4 THEN
       "7层外呼下行指示灯" := FALSE;
       "1号梯7层下呼" := FALSE;
       "DB_GC".HallDownCancel[7] := TRUE;
   END_IF;
   #_w5 := (("6层外呼上行指示灯" AND "6层外呼下行指示灯" AND "1号梯下行命令" AND NOT "1号梯上行命令" AND "1号梯本层召唤开门信号") OR (NOT "6层外呼上行指示灯" AND "6层外呼下行指示灯" AND "1号梯本层召唤开门信号" AND "1号梯下行命令" AND NOT "1号梯上行命令") OR (NOT "1号梯上行命令" AND NOT "1号梯下行命令")) AND "1号梯电梯停稳信号" AND ("1号梯当前楼层数" = 6) AND "6层外呼下行指示灯";
   IF #_w5 THEN
       "6层外呼下行指示灯" := FALSE;
       "1号梯6层下呼" := FALSE;
       "DB_GC".HallDownCancel[6] := TRUE;
   END_IF;
   #_w6 := (("5层外呼上行指示灯" AND "5层外呼下行指示灯" AND "1号梯下行命令" AND NOT "1号梯上行命令" AND "1号梯本层召唤开门信号") OR (NOT "5层外呼上行指示灯" AND "5层外呼下行指示灯" AND "1号梯本层召唤开门信号" AND "1号梯下行命令" AND NOT "1号梯上行命令") OR (NOT "1号梯上行命令" AND NOT "1号梯下行命令")) AND "1号梯电梯停稳信号" AND ("1号梯当前楼层数" = 5) AND "5层外呼下行指示灯";
   IF #_w6 THEN
       "5层外呼下行指示灯" := FALSE;
       "1号梯5层下呼" := FALSE;
       "DB_GC".HallDownCancel[5] := TRUE;
   END_IF;
   #_w7 := (("4层外呼上行指示灯" AND "4层外呼下行指示灯" AND "1号梯下行命令" AND NOT "1号梯上行命令" AND "1号梯本层召唤开门信号") OR (NOT "4层外呼上行指示灯" AND "4层外呼下行指示灯" AND "1号梯本层召唤开门信号" AND "1号梯下行命令" AND NOT "1号梯上行命令") OR (NOT "1号梯上行命令" AND NOT "1号梯下行命令")) AND "1号梯电梯停稳信号" AND ("1号梯当前楼层数" = 4) AND "4层外呼下行指示灯";
   IF #_w7 THEN
       "4层外呼下行指示灯" := FALSE;
       "1号梯4层下呼" := FALSE;
       "DB_GC".HallDownCancel[4] := TRUE;
   END_IF;
   #_w8 := (("3层外呼上行指示灯" AND "3层外呼下行指示灯" AND "1号梯下行命令" AND NOT "1号梯上行命令" AND "1号梯本层召唤开门信号") OR (NOT "3层外呼上行指示灯" AND "3层外呼下行指示灯" AND "1号梯本层召唤开门信号" AND "1号梯下行命令" AND NOT "1号梯上行命令") OR (NOT "1号梯上行命令" AND NOT "1号梯下行命令")) AND "1号梯电梯停稳信号" AND ("1号梯当前楼层数" = 3) AND "3层外呼下行指示灯";
   IF #_w8 THEN
       "3层外呼下行指示灯" := FALSE;
       "1号梯3层下呼" := FALSE;
       "DB_GC".HallDownCancel[3] := TRUE;
   END_IF;
   #_w9 := (("2层外呼上行指示灯" AND "2层外呼下行指示灯" AND "1号梯下行命令" AND NOT "1号梯上行命令" AND "1号梯本层召唤开门信号") OR (NOT "2层外呼上行指示灯" AND "2层外呼下行指示灯" AND "1号梯本层召唤开门信号" AND "1号梯下行命令" AND NOT "1号梯上行命令") OR (NOT "1号梯上行命令" AND NOT "1号梯下行命令")) AND "1号梯电梯停稳信号" AND ("1号梯当前楼层数" = 2) AND "2层外呼下行指示灯";
   IF #_w9 THEN
       "2层外呼下行指示灯" := FALSE;
       "1号梯2层下呼" := FALSE;
       "DB_GC".HallDownCancel[2] := TRUE;
   END_IF;
END_REGION

REGION Network 2: 1号梯终止上呼
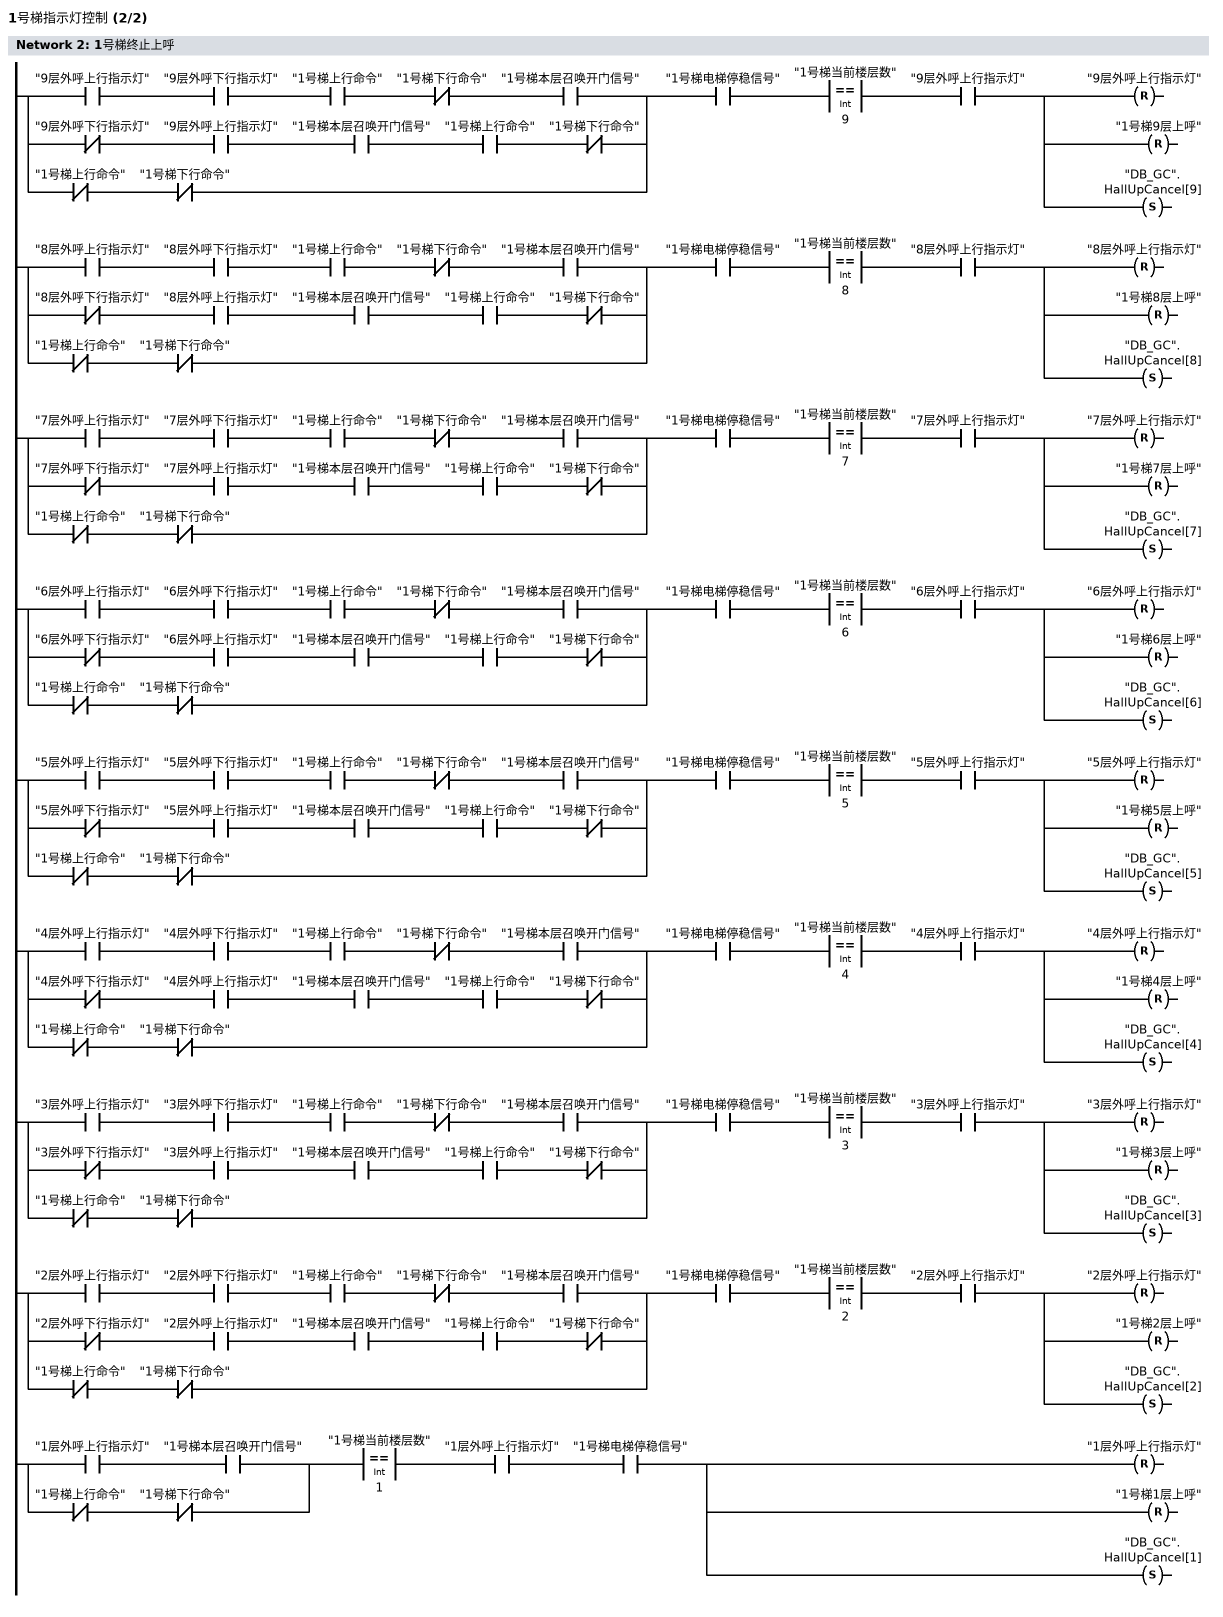
   RUNG wire#powerrail
      Contact( "9层外呼上行指示灯" )
      Contact( "9层外呼下行指示灯" )
      Contact( "1号梯上行命令" )
      I_Contact( "1号梯下行命令" )
      Contact( "1号梯本层召唤开门信号" )
      wire#w1
      Contact( "1号梯电梯停稳信号" )
      { S7_Templates := "SrcType := Int" } EQ_Contact(in1 := "1号梯当前楼层数", in2 := 9)
      Contact( "9层外呼上行指示灯" )
      wire#w2
      R_Coil( "9层外呼上行指示灯" )
   END_RUNG
   RUNG wire#powerrail
      I_Contact( "9层外呼下行指示灯" )
      Contact( "9层外呼上行指示灯" )
      Contact( "1号梯本层召唤开门信号" )
      Contact( "1号梯上行命令" )
      I_Contact( "1号梯下行命令" )
   END_RUNG wire#w1
   RUNG wire#powerrail
      I_Contact( "1号梯上行命令" )
      I_Contact( "1号梯下行命令" )
   END_RUNG wire#w1
   RUNG wire#w2
      R_Coil( "1号梯9层上呼" )
   END_RUNG
   RUNG wire#w2
      S_Coil( "DB_GC".HallUpCancel[9] )
   END_RUNG
   RUNG wire#powerrail
      Contact( "8层外呼上行指示灯" )
      Contact( "8层外呼下行指示灯" )
      Contact( "1号梯上行命令" )
      I_Contact( "1号梯下行命令" )
      Contact( "1号梯本层召唤开门信号" )
      wire#w3
      Contact( "1号梯电梯停稳信号" )
      { S7_Templates := "SrcType := Int" } EQ_Contact(in1 := "1号梯当前楼层数", in2 := 8)
      Contact( "8层外呼上行指示灯" )
      wire#w4
      R_Coil( "8层外呼上行指示灯" )
   END_RUNG
   RUNG wire#powerrail
      I_Contact( "8层外呼下行指示灯" )
      Contact( "8层外呼上行指示灯" )
      Contact( "1号梯本层召唤开门信号" )
      Contact( "1号梯上行命令" )
      I_Contact( "1号梯下行命令" )
   END_RUNG wire#w3
   RUNG wire#powerrail
      I_Contact( "1号梯上行命令" )
      I_Contact( "1号梯下行命令" )
   END_RUNG wire#w3
   RUNG wire#w4
      R_Coil( "1号梯8层上呼" )
   END_RUNG
   RUNG wire#w4
      S_Coil( "DB_GC".HallUpCancel[8] )
   END_RUNG
   RUNG wire#powerrail
      Contact( "7层外呼上行指示灯" )
      Contact( "7层外呼下行指示灯" )
      Contact( "1号梯上行命令" )
      I_Contact( "1号梯下行命令" )
      Contact( "1号梯本层召唤开门信号" )
      wire#w5
      Contact( "1号梯电梯停稳信号" )
      { S7_Templates := "SrcType := Int" } EQ_Contact(in1 := "1号梯当前楼层数", in2 := 7)
      Contact( "7层外呼上行指示灯" )
      wire#w6
      R_Coil( "7层外呼上行指示灯" )
   END_RUNG
   RUNG wire#powerrail
      I_Contact( "7层外呼下行指示灯" )
      Contact( "7层外呼上行指示灯" )
      Contact( "1号梯本层召唤开门信号" )
      Contact( "1号梯上行命令" )
      I_Contact( "1号梯下行命令" )
   END_RUNG wire#w5
   RUNG wire#powerrail
      I_Contact( "1号梯上行命令" )
      I_Contact( "1号梯下行命令" )
   END_RUNG wire#w5
   RUNG wire#w6
      R_Coil( "1号梯7层上呼" )
   END_RUNG
   RUNG wire#w6
      S_Coil( "DB_GC".HallUpCancel[7] )
   END_RUNG
   RUNG wire#powerrail
      Contact( "6层外呼上行指示灯" )
      Contact( "6层外呼下行指示灯" )
      Contact( "1号梯上行命令" )
      I_Contact( "1号梯下行命令" )
      Contact( "1号梯本层召唤开门信号" )
      wire#w7
      Contact( "1号梯电梯停稳信号" )
      { S7_Templates := "SrcType := Int" } EQ_Contact(in1 := "1号梯当前楼层数", in2 := 6)
      Contact( "6层外呼上行指示灯" )
      wire#w8
      R_Coil( "6层外呼上行指示灯" )
   END_RUNG
   RUNG wire#powerrail
      I_Contact( "6层外呼下行指示灯" )
      Contact( "6层外呼上行指示灯" )
      Contact( "1号梯本层召唤开门信号" )
      Contact( "1号梯上行命令" )
      I_Contact( "1号梯下行命令" )
   END_RUNG wire#w7
   RUNG wire#powerrail
      I_Contact( "1号梯上行命令" )
      I_Contact( "1号梯下行命令" )
   END_RUNG wire#w7
   RUNG wire#w8
      R_Coil( "1号梯6层上呼" )
   END_RUNG
   RUNG wire#w8
      S_Coil( "DB_GC".HallUpCancel[6] )
   END_RUNG
   RUNG wire#powerrail
      Contact( "5层外呼上行指示灯" )
      Contact( "5层外呼下行指示灯" )
      Contact( "1号梯上行命令" )
      I_Contact( "1号梯下行命令" )
      Contact( "1号梯本层召唤开门信号" )
      wire#w9
      Contact( "1号梯电梯停稳信号" )
      { S7_Templates := "SrcType := Int" } EQ_Contact(in1 := "1号梯当前楼层数", in2 := 5)
      Contact( "5层外呼上行指示灯" )
      wire#w10
      R_Coil( "5层外呼上行指示灯" )
   END_RUNG
   RUNG wire#powerrail
      I_Contact( "5层外呼下行指示灯" )
      Contact( "5层外呼上行指示灯" )
      Contact( "1号梯本层召唤开门信号" )
      Contact( "1号梯上行命令" )
      I_Contact( "1号梯下行命令" )
   END_RUNG wire#w9
   RUNG wire#powerrail
      I_Contact( "1号梯上行命令" )
      I_Contact( "1号梯下行命令" )
   END_RUNG wire#w9
   RUNG wire#w10
      R_Coil( "1号梯5层上呼" )
   END_RUNG
   RUNG wire#w10
      S_Coil( "DB_GC".HallUpCancel[5] )
   END_RUNG
   RUNG wire#powerrail
      Contact( "4层外呼上行指示灯" )
      Contact( "4层外呼下行指示灯" )
      Contact( "1号梯上行命令" )
      I_Contact( "1号梯下行命令" )
      Contact( "1号梯本层召唤开门信号" )
      wire#w11
      Contact( "1号梯电梯停稳信号" )
      { S7_Templates := "SrcType := Int" } EQ_Contact(in1 := "1号梯当前楼层数", in2 := 4)
      Contact( "4层外呼上行指示灯" )
      wire#w12
      R_Coil( "4层外呼上行指示灯" )
   END_RUNG
   RUNG wire#powerrail
      I_Contact( "4层外呼下行指示灯" )
      Contact( "4层外呼上行指示灯" )
      Contact( "1号梯本层召唤开门信号" )
      Contact( "1号梯上行命令" )
      I_Contact( "1号梯下行命令" )
   END_RUNG wire#w11
   RUNG wire#powerrail
      I_Contact( "1号梯上行命令" )
      I_Contact( "1号梯下行命令" )
   END_RUNG wire#w11
   RUNG wire#w12
      R_Coil( "1号梯4层上呼" )
   END_RUNG
   RUNG wire#w12
      S_Coil( "DB_GC".HallUpCancel[4] )
   END_RUNG
   RUNG wire#powerrail
      Contact( "3层外呼上行指示灯" )
      Contact( "3层外呼下行指示灯" )
      Contact( "1号梯上行命令" )
      I_Contact( "1号梯下行命令" )
      Contact( "1号梯本层召唤开门信号" )
      wire#w13
      Contact( "1号梯电梯停稳信号" )
      { S7_Templates := "SrcType := Int" } EQ_Contact(in1 := "1号梯当前楼层数", in2 := 3)
      Contact( "3层外呼上行指示灯" )
      wire#w14
      R_Coil( "3层外呼上行指示灯" )
   END_RUNG
   RUNG wire#powerrail
      I_Contact( "3层外呼下行指示灯" )
      Contact( "3层外呼上行指示灯" )
      Contact( "1号梯本层召唤开门信号" )
      Contact( "1号梯上行命令" )
      I_Contact( "1号梯下行命令" )
   END_RUNG wire#w13
   RUNG wire#powerrail
      I_Contact( "1号梯上行命令" )
      I_Contact( "1号梯下行命令" )
   END_RUNG wire#w13
   RUNG wire#w14
      R_Coil( "1号梯3层上呼" )
   END_RUNG
   RUNG wire#w14
      S_Coil( "DB_GC".HallUpCancel[3] )
   END_RUNG
   RUNG wire#powerrail
      Contact( "2层外呼上行指示灯" )
      Contact( "2层外呼下行指示灯" )
      Contact( "1号梯上行命令" )
      I_Contact( "1号梯下行命令" )
      Contact( "1号梯本层召唤开门信号" )
      wire#w15
      Contact( "1号梯电梯停稳信号" )
      { S7_Templates := "SrcType := Int" } EQ_Contact(in1 := "1号梯当前楼层数", in2 := 2)
      Contact( "2层外呼上行指示灯" )
      wire#w16
      R_Coil( "2层外呼上行指示灯" )
   END_RUNG
   RUNG wire#powerrail
      I_Contact( "2层外呼下行指示灯" )
      Contact( "2层外呼上行指示灯" )
      Contact( "1号梯本层召唤开门信号" )
      Contact( "1号梯上行命令" )
      I_Contact( "1号梯下行命令" )
   END_RUNG wire#w15
   RUNG wire#powerrail
      I_Contact( "1号梯上行命令" )
      I_Contact( "1号梯下行命令" )
   END_RUNG wire#w15
   RUNG wire#w16
      R_Coil( "1号梯2层上呼" )
   END_RUNG
   RUNG wire#w16
      S_Coil( "DB_GC".HallUpCancel[2] )
   END_RUNG
   RUNG wire#powerrail
      Contact( "1层外呼上行指示灯" )
      Contact( "1号梯本层召唤开门信号" )
      wire#w17
      { S7_Templates := "SrcType := Int" } EQ_Contact(in1 := "1号梯当前楼层数", in2 := 1)
      Contact( "1层外呼上行指示灯" )
      Contact( "1号梯电梯停稳信号" )
      wire#w18
      R_Coil( "1层外呼上行指示灯" )
   END_RUNG
   RUNG wire#powerrail
      I_Contact( "1号梯上行命令" )
      I_Contact( "1号梯下行命令" )
   END_RUNG wire#w17
   RUNG wire#w18
      R_Coil( "1号梯1层上呼" )
   END_RUNG
   RUNG wire#w18
      S_Coil( "DB_GC".HallUpCancel[1] )
   END_RUNG
   // the same network as SCL:
   #_w1 := (("9层外呼上行指示灯" AND "9层外呼下行指示灯" AND "1号梯上行命令" AND NOT "1号梯下行命令" AND "1号梯本层召唤开门信号") OR (NOT "9层外呼下行指示灯" AND "9层外呼上行指示灯" AND "1号梯本层召唤开门信号" AND "1号梯上行命令" AND NOT "1号梯下行命令") OR (NOT "1号梯上行命令" AND NOT "1号梯下行命令")) AND "1号梯电梯停稳信号" AND ("1号梯当前楼层数" = 9) AND "9层外呼上行指示灯";
   IF #_w1 THEN
       "9层外呼上行指示灯" := FALSE;
       "1号梯9层上呼" := FALSE;
       "DB_GC".HallUpCancel[9] := TRUE;
   END_IF;
   #_w2 := (("8层外呼上行指示灯" AND "8层外呼下行指示灯" AND "1号梯上行命令" AND NOT "1号梯下行命令" AND "1号梯本层召唤开门信号") OR (NOT "8层外呼下行指示灯" AND "8层外呼上行指示灯" AND "1号梯本层召唤开门信号" AND "1号梯上行命令" AND NOT "1号梯下行命令") OR (NOT "1号梯上行命令" AND NOT "1号梯下行命令")) AND "1号梯电梯停稳信号" AND ("1号梯当前楼层数" = 8) AND "8层外呼上行指示灯";
   IF #_w2 THEN
       "8层外呼上行指示灯" := FALSE;
       "1号梯8层上呼" := FALSE;
       "DB_GC".HallUpCancel[8] := TRUE;
   END_IF;
   #_w3 := (("7层外呼上行指示灯" AND "7层外呼下行指示灯" AND "1号梯上行命令" AND NOT "1号梯下行命令" AND "1号梯本层召唤开门信号") OR (NOT "7层外呼下行指示灯" AND "7层外呼上行指示灯" AND "1号梯本层召唤开门信号" AND "1号梯上行命令" AND NOT "1号梯下行命令") OR (NOT "1号梯上行命令" AND NOT "1号梯下行命令")) AND "1号梯电梯停稳信号" AND ("1号梯当前楼层数" = 7) AND "7层外呼上行指示灯";
   IF #_w3 THEN
       "7层外呼上行指示灯" := FALSE;
       "1号梯7层上呼" := FALSE;
       "DB_GC".HallUpCancel[7] := TRUE;
   END_IF;
   #_w4 := (("6层外呼上行指示灯" AND "6层外呼下行指示灯" AND "1号梯上行命令" AND NOT "1号梯下行命令" AND "1号梯本层召唤开门信号") OR (NOT "6层外呼下行指示灯" AND "6层外呼上行指示灯" AND "1号梯本层召唤开门信号" AND "1号梯上行命令" AND NOT "1号梯下行命令") OR (NOT "1号梯上行命令" AND NOT "1号梯下行命令")) AND "1号梯电梯停稳信号" AND ("1号梯当前楼层数" = 6) AND "6层外呼上行指示灯";
   IF #_w4 THEN
       "6层外呼上行指示灯" := FALSE;
       "1号梯6层上呼" := FALSE;
       "DB_GC".HallUpCancel[6] := TRUE;
   END_IF;
   #_w5 := (("5层外呼上行指示灯" AND "5层外呼下行指示灯" AND "1号梯上行命令" AND NOT "1号梯下行命令" AND "1号梯本层召唤开门信号") OR (NOT "5层外呼下行指示灯" AND "5层外呼上行指示灯" AND "1号梯本层召唤开门信号" AND "1号梯上行命令" AND NOT "1号梯下行命令") OR (NOT "1号梯上行命令" AND NOT "1号梯下行命令")) AND "1号梯电梯停稳信号" AND ("1号梯当前楼层数" = 5) AND "5层外呼上行指示灯";
   IF #_w5 THEN
       "5层外呼上行指示灯" := FALSE;
       "1号梯5层上呼" := FALSE;
       "DB_GC".HallUpCancel[5] := TRUE;
   END_IF;
   #_w6 := (("4层外呼上行指示灯" AND "4层外呼下行指示灯" AND "1号梯上行命令" AND NOT "1号梯下行命令" AND "1号梯本层召唤开门信号") OR (NOT "4层外呼下行指示灯" AND "4层外呼上行指示灯" AND "1号梯本层召唤开门信号" AND "1号梯上行命令" AND NOT "1号梯下行命令") OR (NOT "1号梯上行命令" AND NOT "1号梯下行命令")) AND "1号梯电梯停稳信号" AND ("1号梯当前楼层数" = 4) AND "4层外呼上行指示灯";
   IF #_w6 THEN
       "4层外呼上行指示灯" := FALSE;
       "1号梯4层上呼" := FALSE;
       "DB_GC".HallUpCancel[4] := TRUE;
   END_IF;
   #_w7 := (("3层外呼上行指示灯" AND "3层外呼下行指示灯" AND "1号梯上行命令" AND NOT "1号梯下行命令" AND "1号梯本层召唤开门信号") OR (NOT "3层外呼下行指示灯" AND "3层外呼上行指示灯" AND "1号梯本层召唤开门信号" AND "1号梯上行命令" AND NOT "1号梯下行命令") OR (NOT "1号梯上行命令" AND NOT "1号梯下行命令")) AND "1号梯电梯停稳信号" AND ("1号梯当前楼层数" = 3) AND "3层外呼上行指示灯";
   IF #_w7 THEN
       "3层外呼上行指示灯" := FALSE;
       "1号梯3层上呼" := FALSE;
       "DB_GC".HallUpCancel[3] := TRUE;
   END_IF;
   #_w8 := (("2层外呼上行指示灯" AND "2层外呼下行指示灯" AND "1号梯上行命令" AND NOT "1号梯下行命令" AND "1号梯本层召唤开门信号") OR (NOT "2层外呼下行指示灯" AND "2层外呼上行指示灯" AND "1号梯本层召唤开门信号" AND "1号梯上行命令" AND NOT "1号梯下行命令") OR (NOT "1号梯上行命令" AND NOT "1号梯下行命令")) AND "1号梯电梯停稳信号" AND ("1号梯当前楼层数" = 2) AND "2层外呼上行指示灯";
   IF #_w8 THEN
       "2层外呼上行指示灯" := FALSE;
       "1号梯2层上呼" := FALSE;
       "DB_GC".HallUpCancel[2] := TRUE;
   END_IF;
   #_w9 := (("1层外呼上行指示灯" AND "1号梯本层召唤开门信号") OR (NOT "1号梯上行命令" AND NOT "1号梯下行命令")) AND ("1号梯当前楼层数" = 1) AND "1层外呼上行指示灯" AND "1号梯电梯停稳信号";
   IF #_w9 THEN
       "1层外呼上行指示灯" := FALSE;
       "1号梯1层上呼" := FALSE;
       "DB_GC".HallUpCancel[1] := TRUE;
   END_IF;
END_REGION
END_FUNCTION

FUNCTION "3号梯指示灯控制" : Void   // FC14, LAD
{ S7_Optimized_Access := 'TRUE' }
VERSION : 0.1
   VAR_TEMP   // added for the SCL form of the ladder/FBD networks
      _w1 : Bool;
      _w2 : Bool;
      _w3 : Bool;
      _w4 : Bool;
      _w5 : Bool;
      _w6 : Bool;
      _w7 : Bool;
      _w8 : Bool;
      _w9 : Bool;
   END_VAR
BEGIN

REGION Network 1: 3号梯终止下呼
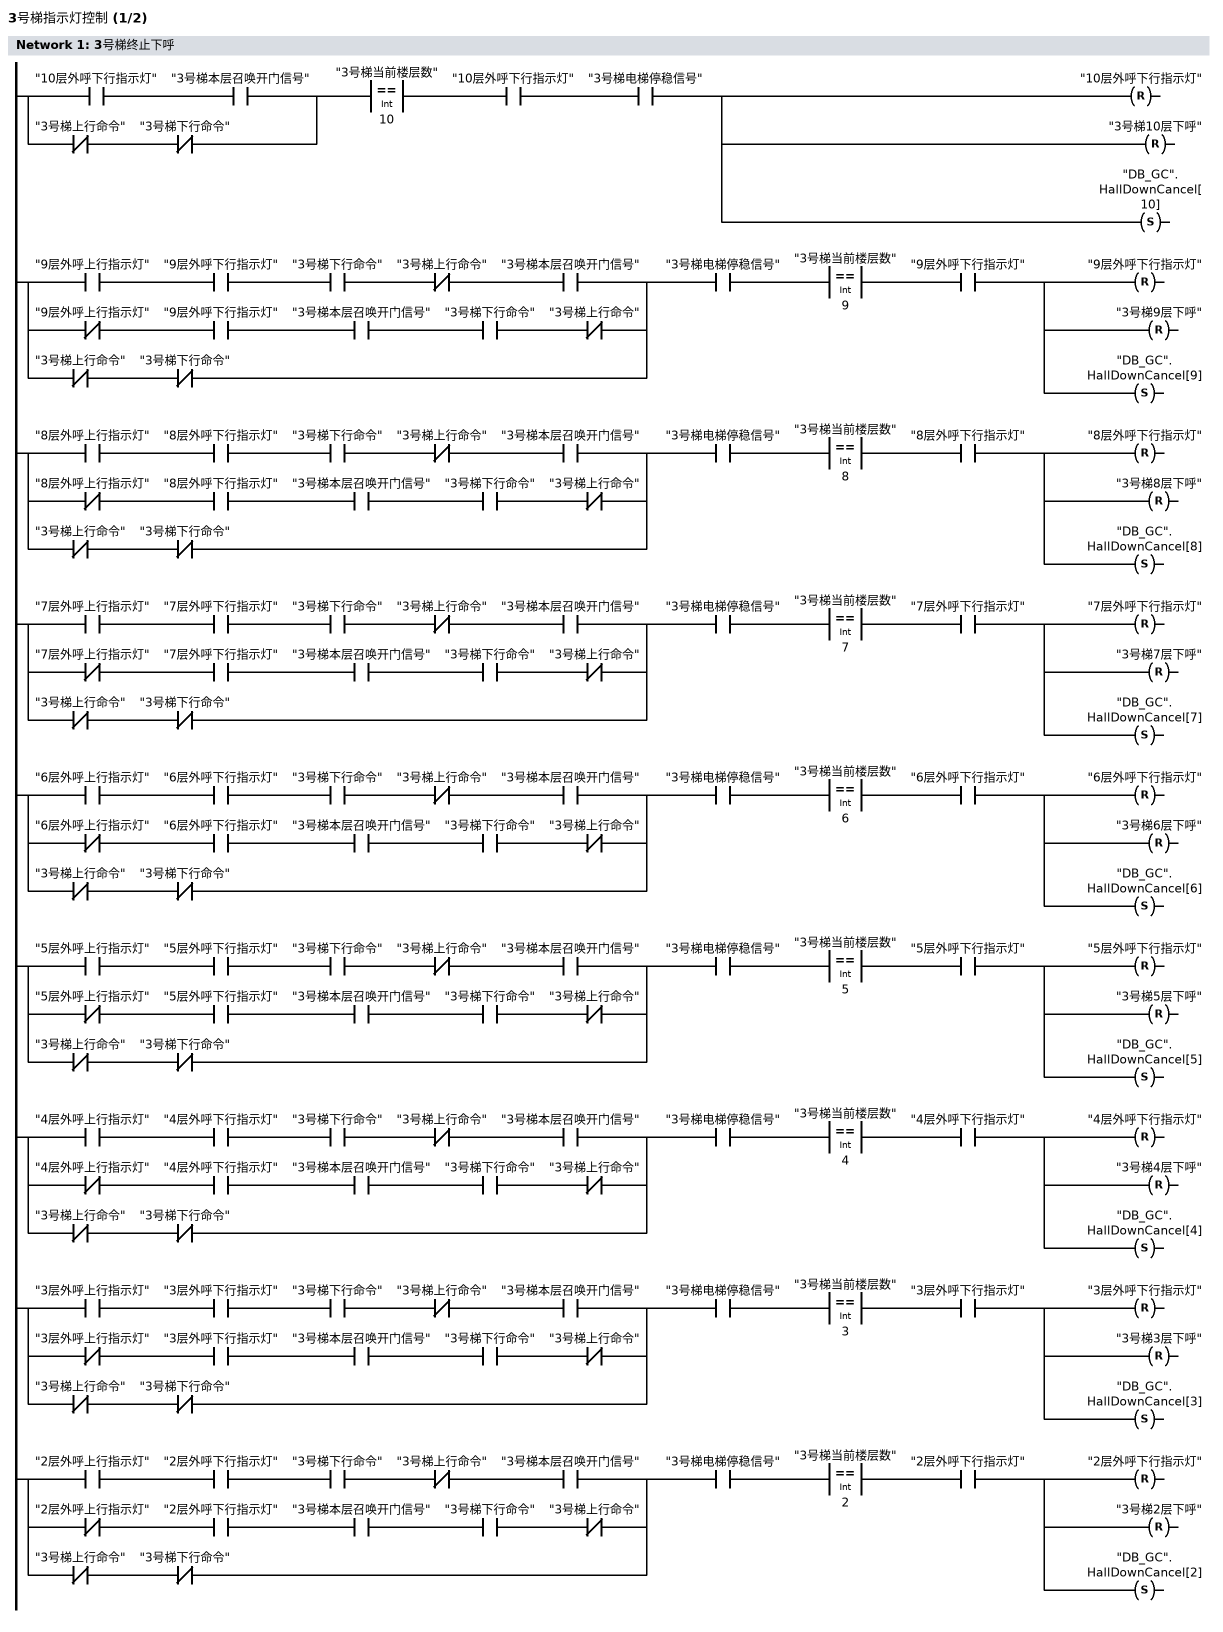
   RUNG wire#powerrail
      Contact( "10层外呼下行指示灯" )
      Contact( "3号梯本层召唤开门信号" )
      wire#w1
      { S7_Templates := "SrcType := Int" } EQ_Contact(in1 := "3号梯当前楼层数", in2 := 10)
      Contact( "10层外呼下行指示灯" )
      Contact( "3号梯电梯停稳信号" )
      wire#w2
      R_Coil( "10层外呼下行指示灯" )
   END_RUNG
   RUNG wire#powerrail
      I_Contact( "3号梯上行命令" )
      I_Contact( "3号梯下行命令" )
   END_RUNG wire#w1
   RUNG wire#w2
      R_Coil( "3号梯10层下呼" )
   END_RUNG
   RUNG wire#w2
      S_Coil( "DB_GC".HallDownCancel[10] )
   END_RUNG
   RUNG wire#powerrail
      Contact( "9层外呼上行指示灯" )
      Contact( "9层外呼下行指示灯" )
      Contact( "3号梯下行命令" )
      I_Contact( "3号梯上行命令" )
      Contact( "3号梯本层召唤开门信号" )
      wire#w3
      Contact( "3号梯电梯停稳信号" )
      { S7_Templates := "SrcType := Int" } EQ_Contact(in1 := "3号梯当前楼层数", in2 := 9)
      Contact( "9层外呼下行指示灯" )
      wire#w4
      R_Coil( "9层外呼下行指示灯" )
   END_RUNG
   RUNG wire#powerrail
      I_Contact( "9层外呼上行指示灯" )
      Contact( "9层外呼下行指示灯" )
      Contact( "3号梯本层召唤开门信号" )
      Contact( "3号梯下行命令" )
      I_Contact( "3号梯上行命令" )
   END_RUNG wire#w3
   RUNG wire#powerrail
      I_Contact( "3号梯上行命令" )
      I_Contact( "3号梯下行命令" )
   END_RUNG wire#w3
   RUNG wire#w4
      R_Coil( "3号梯9层下呼" )
   END_RUNG
   RUNG wire#w4
      S_Coil( "DB_GC".HallDownCancel[9] )
   END_RUNG
   RUNG wire#powerrail
      Contact( "8层外呼上行指示灯" )
      Contact( "8层外呼下行指示灯" )
      Contact( "3号梯下行命令" )
      I_Contact( "3号梯上行命令" )
      Contact( "3号梯本层召唤开门信号" )
      wire#w5
      Contact( "3号梯电梯停稳信号" )
      { S7_Templates := "SrcType := Int" } EQ_Contact(in1 := "3号梯当前楼层数", in2 := 8)
      Contact( "8层外呼下行指示灯" )
      wire#w6
      R_Coil( "8层外呼下行指示灯" )
   END_RUNG
   RUNG wire#powerrail
      I_Contact( "8层外呼上行指示灯" )
      Contact( "8层外呼下行指示灯" )
      Contact( "3号梯本层召唤开门信号" )
      Contact( "3号梯下行命令" )
      I_Contact( "3号梯上行命令" )
   END_RUNG wire#w5
   RUNG wire#powerrail
      I_Contact( "3号梯上行命令" )
      I_Contact( "3号梯下行命令" )
   END_RUNG wire#w5
   RUNG wire#w6
      R_Coil( "3号梯8层下呼" )
   END_RUNG
   RUNG wire#w6
      S_Coil( "DB_GC".HallDownCancel[8] )
   END_RUNG
   RUNG wire#powerrail
      Contact( "7层外呼上行指示灯" )
      Contact( "7层外呼下行指示灯" )
      Contact( "3号梯下行命令" )
      I_Contact( "3号梯上行命令" )
      Contact( "3号梯本层召唤开门信号" )
      wire#w7
      Contact( "3号梯电梯停稳信号" )
      { S7_Templates := "SrcType := Int" } EQ_Contact(in1 := "3号梯当前楼层数", in2 := 7)
      Contact( "7层外呼下行指示灯" )
      wire#w8
      R_Coil( "7层外呼下行指示灯" )
   END_RUNG
   RUNG wire#powerrail
      I_Contact( "7层外呼上行指示灯" )
      Contact( "7层外呼下行指示灯" )
      Contact( "3号梯本层召唤开门信号" )
      Contact( "3号梯下行命令" )
      I_Contact( "3号梯上行命令" )
   END_RUNG wire#w7
   RUNG wire#powerrail
      I_Contact( "3号梯上行命令" )
      I_Contact( "3号梯下行命令" )
   END_RUNG wire#w7
   RUNG wire#w8
      R_Coil( "3号梯7层下呼" )
   END_RUNG
   RUNG wire#w8
      S_Coil( "DB_GC".HallDownCancel[7] )
   END_RUNG
   RUNG wire#powerrail
      Contact( "6层外呼上行指示灯" )
      Contact( "6层外呼下行指示灯" )
      Contact( "3号梯下行命令" )
      I_Contact( "3号梯上行命令" )
      Contact( "3号梯本层召唤开门信号" )
      wire#w9
      Contact( "3号梯电梯停稳信号" )
      { S7_Templates := "SrcType := Int" } EQ_Contact(in1 := "3号梯当前楼层数", in2 := 6)
      Contact( "6层外呼下行指示灯" )
      wire#w10
      R_Coil( "6层外呼下行指示灯" )
   END_RUNG
   RUNG wire#powerrail
      I_Contact( "6层外呼上行指示灯" )
      Contact( "6层外呼下行指示灯" )
      Contact( "3号梯本层召唤开门信号" )
      Contact( "3号梯下行命令" )
      I_Contact( "3号梯上行命令" )
   END_RUNG wire#w9
   RUNG wire#powerrail
      I_Contact( "3号梯上行命令" )
      I_Contact( "3号梯下行命令" )
   END_RUNG wire#w9
   RUNG wire#w10
      R_Coil( "3号梯6层下呼" )
   END_RUNG
   RUNG wire#w10
      S_Coil( "DB_GC".HallDownCancel[6] )
   END_RUNG
   RUNG wire#powerrail
      Contact( "5层外呼上行指示灯" )
      Contact( "5层外呼下行指示灯" )
      Contact( "3号梯下行命令" )
      I_Contact( "3号梯上行命令" )
      Contact( "3号梯本层召唤开门信号" )
      wire#w11
      Contact( "3号梯电梯停稳信号" )
      { S7_Templates := "SrcType := Int" } EQ_Contact(in1 := "3号梯当前楼层数", in2 := 5)
      Contact( "5层外呼下行指示灯" )
      wire#w12
      R_Coil( "5层外呼下行指示灯" )
   END_RUNG
   RUNG wire#powerrail
      I_Contact( "5层外呼上行指示灯" )
      Contact( "5层外呼下行指示灯" )
      Contact( "3号梯本层召唤开门信号" )
      Contact( "3号梯下行命令" )
      I_Contact( "3号梯上行命令" )
   END_RUNG wire#w11
   RUNG wire#powerrail
      I_Contact( "3号梯上行命令" )
      I_Contact( "3号梯下行命令" )
   END_RUNG wire#w11
   RUNG wire#w12
      R_Coil( "3号梯5层下呼" )
   END_RUNG
   RUNG wire#w12
      S_Coil( "DB_GC".HallDownCancel[5] )
   END_RUNG
   RUNG wire#powerrail
      Contact( "4层外呼上行指示灯" )
      Contact( "4层外呼下行指示灯" )
      Contact( "3号梯下行命令" )
      I_Contact( "3号梯上行命令" )
      Contact( "3号梯本层召唤开门信号" )
      wire#w13
      Contact( "3号梯电梯停稳信号" )
      { S7_Templates := "SrcType := Int" } EQ_Contact(in1 := "3号梯当前楼层数", in2 := 4)
      Contact( "4层外呼下行指示灯" )
      wire#w14
      R_Coil( "4层外呼下行指示灯" )
   END_RUNG
   RUNG wire#powerrail
      I_Contact( "4层外呼上行指示灯" )
      Contact( "4层外呼下行指示灯" )
      Contact( "3号梯本层召唤开门信号" )
      Contact( "3号梯下行命令" )
      I_Contact( "3号梯上行命令" )
   END_RUNG wire#w13
   RUNG wire#powerrail
      I_Contact( "3号梯上行命令" )
      I_Contact( "3号梯下行命令" )
   END_RUNG wire#w13
   RUNG wire#w14
      R_Coil( "3号梯4层下呼" )
   END_RUNG
   RUNG wire#w14
      S_Coil( "DB_GC".HallDownCancel[4] )
   END_RUNG
   RUNG wire#powerrail
      Contact( "3层外呼上行指示灯" )
      Contact( "3层外呼下行指示灯" )
      Contact( "3号梯下行命令" )
      I_Contact( "3号梯上行命令" )
      Contact( "3号梯本层召唤开门信号" )
      wire#w15
      Contact( "3号梯电梯停稳信号" )
      { S7_Templates := "SrcType := Int" } EQ_Contact(in1 := "3号梯当前楼层数", in2 := 3)
      Contact( "3层外呼下行指示灯" )
      wire#w16
      R_Coil( "3层外呼下行指示灯" )
   END_RUNG
   RUNG wire#powerrail
      I_Contact( "3层外呼上行指示灯" )
      Contact( "3层外呼下行指示灯" )
      Contact( "3号梯本层召唤开门信号" )
      Contact( "3号梯下行命令" )
      I_Contact( "3号梯上行命令" )
   END_RUNG wire#w15
   RUNG wire#powerrail
      I_Contact( "3号梯上行命令" )
      I_Contact( "3号梯下行命令" )
   END_RUNG wire#w15
   RUNG wire#w16
      R_Coil( "3号梯3层下呼" )
   END_RUNG
   RUNG wire#w16
      S_Coil( "DB_GC".HallDownCancel[3] )
   END_RUNG
   RUNG wire#powerrail
      Contact( "2层外呼上行指示灯" )
      Contact( "2层外呼下行指示灯" )
      Contact( "3号梯下行命令" )
      I_Contact( "3号梯上行命令" )
      Contact( "3号梯本层召唤开门信号" )
      wire#w17
      Contact( "3号梯电梯停稳信号" )
      { S7_Templates := "SrcType := Int" } EQ_Contact(in1 := "3号梯当前楼层数", in2 := 2)
      Contact( "2层外呼下行指示灯" )
      wire#w18
      R_Coil( "2层外呼下行指示灯" )
   END_RUNG
   RUNG wire#powerrail
      I_Contact( "2层外呼上行指示灯" )
      Contact( "2层外呼下行指示灯" )
      Contact( "3号梯本层召唤开门信号" )
      Contact( "3号梯下行命令" )
      I_Contact( "3号梯上行命令" )
   END_RUNG wire#w17
   RUNG wire#powerrail
      I_Contact( "3号梯上行命令" )
      I_Contact( "3号梯下行命令" )
   END_RUNG wire#w17
   RUNG wire#w18
      R_Coil( "3号梯2层下呼" )
   END_RUNG
   RUNG wire#w18
      S_Coil( "DB_GC".HallDownCancel[2] )
   END_RUNG
   // the same network as SCL:
   #_w1 := (("10层外呼下行指示灯" AND "3号梯本层召唤开门信号") OR (NOT "3号梯上行命令" AND NOT "3号梯下行命令")) AND ("3号梯当前楼层数" = 10) AND "10层外呼下行指示灯" AND "3号梯电梯停稳信号";
   IF #_w1 THEN
       "10层外呼下行指示灯" := FALSE;
       "3号梯10层下呼" := FALSE;
       "DB_GC".HallDownCancel[10] := TRUE;
   END_IF;
   #_w2 := (("9层外呼上行指示灯" AND "9层外呼下行指示灯" AND "3号梯下行命令" AND NOT "3号梯上行命令" AND "3号梯本层召唤开门信号") OR (NOT "9层外呼上行指示灯" AND "9层外呼下行指示灯" AND "3号梯本层召唤开门信号" AND "3号梯下行命令" AND NOT "3号梯上行命令") OR (NOT "3号梯上行命令" AND NOT "3号梯下行命令")) AND "3号梯电梯停稳信号" AND ("3号梯当前楼层数" = 9) AND "9层外呼下行指示灯";
   IF #_w2 THEN
       "9层外呼下行指示灯" := FALSE;
       "3号梯9层下呼" := FALSE;
       "DB_GC".HallDownCancel[9] := TRUE;
   END_IF;
   #_w3 := (("8层外呼上行指示灯" AND "8层外呼下行指示灯" AND "3号梯下行命令" AND NOT "3号梯上行命令" AND "3号梯本层召唤开门信号") OR (NOT "8层外呼上行指示灯" AND "8层外呼下行指示灯" AND "3号梯本层召唤开门信号" AND "3号梯下行命令" AND NOT "3号梯上行命令") OR (NOT "3号梯上行命令" AND NOT "3号梯下行命令")) AND "3号梯电梯停稳信号" AND ("3号梯当前楼层数" = 8) AND "8层外呼下行指示灯";
   IF #_w3 THEN
       "8层外呼下行指示灯" := FALSE;
       "3号梯8层下呼" := FALSE;
       "DB_GC".HallDownCancel[8] := TRUE;
   END_IF;
   #_w4 := (("7层外呼上行指示灯" AND "7层外呼下行指示灯" AND "3号梯下行命令" AND NOT "3号梯上行命令" AND "3号梯本层召唤开门信号") OR (NOT "7层外呼上行指示灯" AND "7层外呼下行指示灯" AND "3号梯本层召唤开门信号" AND "3号梯下行命令" AND NOT "3号梯上行命令") OR (NOT "3号梯上行命令" AND NOT "3号梯下行命令")) AND "3号梯电梯停稳信号" AND ("3号梯当前楼层数" = 7) AND "7层外呼下行指示灯";
   IF #_w4 THEN
       "7层外呼下行指示灯" := FALSE;
       "3号梯7层下呼" := FALSE;
       "DB_GC".HallDownCancel[7] := TRUE;
   END_IF;
   #_w5 := (("6层外呼上行指示灯" AND "6层外呼下行指示灯" AND "3号梯下行命令" AND NOT "3号梯上行命令" AND "3号梯本层召唤开门信号") OR (NOT "6层外呼上行指示灯" AND "6层外呼下行指示灯" AND "3号梯本层召唤开门信号" AND "3号梯下行命令" AND NOT "3号梯上行命令") OR (NOT "3号梯上行命令" AND NOT "3号梯下行命令")) AND "3号梯电梯停稳信号" AND ("3号梯当前楼层数" = 6) AND "6层外呼下行指示灯";
   IF #_w5 THEN
       "6层外呼下行指示灯" := FALSE;
       "3号梯6层下呼" := FALSE;
       "DB_GC".HallDownCancel[6] := TRUE;
   END_IF;
   #_w6 := (("5层外呼上行指示灯" AND "5层外呼下行指示灯" AND "3号梯下行命令" AND NOT "3号梯上行命令" AND "3号梯本层召唤开门信号") OR (NOT "5层外呼上行指示灯" AND "5层外呼下行指示灯" AND "3号梯本层召唤开门信号" AND "3号梯下行命令" AND NOT "3号梯上行命令") OR (NOT "3号梯上行命令" AND NOT "3号梯下行命令")) AND "3号梯电梯停稳信号" AND ("3号梯当前楼层数" = 5) AND "5层外呼下行指示灯";
   IF #_w6 THEN
       "5层外呼下行指示灯" := FALSE;
       "3号梯5层下呼" := FALSE;
       "DB_GC".HallDownCancel[5] := TRUE;
   END_IF;
   #_w7 := (("4层外呼上行指示灯" AND "4层外呼下行指示灯" AND "3号梯下行命令" AND NOT "3号梯上行命令" AND "3号梯本层召唤开门信号") OR (NOT "4层外呼上行指示灯" AND "4层外呼下行指示灯" AND "3号梯本层召唤开门信号" AND "3号梯下行命令" AND NOT "3号梯上行命令") OR (NOT "3号梯上行命令" AND NOT "3号梯下行命令")) AND "3号梯电梯停稳信号" AND ("3号梯当前楼层数" = 4) AND "4层外呼下行指示灯";
   IF #_w7 THEN
       "4层外呼下行指示灯" := FALSE;
       "3号梯4层下呼" := FALSE;
       "DB_GC".HallDownCancel[4] := TRUE;
   END_IF;
   #_w8 := (("3层外呼上行指示灯" AND "3层外呼下行指示灯" AND "3号梯下行命令" AND NOT "3号梯上行命令" AND "3号梯本层召唤开门信号") OR (NOT "3层外呼上行指示灯" AND "3层外呼下行指示灯" AND "3号梯本层召唤开门信号" AND "3号梯下行命令" AND NOT "3号梯上行命令") OR (NOT "3号梯上行命令" AND NOT "3号梯下行命令")) AND "3号梯电梯停稳信号" AND ("3号梯当前楼层数" = 3) AND "3层外呼下行指示灯";
   IF #_w8 THEN
       "3层外呼下行指示灯" := FALSE;
       "3号梯3层下呼" := FALSE;
       "DB_GC".HallDownCancel[3] := TRUE;
   END_IF;
   #_w9 := (("2层外呼上行指示灯" AND "2层外呼下行指示灯" AND "3号梯下行命令" AND NOT "3号梯上行命令" AND "3号梯本层召唤开门信号") OR (NOT "2层外呼上行指示灯" AND "2层外呼下行指示灯" AND "3号梯本层召唤开门信号" AND "3号梯下行命令" AND NOT "3号梯上行命令") OR (NOT "3号梯上行命令" AND NOT "3号梯下行命令")) AND "3号梯电梯停稳信号" AND ("3号梯当前楼层数" = 2) AND "2层外呼下行指示灯";
   IF #_w9 THEN
       "2层外呼下行指示灯" := FALSE;
       "3号梯2层下呼" := FALSE;
       "DB_GC".HallDownCancel[2] := TRUE;
   END_IF;
END_REGION

REGION Network 2: 3号梯终止上呼
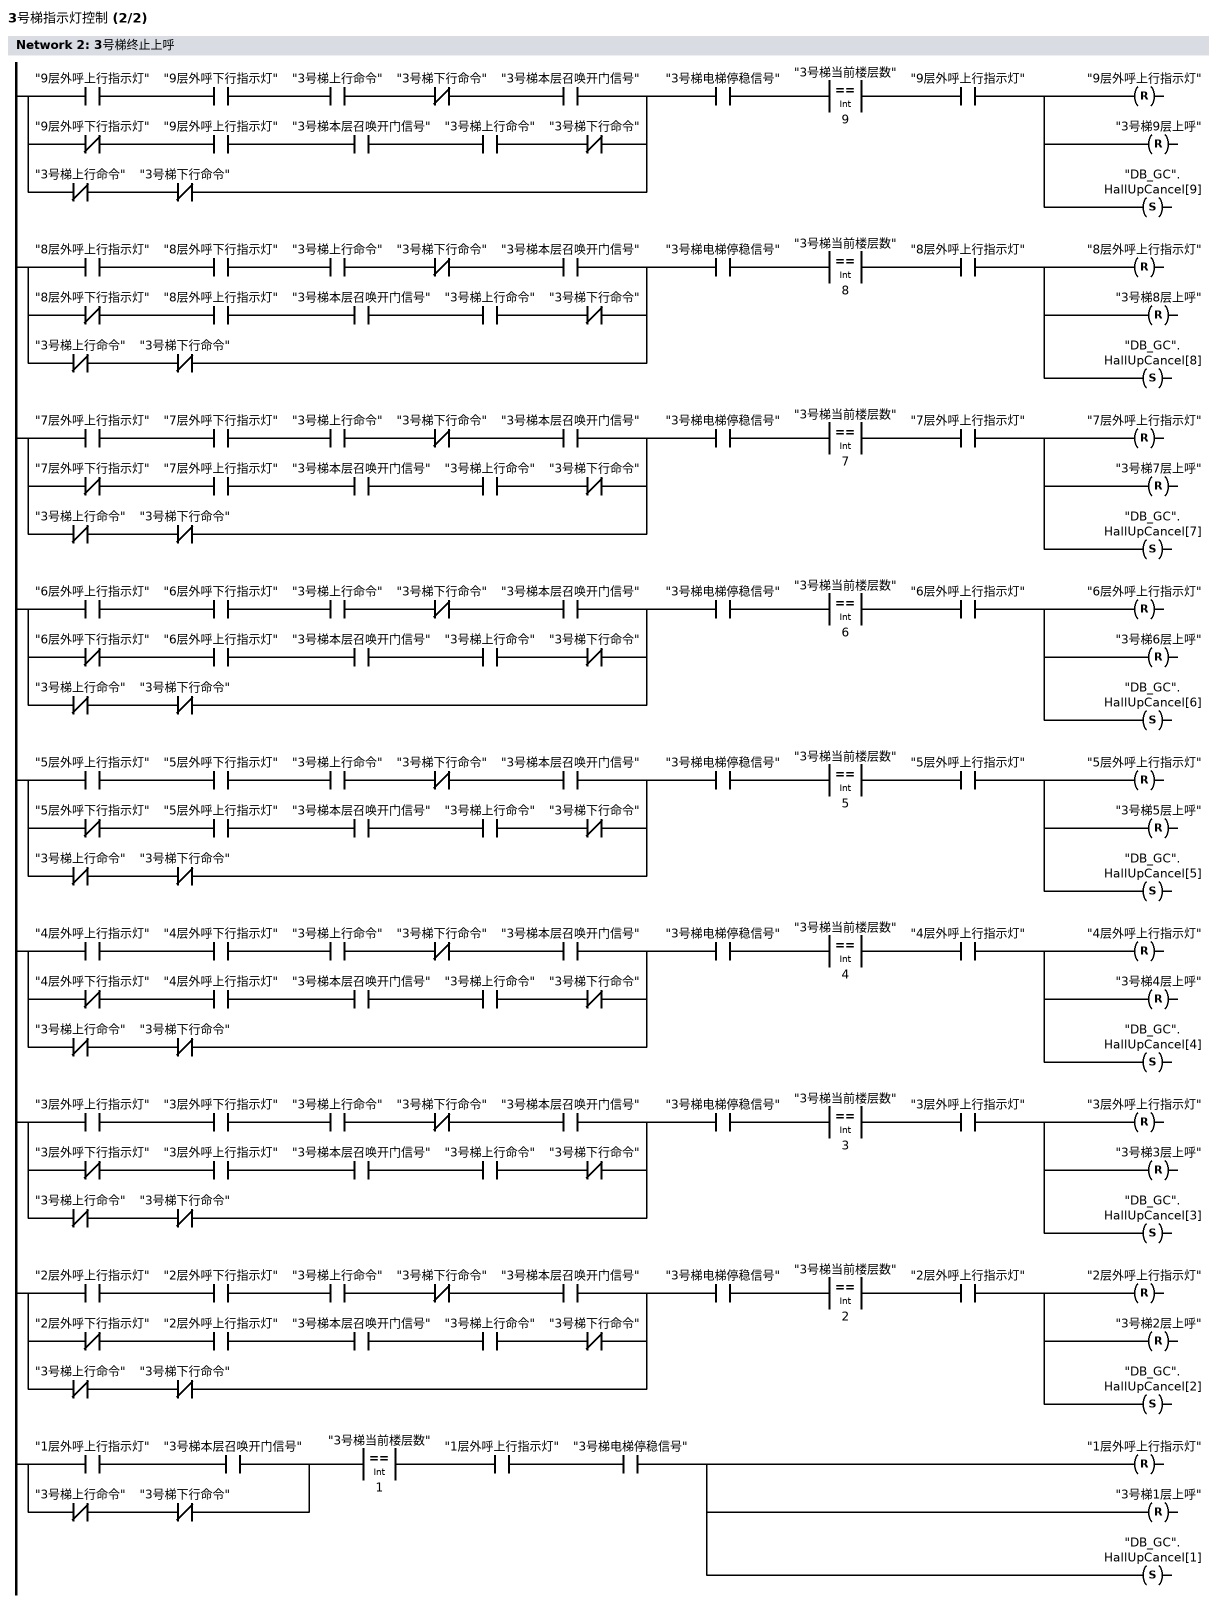
   RUNG wire#powerrail
      Contact( "9层外呼上行指示灯" )
      Contact( "9层外呼下行指示灯" )
      Contact( "3号梯上行命令" )
      I_Contact( "3号梯下行命令" )
      Contact( "3号梯本层召唤开门信号" )
      wire#w1
      Contact( "3号梯电梯停稳信号" )
      { S7_Templates := "SrcType := Int" } EQ_Contact(in1 := "3号梯当前楼层数", in2 := 9)
      Contact( "9层外呼上行指示灯" )
      wire#w2
      R_Coil( "9层外呼上行指示灯" )
   END_RUNG
   RUNG wire#powerrail
      I_Contact( "9层外呼下行指示灯" )
      Contact( "9层外呼上行指示灯" )
      Contact( "3号梯本层召唤开门信号" )
      Contact( "3号梯上行命令" )
      I_Contact( "3号梯下行命令" )
   END_RUNG wire#w1
   RUNG wire#powerrail
      I_Contact( "3号梯上行命令" )
      I_Contact( "3号梯下行命令" )
   END_RUNG wire#w1
   RUNG wire#w2
      R_Coil( "3号梯9层上呼" )
   END_RUNG
   RUNG wire#w2
      S_Coil( "DB_GC".HallUpCancel[9] )
   END_RUNG
   RUNG wire#powerrail
      Contact( "8层外呼上行指示灯" )
      Contact( "8层外呼下行指示灯" )
      Contact( "3号梯上行命令" )
      I_Contact( "3号梯下行命令" )
      Contact( "3号梯本层召唤开门信号" )
      wire#w3
      Contact( "3号梯电梯停稳信号" )
      { S7_Templates := "SrcType := Int" } EQ_Contact(in1 := "3号梯当前楼层数", in2 := 8)
      Contact( "8层外呼上行指示灯" )
      wire#w4
      R_Coil( "8层外呼上行指示灯" )
   END_RUNG
   RUNG wire#powerrail
      I_Contact( "8层外呼下行指示灯" )
      Contact( "8层外呼上行指示灯" )
      Contact( "3号梯本层召唤开门信号" )
      Contact( "3号梯上行命令" )
      I_Contact( "3号梯下行命令" )
   END_RUNG wire#w3
   RUNG wire#powerrail
      I_Contact( "3号梯上行命令" )
      I_Contact( "3号梯下行命令" )
   END_RUNG wire#w3
   RUNG wire#w4
      R_Coil( "3号梯8层上呼" )
   END_RUNG
   RUNG wire#w4
      S_Coil( "DB_GC".HallUpCancel[8] )
   END_RUNG
   RUNG wire#powerrail
      Contact( "7层外呼上行指示灯" )
      Contact( "7层外呼下行指示灯" )
      Contact( "3号梯上行命令" )
      I_Contact( "3号梯下行命令" )
      Contact( "3号梯本层召唤开门信号" )
      wire#w5
      Contact( "3号梯电梯停稳信号" )
      { S7_Templates := "SrcType := Int" } EQ_Contact(in1 := "3号梯当前楼层数", in2 := 7)
      Contact( "7层外呼上行指示灯" )
      wire#w6
      R_Coil( "7层外呼上行指示灯" )
   END_RUNG
   RUNG wire#powerrail
      I_Contact( "7层外呼下行指示灯" )
      Contact( "7层外呼上行指示灯" )
      Contact( "3号梯本层召唤开门信号" )
      Contact( "3号梯上行命令" )
      I_Contact( "3号梯下行命令" )
   END_RUNG wire#w5
   RUNG wire#powerrail
      I_Contact( "3号梯上行命令" )
      I_Contact( "3号梯下行命令" )
   END_RUNG wire#w5
   RUNG wire#w6
      R_Coil( "3号梯7层上呼" )
   END_RUNG
   RUNG wire#w6
      S_Coil( "DB_GC".HallUpCancel[7] )
   END_RUNG
   RUNG wire#powerrail
      Contact( "6层外呼上行指示灯" )
      Contact( "6层外呼下行指示灯" )
      Contact( "3号梯上行命令" )
      I_Contact( "3号梯下行命令" )
      Contact( "3号梯本层召唤开门信号" )
      wire#w7
      Contact( "3号梯电梯停稳信号" )
      { S7_Templates := "SrcType := Int" } EQ_Contact(in1 := "3号梯当前楼层数", in2 := 6)
      Contact( "6层外呼上行指示灯" )
      wire#w8
      R_Coil( "6层外呼上行指示灯" )
   END_RUNG
   RUNG wire#powerrail
      I_Contact( "6层外呼下行指示灯" )
      Contact( "6层外呼上行指示灯" )
      Contact( "3号梯本层召唤开门信号" )
      Contact( "3号梯上行命令" )
      I_Contact( "3号梯下行命令" )
   END_RUNG wire#w7
   RUNG wire#powerrail
      I_Contact( "3号梯上行命令" )
      I_Contact( "3号梯下行命令" )
   END_RUNG wire#w7
   RUNG wire#w8
      R_Coil( "3号梯6层上呼" )
   END_RUNG
   RUNG wire#w8
      S_Coil( "DB_GC".HallUpCancel[6] )
   END_RUNG
   RUNG wire#powerrail
      Contact( "5层外呼上行指示灯" )
      Contact( "5层外呼下行指示灯" )
      Contact( "3号梯上行命令" )
      I_Contact( "3号梯下行命令" )
      Contact( "3号梯本层召唤开门信号" )
      wire#w9
      Contact( "3号梯电梯停稳信号" )
      { S7_Templates := "SrcType := Int" } EQ_Contact(in1 := "3号梯当前楼层数", in2 := 5)
      Contact( "5层外呼上行指示灯" )
      wire#w10
      R_Coil( "5层外呼上行指示灯" )
   END_RUNG
   RUNG wire#powerrail
      I_Contact( "5层外呼下行指示灯" )
      Contact( "5层外呼上行指示灯" )
      Contact( "3号梯本层召唤开门信号" )
      Contact( "3号梯上行命令" )
      I_Contact( "3号梯下行命令" )
   END_RUNG wire#w9
   RUNG wire#powerrail
      I_Contact( "3号梯上行命令" )
      I_Contact( "3号梯下行命令" )
   END_RUNG wire#w9
   RUNG wire#w10
      R_Coil( "3号梯5层上呼" )
   END_RUNG
   RUNG wire#w10
      S_Coil( "DB_GC".HallUpCancel[5] )
   END_RUNG
   RUNG wire#powerrail
      Contact( "4层外呼上行指示灯" )
      Contact( "4层外呼下行指示灯" )
      Contact( "3号梯上行命令" )
      I_Contact( "3号梯下行命令" )
      Contact( "3号梯本层召唤开门信号" )
      wire#w11
      Contact( "3号梯电梯停稳信号" )
      { S7_Templates := "SrcType := Int" } EQ_Contact(in1 := "3号梯当前楼层数", in2 := 4)
      Contact( "4层外呼上行指示灯" )
      wire#w12
      R_Coil( "4层外呼上行指示灯" )
   END_RUNG
   RUNG wire#powerrail
      I_Contact( "4层外呼下行指示灯" )
      Contact( "4层外呼上行指示灯" )
      Contact( "3号梯本层召唤开门信号" )
      Contact( "3号梯上行命令" )
      I_Contact( "3号梯下行命令" )
   END_RUNG wire#w11
   RUNG wire#powerrail
      I_Contact( "3号梯上行命令" )
      I_Contact( "3号梯下行命令" )
   END_RUNG wire#w11
   RUNG wire#w12
      R_Coil( "3号梯4层上呼" )
   END_RUNG
   RUNG wire#w12
      S_Coil( "DB_GC".HallUpCancel[4] )
   END_RUNG
   RUNG wire#powerrail
      Contact( "3层外呼上行指示灯" )
      Contact( "3层外呼下行指示灯" )
      Contact( "3号梯上行命令" )
      I_Contact( "3号梯下行命令" )
      Contact( "3号梯本层召唤开门信号" )
      wire#w13
      Contact( "3号梯电梯停稳信号" )
      { S7_Templates := "SrcType := Int" } EQ_Contact(in1 := "3号梯当前楼层数", in2 := 3)
      Contact( "3层外呼上行指示灯" )
      wire#w14
      R_Coil( "3层外呼上行指示灯" )
   END_RUNG
   RUNG wire#powerrail
      I_Contact( "3层外呼下行指示灯" )
      Contact( "3层外呼上行指示灯" )
      Contact( "3号梯本层召唤开门信号" )
      Contact( "3号梯上行命令" )
      I_Contact( "3号梯下行命令" )
   END_RUNG wire#w13
   RUNG wire#powerrail
      I_Contact( "3号梯上行命令" )
      I_Contact( "3号梯下行命令" )
   END_RUNG wire#w13
   RUNG wire#w14
      R_Coil( "3号梯3层上呼" )
   END_RUNG
   RUNG wire#w14
      S_Coil( "DB_GC".HallUpCancel[3] )
   END_RUNG
   RUNG wire#powerrail
      Contact( "2层外呼上行指示灯" )
      Contact( "2层外呼下行指示灯" )
      Contact( "3号梯上行命令" )
      I_Contact( "3号梯下行命令" )
      Contact( "3号梯本层召唤开门信号" )
      wire#w15
      Contact( "3号梯电梯停稳信号" )
      { S7_Templates := "SrcType := Int" } EQ_Contact(in1 := "3号梯当前楼层数", in2 := 2)
      Contact( "2层外呼上行指示灯" )
      wire#w16
      R_Coil( "2层外呼上行指示灯" )
   END_RUNG
   RUNG wire#powerrail
      I_Contact( "2层外呼下行指示灯" )
      Contact( "2层外呼上行指示灯" )
      Contact( "3号梯本层召唤开门信号" )
      Contact( "3号梯上行命令" )
      I_Contact( "3号梯下行命令" )
   END_RUNG wire#w15
   RUNG wire#powerrail
      I_Contact( "3号梯上行命令" )
      I_Contact( "3号梯下行命令" )
   END_RUNG wire#w15
   RUNG wire#w16
      R_Coil( "3号梯2层上呼" )
   END_RUNG
   RUNG wire#w16
      S_Coil( "DB_GC".HallUpCancel[2] )
   END_RUNG
   RUNG wire#powerrail
      Contact( "1层外呼上行指示灯" )
      Contact( "3号梯本层召唤开门信号" )
      wire#w17
      { S7_Templates := "SrcType := Int" } EQ_Contact(in1 := "3号梯当前楼层数", in2 := 1)
      Contact( "1层外呼上行指示灯" )
      Contact( "3号梯电梯停稳信号" )
      wire#w18
      R_Coil( "1层外呼上行指示灯" )
   END_RUNG
   RUNG wire#powerrail
      I_Contact( "3号梯上行命令" )
      I_Contact( "3号梯下行命令" )
   END_RUNG wire#w17
   RUNG wire#w18
      R_Coil( "3号梯1层上呼" )
   END_RUNG
   RUNG wire#w18
      S_Coil( "DB_GC".HallUpCancel[1] )
   END_RUNG
   // the same network as SCL:
   #_w1 := (("9层外呼上行指示灯" AND "9层外呼下行指示灯" AND "3号梯上行命令" AND NOT "3号梯下行命令" AND "3号梯本层召唤开门信号") OR (NOT "9层外呼下行指示灯" AND "9层外呼上行指示灯" AND "3号梯本层召唤开门信号" AND "3号梯上行命令" AND NOT "3号梯下行命令") OR (NOT "3号梯上行命令" AND NOT "3号梯下行命令")) AND "3号梯电梯停稳信号" AND ("3号梯当前楼层数" = 9) AND "9层外呼上行指示灯";
   IF #_w1 THEN
       "9层外呼上行指示灯" := FALSE;
       "3号梯9层上呼" := FALSE;
       "DB_GC".HallUpCancel[9] := TRUE;
   END_IF;
   #_w2 := (("8层外呼上行指示灯" AND "8层外呼下行指示灯" AND "3号梯上行命令" AND NOT "3号梯下行命令" AND "3号梯本层召唤开门信号") OR (NOT "8层外呼下行指示灯" AND "8层外呼上行指示灯" AND "3号梯本层召唤开门信号" AND "3号梯上行命令" AND NOT "3号梯下行命令") OR (NOT "3号梯上行命令" AND NOT "3号梯下行命令")) AND "3号梯电梯停稳信号" AND ("3号梯当前楼层数" = 8) AND "8层外呼上行指示灯";
   IF #_w2 THEN
       "8层外呼上行指示灯" := FALSE;
       "3号梯8层上呼" := FALSE;
       "DB_GC".HallUpCancel[8] := TRUE;
   END_IF;
   #_w3 := (("7层外呼上行指示灯" AND "7层外呼下行指示灯" AND "3号梯上行命令" AND NOT "3号梯下行命令" AND "3号梯本层召唤开门信号") OR (NOT "7层外呼下行指示灯" AND "7层外呼上行指示灯" AND "3号梯本层召唤开门信号" AND "3号梯上行命令" AND NOT "3号梯下行命令") OR (NOT "3号梯上行命令" AND NOT "3号梯下行命令")) AND "3号梯电梯停稳信号" AND ("3号梯当前楼层数" = 7) AND "7层外呼上行指示灯";
   IF #_w3 THEN
       "7层外呼上行指示灯" := FALSE;
       "3号梯7层上呼" := FALSE;
       "DB_GC".HallUpCancel[7] := TRUE;
   END_IF;
   #_w4 := (("6层外呼上行指示灯" AND "6层外呼下行指示灯" AND "3号梯上行命令" AND NOT "3号梯下行命令" AND "3号梯本层召唤开门信号") OR (NOT "6层外呼下行指示灯" AND "6层外呼上行指示灯" AND "3号梯本层召唤开门信号" AND "3号梯上行命令" AND NOT "3号梯下行命令") OR (NOT "3号梯上行命令" AND NOT "3号梯下行命令")) AND "3号梯电梯停稳信号" AND ("3号梯当前楼层数" = 6) AND "6层外呼上行指示灯";
   IF #_w4 THEN
       "6层外呼上行指示灯" := FALSE;
       "3号梯6层上呼" := FALSE;
       "DB_GC".HallUpCancel[6] := TRUE;
   END_IF;
   #_w5 := (("5层外呼上行指示灯" AND "5层外呼下行指示灯" AND "3号梯上行命令" AND NOT "3号梯下行命令" AND "3号梯本层召唤开门信号") OR (NOT "5层外呼下行指示灯" AND "5层外呼上行指示灯" AND "3号梯本层召唤开门信号" AND "3号梯上行命令" AND NOT "3号梯下行命令") OR (NOT "3号梯上行命令" AND NOT "3号梯下行命令")) AND "3号梯电梯停稳信号" AND ("3号梯当前楼层数" = 5) AND "5层外呼上行指示灯";
   IF #_w5 THEN
       "5层外呼上行指示灯" := FALSE;
       "3号梯5层上呼" := FALSE;
       "DB_GC".HallUpCancel[5] := TRUE;
   END_IF;
   #_w6 := (("4层外呼上行指示灯" AND "4层外呼下行指示灯" AND "3号梯上行命令" AND NOT "3号梯下行命令" AND "3号梯本层召唤开门信号") OR (NOT "4层外呼下行指示灯" AND "4层外呼上行指示灯" AND "3号梯本层召唤开门信号" AND "3号梯上行命令" AND NOT "3号梯下行命令") OR (NOT "3号梯上行命令" AND NOT "3号梯下行命令")) AND "3号梯电梯停稳信号" AND ("3号梯当前楼层数" = 4) AND "4层外呼上行指示灯";
   IF #_w6 THEN
       "4层外呼上行指示灯" := FALSE;
       "3号梯4层上呼" := FALSE;
       "DB_GC".HallUpCancel[4] := TRUE;
   END_IF;
   #_w7 := (("3层外呼上行指示灯" AND "3层外呼下行指示灯" AND "3号梯上行命令" AND NOT "3号梯下行命令" AND "3号梯本层召唤开门信号") OR (NOT "3层外呼下行指示灯" AND "3层外呼上行指示灯" AND "3号梯本层召唤开门信号" AND "3号梯上行命令" AND NOT "3号梯下行命令") OR (NOT "3号梯上行命令" AND NOT "3号梯下行命令")) AND "3号梯电梯停稳信号" AND ("3号梯当前楼层数" = 3) AND "3层外呼上行指示灯";
   IF #_w7 THEN
       "3层外呼上行指示灯" := FALSE;
       "3号梯3层上呼" := FALSE;
       "DB_GC".HallUpCancel[3] := TRUE;
   END_IF;
   #_w8 := (("2层外呼上行指示灯" AND "2层外呼下行指示灯" AND "3号梯上行命令" AND NOT "3号梯下行命令" AND "3号梯本层召唤开门信号") OR (NOT "2层外呼下行指示灯" AND "2层外呼上行指示灯" AND "3号梯本层召唤开门信号" AND "3号梯上行命令" AND NOT "3号梯下行命令") OR (NOT "3号梯上行命令" AND NOT "3号梯下行命令")) AND "3号梯电梯停稳信号" AND ("3号梯当前楼层数" = 2) AND "2层外呼上行指示灯";
   IF #_w8 THEN
       "2层外呼上行指示灯" := FALSE;
       "3号梯2层上呼" := FALSE;
       "DB_GC".HallUpCancel[2] := TRUE;
   END_IF;
   #_w9 := (("1层外呼上行指示灯" AND "3号梯本层召唤开门信号") OR (NOT "3号梯上行命令" AND NOT "3号梯下行命令")) AND ("3号梯当前楼层数" = 1) AND "1层外呼上行指示灯" AND "3号梯电梯停稳信号";
   IF #_w9 THEN
       "1层外呼上行指示灯" := FALSE;
       "3号梯1层上呼" := FALSE;
       "DB_GC".HallUpCancel[1] := TRUE;
   END_IF;
END_REGION
END_FUNCTION

FUNCTION "1号梯目标楼层登记" : Void   // FC15, LAD
{ S7_Optimized_Access := 'TRUE' }
VERSION : 0.1
BEGIN

REGION Network 1: 楼层登记
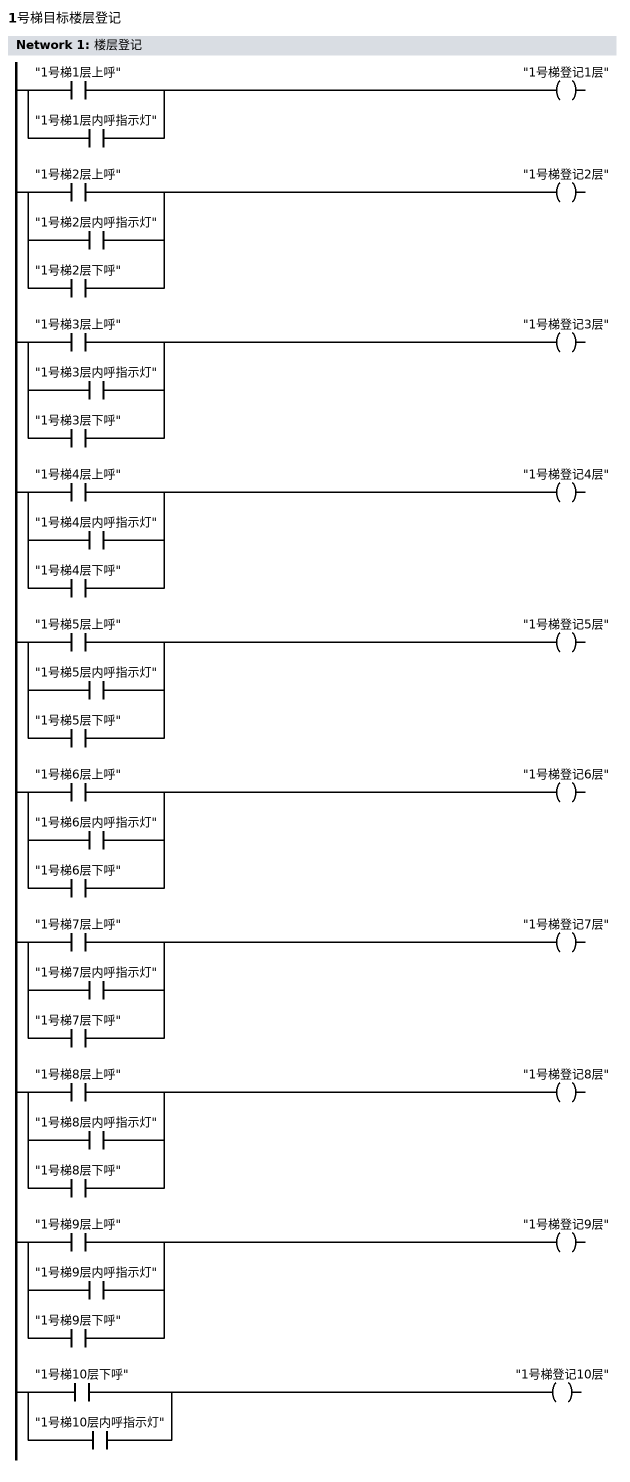
   RUNG wire#powerrail
      Contact( "1号梯1层上呼" )
      wire#w1
      Coil( "1号梯登记1层" )
   END_RUNG
   RUNG wire#powerrail
      Contact( "1号梯1层内呼指示灯" )
   END_RUNG wire#w1
   RUNG wire#powerrail
      Contact( "1号梯2层上呼" )
      wire#w2
      Coil( "1号梯登记2层" )
   END_RUNG
   RUNG wire#powerrail
      Contact( "1号梯2层内呼指示灯" )
   END_RUNG wire#w2
   RUNG wire#powerrail
      Contact( "1号梯2层下呼" )
   END_RUNG wire#w2
   RUNG wire#powerrail
      Contact( "1号梯3层上呼" )
      wire#w3
      Coil( "1号梯登记3层" )
   END_RUNG
   RUNG wire#powerrail
      Contact( "1号梯3层内呼指示灯" )
   END_RUNG wire#w3
   RUNG wire#powerrail
      Contact( "1号梯3层下呼" )
   END_RUNG wire#w3
   RUNG wire#powerrail
      Contact( "1号梯4层上呼" )
      wire#w4
      Coil( "1号梯登记4层" )
   END_RUNG
   RUNG wire#powerrail
      Contact( "1号梯4层内呼指示灯" )
   END_RUNG wire#w4
   RUNG wire#powerrail
      Contact( "1号梯4层下呼" )
   END_RUNG wire#w4
   RUNG wire#powerrail
      Contact( "1号梯5层上呼" )
      wire#w5
      Coil( "1号梯登记5层" )
   END_RUNG
   RUNG wire#powerrail
      Contact( "1号梯5层内呼指示灯" )
   END_RUNG wire#w5
   RUNG wire#powerrail
      Contact( "1号梯5层下呼" )
   END_RUNG wire#w5
   RUNG wire#powerrail
      Contact( "1号梯6层上呼" )
      wire#w6
      Coil( "1号梯登记6层" )
   END_RUNG
   RUNG wire#powerrail
      Contact( "1号梯6层内呼指示灯" )
   END_RUNG wire#w6
   RUNG wire#powerrail
      Contact( "1号梯6层下呼" )
   END_RUNG wire#w6
   RUNG wire#powerrail
      Contact( "1号梯7层上呼" )
      wire#w7
      Coil( "1号梯登记7层" )
   END_RUNG
   RUNG wire#powerrail
      Contact( "1号梯7层内呼指示灯" )
   END_RUNG wire#w7
   RUNG wire#powerrail
      Contact( "1号梯7层下呼" )
   END_RUNG wire#w7
   RUNG wire#powerrail
      Contact( "1号梯8层上呼" )
      wire#w8
      Coil( "1号梯登记8层" )
   END_RUNG
   RUNG wire#powerrail
      Contact( "1号梯8层内呼指示灯" )
   END_RUNG wire#w8
   RUNG wire#powerrail
      Contact( "1号梯8层下呼" )
   END_RUNG wire#w8
   RUNG wire#powerrail
      Contact( "1号梯9层上呼" )
      wire#w9
      Coil( "1号梯登记9层" )
   END_RUNG
   RUNG wire#powerrail
      Contact( "1号梯9层内呼指示灯" )
   END_RUNG wire#w9
   RUNG wire#powerrail
      Contact( "1号梯9层下呼" )
   END_RUNG wire#w9
   RUNG wire#powerrail
      Contact( "1号梯10层下呼" )
      wire#w10
      Coil( "1号梯登记10层" )
   END_RUNG
   RUNG wire#powerrail
      Contact( "1号梯10层内呼指示灯" )
   END_RUNG wire#w10
   // the same network as SCL:
   "1号梯登记1层" := "1号梯1层上呼" OR "1号梯1层内呼指示灯";
   "1号梯登记2层" := "1号梯2层上呼" OR "1号梯2层内呼指示灯" OR "1号梯2层下呼";
   "1号梯登记3层" := "1号梯3层上呼" OR "1号梯3层内呼指示灯" OR "1号梯3层下呼";
   "1号梯登记4层" := "1号梯4层上呼" OR "1号梯4层内呼指示灯" OR "1号梯4层下呼";
   "1号梯登记5层" := "1号梯5层上呼" OR "1号梯5层内呼指示灯" OR "1号梯5层下呼";
   "1号梯登记6层" := "1号梯6层上呼" OR "1号梯6层内呼指示灯" OR "1号梯6层下呼";
   "1号梯登记7层" := "1号梯7层上呼" OR "1号梯7层内呼指示灯" OR "1号梯7层下呼";
   "1号梯登记8层" := "1号梯8层上呼" OR "1号梯8层内呼指示灯" OR "1号梯8层下呼";
   "1号梯登记9层" := "1号梯9层上呼" OR "1号梯9层内呼指示灯" OR "1号梯9层下呼";
   "1号梯登记10层" := "1号梯10层下呼" OR "1号梯10层内呼指示灯";
END_REGION
END_FUNCTION

FUNCTION "1号梯自动选向" : Void   // FC16, LAD
{ S7_Optimized_Access := 'TRUE' }
VERSION : 0.1
BEGIN

REGION Network 1: 上行选向
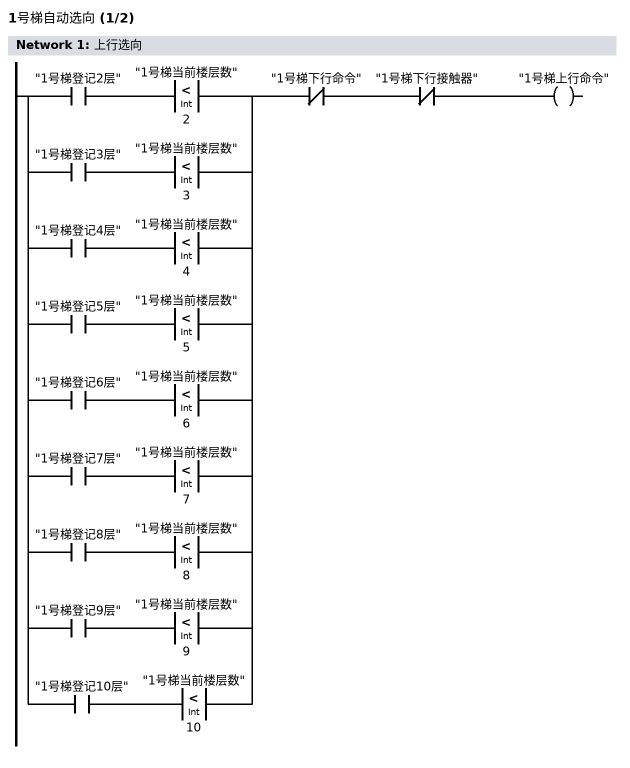
   RUNG wire#powerrail
      Contact( "1号梯登记2层" )
      { S7_Templates := "SrcType := Int" } LT_Contact(in1 := "1号梯当前楼层数", in2 := 2)
      wire#w1
      I_Contact( "1号梯下行命令" )
      I_Contact( "1号梯下行接触器" )
      Coil( "1号梯上行命令" )
   END_RUNG
   RUNG wire#powerrail
      Contact( "1号梯登记3层" )
      { S7_Templates := "SrcType := Int" } LT_Contact(in1 := "1号梯当前楼层数", in2 := 3)
   END_RUNG wire#w1
   RUNG wire#powerrail
      Contact( "1号梯登记4层" )
      { S7_Templates := "SrcType := Int" } LT_Contact(in1 := "1号梯当前楼层数", in2 := 4)
   END_RUNG wire#w1
   RUNG wire#powerrail
      Contact( "1号梯登记5层" )
      { S7_Templates := "SrcType := Int" } LT_Contact(in1 := "1号梯当前楼层数", in2 := 5)
   END_RUNG wire#w1
   RUNG wire#powerrail
      Contact( "1号梯登记6层" )
      { S7_Templates := "SrcType := Int" } LT_Contact(in1 := "1号梯当前楼层数", in2 := 6)
   END_RUNG wire#w1
   RUNG wire#powerrail
      Contact( "1号梯登记7层" )
      { S7_Templates := "SrcType := Int" } LT_Contact(in1 := "1号梯当前楼层数", in2 := 7)
   END_RUNG wire#w1
   RUNG wire#powerrail
      Contact( "1号梯登记8层" )
      { S7_Templates := "SrcType := Int" } LT_Contact(in1 := "1号梯当前楼层数", in2 := 8)
   END_RUNG wire#w1
   RUNG wire#powerrail
      Contact( "1号梯登记9层" )
      { S7_Templates := "SrcType := Int" } LT_Contact(in1 := "1号梯当前楼层数", in2 := 9)
   END_RUNG wire#w1
   RUNG wire#powerrail
      Contact( "1号梯登记10层" )
      { S7_Templates := "SrcType := Int" } LT_Contact(in1 := "1号梯当前楼层数", in2 := 10)
   END_RUNG wire#w1
   // the same network as SCL:
   "1号梯上行命令" := (("1号梯登记2层" AND ("1号梯当前楼层数" < 2)) OR ("1号梯登记3层" AND ("1号梯当前楼层数" < 3)) OR ("1号梯登记4层" AND ("1号梯当前楼层数" < 4)) OR ("1号梯登记5层" AND ("1号梯当前楼层数" < 5)) OR ("1号梯登记6层" AND ("1号梯当前楼层数" < 6)) OR ("1号梯登记7层" AND ("1号梯当前楼层数" < 7)) OR ("1号梯登记8层" AND ("1号梯当前楼层数" < 8)) OR ("1号梯登记9层" AND ("1号梯当前楼层数" < 9)) OR ("1号梯登记10层" AND ("1号梯当前楼层数" < 10))) AND NOT "1号梯下行命令" AND NOT "1号梯下行接触器";
END_REGION

REGION Network 2: 下行选向
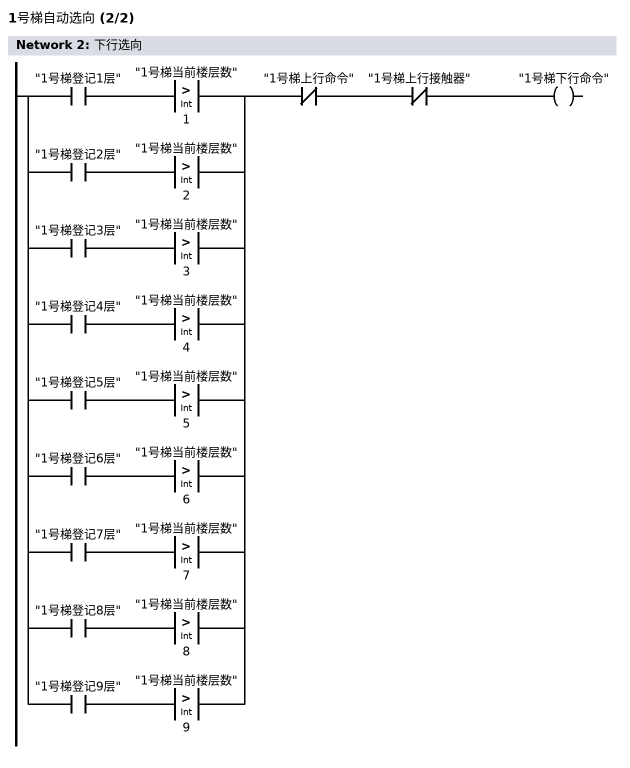
   RUNG wire#powerrail
      Contact( "1号梯登记1层" )
      { S7_Templates := "SrcType := Int" } GT_Contact(in1 := "1号梯当前楼层数", in2 := 1)
      wire#w1
      I_Contact( "1号梯上行命令" )
      I_Contact( "1号梯上行接触器" )
      Coil( "1号梯下行命令" )
   END_RUNG
   RUNG wire#powerrail
      Contact( "1号梯登记2层" )
      { S7_Templates := "SrcType := Int" } GT_Contact(in1 := "1号梯当前楼层数", in2 := 2)
   END_RUNG wire#w1
   RUNG wire#powerrail
      Contact( "1号梯登记3层" )
      { S7_Templates := "SrcType := Int" } GT_Contact(in1 := "1号梯当前楼层数", in2 := 3)
   END_RUNG wire#w1
   RUNG wire#powerrail
      Contact( "1号梯登记4层" )
      { S7_Templates := "SrcType := Int" } GT_Contact(in1 := "1号梯当前楼层数", in2 := 4)
   END_RUNG wire#w1
   RUNG wire#powerrail
      Contact( "1号梯登记5层" )
      { S7_Templates := "SrcType := Int" } GT_Contact(in1 := "1号梯当前楼层数", in2 := 5)
   END_RUNG wire#w1
   RUNG wire#powerrail
      Contact( "1号梯登记6层" )
      { S7_Templates := "SrcType := Int" } GT_Contact(in1 := "1号梯当前楼层数", in2 := 6)
   END_RUNG wire#w1
   RUNG wire#powerrail
      Contact( "1号梯登记7层" )
      { S7_Templates := "SrcType := Int" } GT_Contact(in1 := "1号梯当前楼层数", in2 := 7)
   END_RUNG wire#w1
   RUNG wire#powerrail
      Contact( "1号梯登记8层" )
      { S7_Templates := "SrcType := Int" } GT_Contact(in1 := "1号梯当前楼层数", in2 := 8)
   END_RUNG wire#w1
   RUNG wire#powerrail
      Contact( "1号梯登记9层" )
      { S7_Templates := "SrcType := Int" } GT_Contact(in1 := "1号梯当前楼层数", in2 := 9)
   END_RUNG wire#w1
   // the same network as SCL:
   "1号梯下行命令" := (("1号梯登记1层" AND ("1号梯当前楼层数" > 1)) OR ("1号梯登记2层" AND ("1号梯当前楼层数" > 2)) OR ("1号梯登记3层" AND ("1号梯当前楼层数" > 3)) OR ("1号梯登记4层" AND ("1号梯当前楼层数" > 4)) OR ("1号梯登记5层" AND ("1号梯当前楼层数" > 5)) OR ("1号梯登记6层" AND ("1号梯当前楼层数" > 6)) OR ("1号梯登记7层" AND ("1号梯当前楼层数" > 7)) OR ("1号梯登记8层" AND ("1号梯当前楼层数" > 8)) OR ("1号梯登记9层" AND ("1号梯当前楼层数" > 9))) AND NOT "1号梯上行命令" AND NOT "1号梯上行接触器";
END_REGION
END_FUNCTION

FUNCTION "1号梯启停" : Void   // FC17, LAD
{ S7_Optimized_Access := 'TRUE' }
VERSION : 0.1
   VAR_TEMP   // added for the SCL form of the ladder/FBD networks
      _w1 : Bool;
   END_VAR
BEGIN

REGION Network 1: 上行
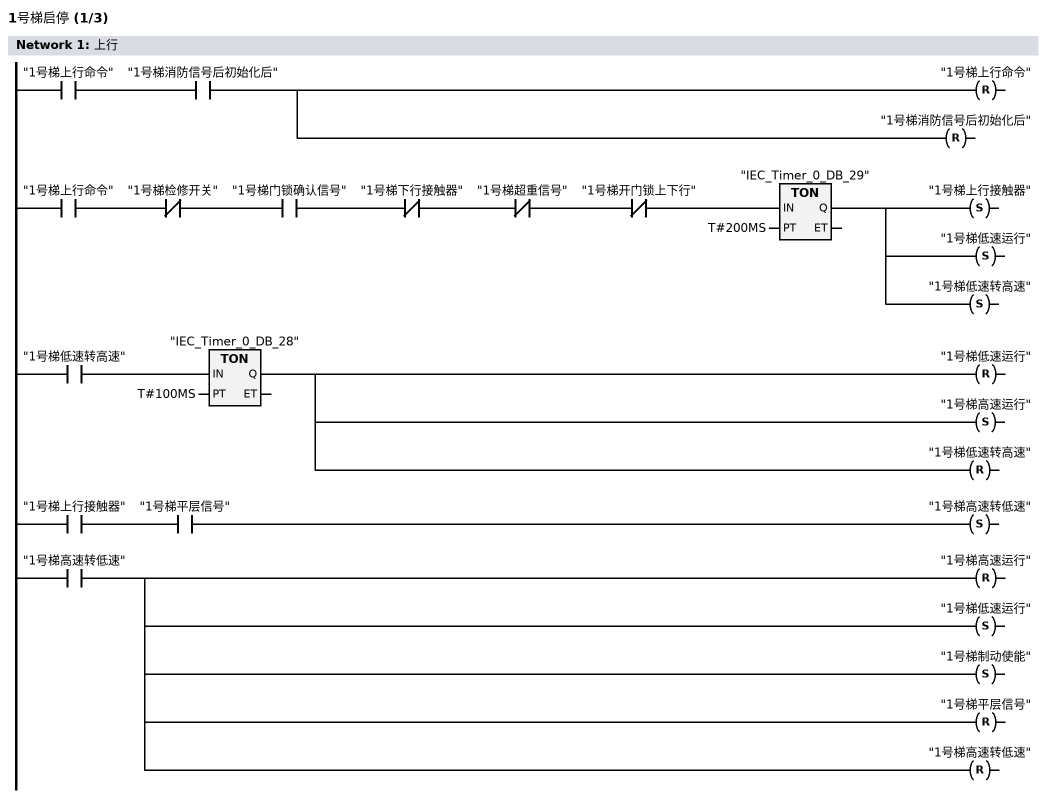
   #_w1 := "1号梯上行命令" AND "1号梯消防信号后初始化后";
   IF #_w1 THEN
       "1号梯上行命令" := FALSE;
       "1号梯消防信号后初始化后" := FALSE;
   END_IF;
   "IEC_Timer_0_DB_29".TON(IN := "1号梯上行命令" AND NOT "1号梯检修开关" AND "1号梯门锁确认信号" AND NOT "1号梯下行接触器" AND NOT "1号梯超重信号" AND NOT "1号梯开门锁上下行",
                           PT := T#200MS);
   IF "IEC_Timer_0_DB_29".Q THEN
       "1号梯上行接触器" := TRUE;
       "1号梯低速运行" := TRUE;
       "1号梯低速转高速" := TRUE;
   END_IF;
   "IEC_Timer_0_DB_28".TON(IN := "1号梯低速转高速", PT := T#100MS);
   IF "IEC_Timer_0_DB_28".Q THEN
       "1号梯低速运行" := FALSE;
       "1号梯高速运行" := TRUE;
       "1号梯低速转高速" := FALSE;
   END_IF;
   IF "1号梯上行接触器" AND "1号梯平层信号" THEN "1号梯高速转低速" := TRUE; END_IF;
   IF "1号梯高速转低速" THEN
       "1号梯高速运行" := FALSE;
       "1号梯低速运行" := TRUE;
       "1号梯制动使能" := TRUE;
       "1号梯平层信号" := FALSE;
       "1号梯高速转低速" := FALSE;
   END_IF;
END_REGION

